REGION Network 8: PREMIXING_TEMP_CUTOUT
   RUNG wire#powerrail
      Contact( "AlwaysTRUE" )
      { S7_Templates := "SrcType := Int" } EQ_Contact(in1 := "MODE SELECTION DB"."MODE BUFF", in2 := 2)
      I_Contact( "DO MAPING"."PAV-13 WATER COOLING INLET" )
      Contact( "MANUAL BIT"."PAV-09 JACKET STEAM INLET" )
      Coil( "MANUAL BIT"."PAV-10 JACKET CONDENSATE DRAIN" )
   END_RUNG
   // the same network as SCL:
   "MANUAL BIT"."PAV-10 JACKET CONDENSATE DRAIN" := "AlwaysTRUE" AND ("MODE SELECTION DB"."MODE BUFF" = 2) AND NOT "DO MAPING"."PAV-13 WATER COOLING INLET" AND "MANUAL BIT"."PAV-09 JACKET STEAM INLET";
END_REGION

REGION Network 9: PREMIXING_COOLING_CUTOUT
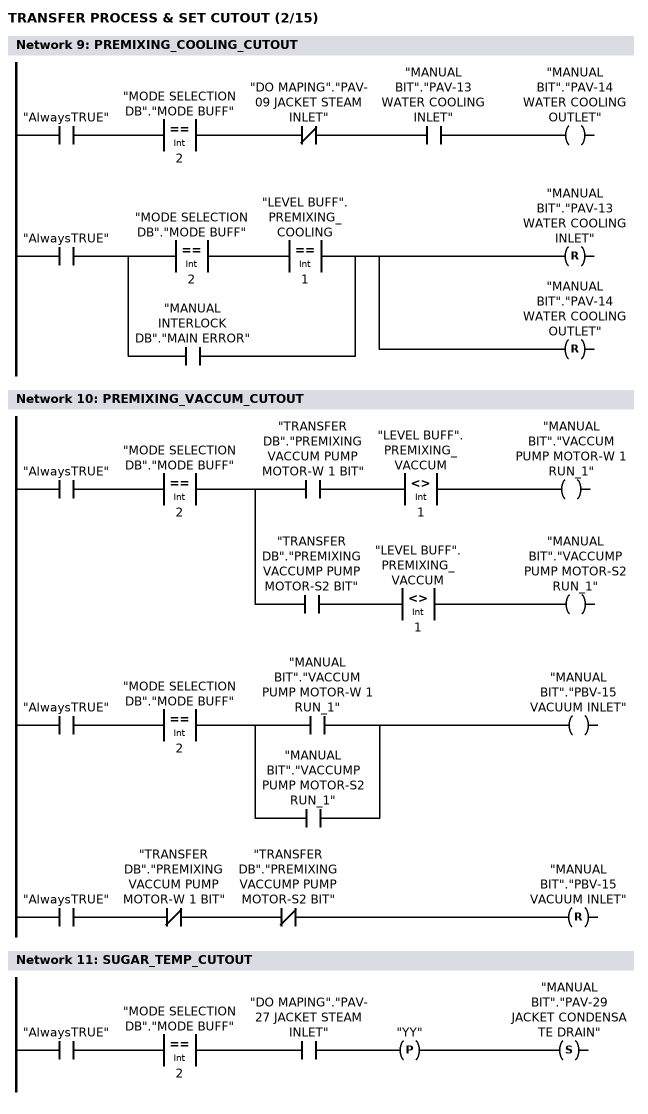
   RUNG wire#powerrail
      Contact( "AlwaysTRUE" )
      { S7_Templates := "SrcType := Int" } EQ_Contact(in1 := "MODE SELECTION DB"."MODE BUFF", in2 := 2)
      I_Contact( "DO MAPING"."PAV-09 JACKET STEAM INLET" )
      Contact( "MANUAL BIT"."PAV-13 WATER COOLING INLET" )
      Coil( "MANUAL BIT"."PAV-14 WATER COOLING OUTLET" )
   END_RUNG
   RUNG wire#powerrail
      Contact( "AlwaysTRUE" )
      wire#w1
      { S7_Templates := "SrcType := Int" } EQ_Contact(in1 := "MODE SELECTION DB"."MODE BUFF", in2 := 2)
      { S7_Templates := "SrcType := Int" } EQ_Contact(in1 := "LEVEL BUFF".PREMIXING_COOLING, in2 := 1)
      wire#w2
      R_Coil( "MANUAL BIT"."PAV-13 WATER COOLING INLET" )
   END_RUNG
   RUNG wire#w1
      Contact( "MANUAL INTERLOCK DB"."MAIN ERROR" )
   END_RUNG wire#w2
   RUNG wire#w2
      R_Coil( "MANUAL BIT"."PAV-14 WATER COOLING OUTLET" )
   END_RUNG
   // the same network as SCL:
   "MANUAL BIT"."PAV-14 WATER COOLING OUTLET" := "AlwaysTRUE" AND ("MODE SELECTION DB"."MODE BUFF" = 2) AND NOT "DO MAPING"."PAV-09 JACKET STEAM INLET" AND "MANUAL BIT"."PAV-13 WATER COOLING INLET";
   IF "AlwaysTRUE" AND ((("MODE SELECTION DB"."MODE BUFF" = 2) AND ("LEVEL BUFF".PREMIXING_COOLING = 1)) OR "MANUAL INTERLOCK DB"."MAIN ERROR") THEN
       "MANUAL BIT"."PAV-13 WATER COOLING INLET" := FALSE;
       "MANUAL BIT"."PAV-14 WATER COOLING OUTLET" := FALSE;
   END_IF;
END_REGION

REGION Network 10: PREMIXING_VACCUM_CUTOUT
   RUNG wire#powerrail
      Contact( "AlwaysTRUE" )
      { S7_Templates := "SrcType := Int" } EQ_Contact(in1 := "MODE SELECTION DB"."MODE BUFF", in2 := 2)
      wire#w1
      Contact( "TRANSFER DB"."PREMIXING VACCUM PUMP MOTOR-W 1 BIT" )
      { S7_Templates := "SrcType := Int" } NE_Contact(in1 := "LEVEL BUFF".PREMIXING_VACCUM, in2 := 1)
      Coil( "MANUAL BIT"."VACCUM PUMP MOTOR-W 1 RUN_1" )
   END_RUNG
   RUNG wire#w1
      Contact( "TRANSFER DB"."PREMIXING VACCUMP PUMP MOTOR-S2 BIT" )
      { S7_Templates := "SrcType := Int" } NE_Contact(in1 := "LEVEL BUFF".PREMIXING_VACCUM, in2 := 1)
      Coil( "MANUAL BIT"."VACCUMP PUMP MOTOR-S2 RUN_1" )
   END_RUNG
   RUNG wire#powerrail
      Contact( "AlwaysTRUE" )
      { S7_Templates := "SrcType := Int" } EQ_Contact(in1 := "MODE SELECTION DB"."MODE BUFF", in2 := 2)
      wire#w2
      Contact( "MANUAL BIT"."VACCUM PUMP MOTOR-W 1 RUN_1" )
      wire#w3
      Coil( "MANUAL BIT"."PBV-15 VACUUM INLET" )
   END_RUNG
   RUNG wire#w2
      Contact( "MANUAL BIT"."VACCUMP PUMP MOTOR-S2 RUN_1" )
   END_RUNG wire#w3
   RUNG wire#powerrail
      Contact( "AlwaysTRUE" )
      I_Contact( "TRANSFER DB"."PREMIXING VACCUM PUMP MOTOR-W 1 BIT" )
      I_Contact( "TRANSFER DB"."PREMIXING VACCUMP PUMP MOTOR-S2 BIT" )
      R_Coil( "MANUAL BIT"."PBV-15 VACUUM INLET" )
   END_RUNG
   // the same network as SCL:
   #_w1 := "AlwaysTRUE" AND ("MODE SELECTION DB"."MODE BUFF" = 2);
   "MANUAL BIT"."VACCUM PUMP MOTOR-W 1 RUN_1" := #_w1 AND "TRANSFER DB"."PREMIXING VACCUM PUMP MOTOR-W 1 BIT" AND ("LEVEL BUFF".PREMIXING_VACCUM <> 1);
   "MANUAL BIT"."VACCUMP PUMP MOTOR-S2 RUN_1" := #_w1 AND "TRANSFER DB"."PREMIXING VACCUMP PUMP MOTOR-S2 BIT" AND ("LEVEL BUFF".PREMIXING_VACCUM <> 1);
   "MANUAL BIT"."PBV-15 VACUUM INLET" := "AlwaysTRUE" AND ("MODE SELECTION DB"."MODE BUFF" = 2) AND ("MANUAL BIT"."VACCUM PUMP MOTOR-W 1 RUN_1" OR "MANUAL BIT"."VACCUMP PUMP MOTOR-S2 RUN_1");
   IF "AlwaysTRUE" AND NOT "TRANSFER DB"."PREMIXING VACCUM PUMP MOTOR-W 1 BIT" AND NOT "TRANSFER DB"."PREMIXING VACCUMP PUMP MOTOR-S2 BIT" THEN
       "MANUAL BIT"."PBV-15 VACUUM INLET" := FALSE;
   END_IF;
END_REGION

REGION Network 11: SUGAR_TEMP_CUTOUT
   RUNG wire#powerrail
      Contact( "AlwaysTRUE" )
      { S7_Templates := "SrcType := Int" } EQ_Contact(in1 := "MODE SELECTION DB"."MODE BUFF", in2 := 2)
      Contact( "DO MAPING"."PAV-27 JACKET STEAM INLET" )
      P_Trig( "YY" )
      S_Coil( "MANUAL BIT"."PAV-29 JACKET CONDENSATE DRAIN" )
   END_RUNG
   // the same network as SCL:
   #_w1 := "AlwaysTRUE" AND ("MODE SELECTION DB"."MODE BUFF" = 2) AND "DO MAPING"."PAV-27 JACKET STEAM INLET";
   #_w2 := #_w1 AND NOT "YY";   // rising edge
   "YY" := #_w1;
   IF #_w2 THEN "MANUAL BIT"."PAV-29 JACKET CONDENSATE DRAIN" := TRUE; END_IF;
END_REGION

REGION Network 12: SUGAR_VACCUM_CUTOUT
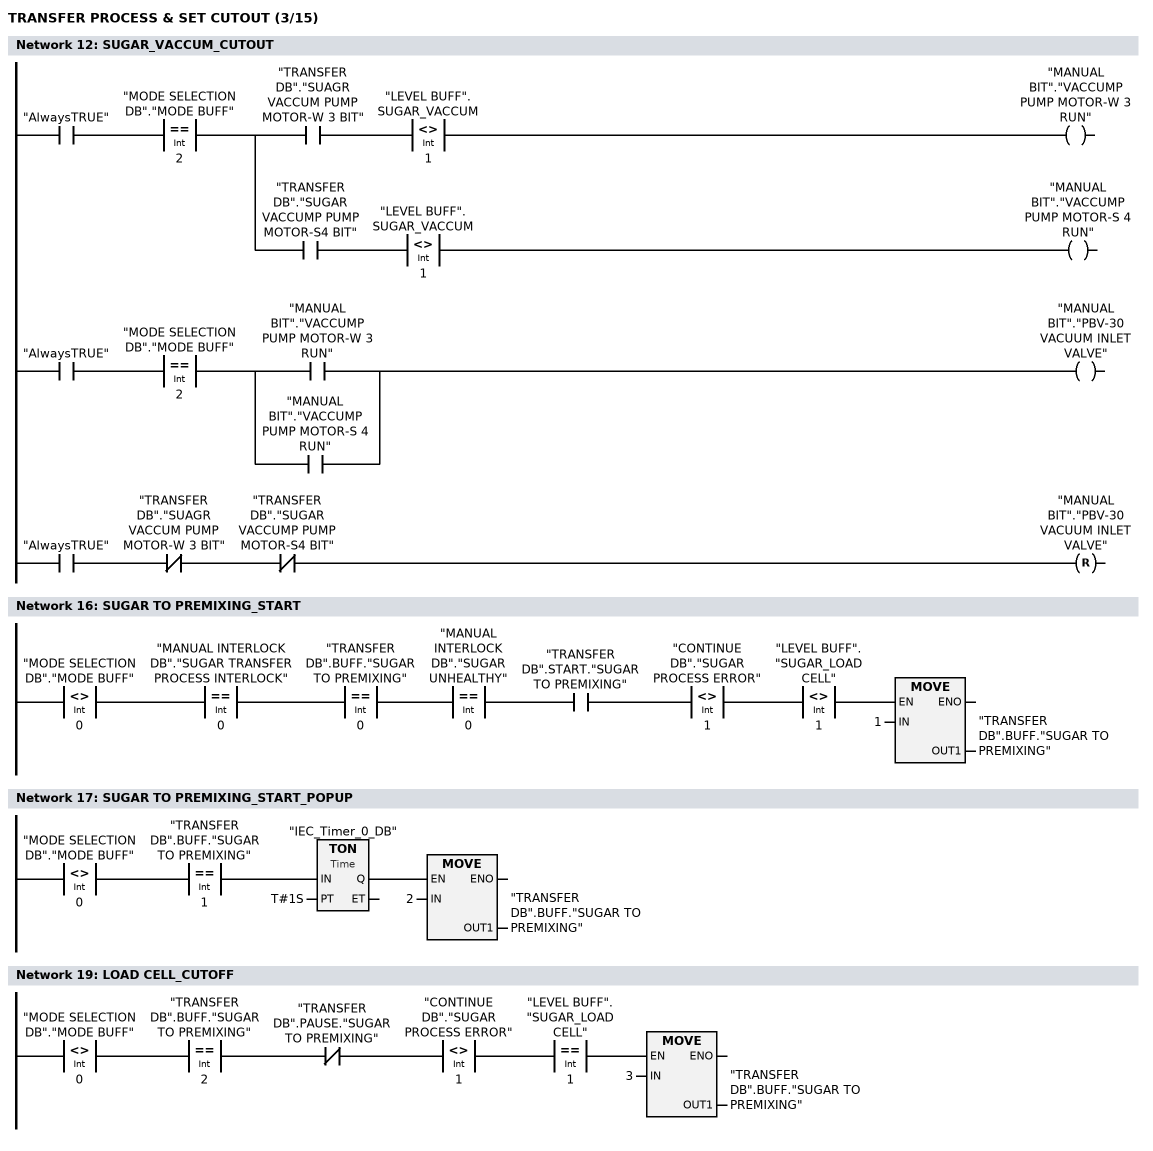
   RUNG wire#powerrail
      Contact( "AlwaysTRUE" )
      { S7_Templates := "SrcType := Int" } EQ_Contact(in1 := "MODE SELECTION DB"."MODE BUFF", in2 := 2)
      wire#w1
      Contact( "TRANSFER DB"."SUAGR VACCUM PUMP MOTOR-W 3 BIT" )
      { S7_Templates := "SrcType := Int" } NE_Contact(in1 := "LEVEL BUFF".SUGAR_VACCUM, in2 := 1)
      Coil( "MANUAL BIT"."VACCUMP PUMP MOTOR-W 3 RUN" )
   END_RUNG
   RUNG wire#w1
      Contact( "TRANSFER DB"."SUGAR VACCUMP PUMP MOTOR-S4 BIT" )
      { S7_Templates := "SrcType := Int" } NE_Contact(in1 := "LEVEL BUFF".SUGAR_VACCUM, in2 := 1)
      Coil( "MANUAL BIT"."VACCUMP PUMP MOTOR-S 4 RUN" )
   END_RUNG
   RUNG wire#powerrail
      Contact( "AlwaysTRUE" )
      { S7_Templates := "SrcType := Int" } EQ_Contact(in1 := "MODE SELECTION DB"."MODE BUFF", in2 := 2)
      wire#w2
      Contact( "MANUAL BIT"."VACCUMP PUMP MOTOR-W 3 RUN" )
      wire#w3
      Coil( "MANUAL BIT"."PBV-30 VACUUM INLET VALVE" )
   END_RUNG
   RUNG wire#w2
      Contact( "MANUAL BIT"."VACCUMP PUMP MOTOR-S 4 RUN" )
   END_RUNG wire#w3
   RUNG wire#powerrail
      Contact( "AlwaysTRUE" )
      I_Contact( "TRANSFER DB"."SUAGR VACCUM PUMP MOTOR-W 3 BIT" )
      I_Contact( "TRANSFER DB"."SUGAR VACCUMP PUMP MOTOR-S4 BIT" )
      R_Coil( "MANUAL BIT"."PBV-30 VACUUM INLET VALVE" )
   END_RUNG
   // the same network as SCL:
   #_w1 := "AlwaysTRUE" AND ("MODE SELECTION DB"."MODE BUFF" = 2);
   "MANUAL BIT"."VACCUMP PUMP MOTOR-W 3 RUN" := #_w1 AND "TRANSFER DB"."SUAGR VACCUM PUMP MOTOR-W 3 BIT" AND ("LEVEL BUFF".SUGAR_VACCUM <> 1);
   "MANUAL BIT"."VACCUMP PUMP MOTOR-S 4 RUN" := #_w1 AND "TRANSFER DB"."SUGAR VACCUMP PUMP MOTOR-S4 BIT" AND ("LEVEL BUFF".SUGAR_VACCUM <> 1);
   "MANUAL BIT"."PBV-30 VACUUM INLET VALVE" := "AlwaysTRUE" AND ("MODE SELECTION DB"."MODE BUFF" = 2) AND ("MANUAL BIT"."VACCUMP PUMP MOTOR-W 3 RUN" OR "MANUAL BIT"."VACCUMP PUMP MOTOR-S 4 RUN");
   IF "AlwaysTRUE" AND NOT "TRANSFER DB"."SUAGR VACCUM PUMP MOTOR-W 3 BIT" AND NOT "TRANSFER DB"."SUGAR VACCUMP PUMP MOTOR-S4 BIT" THEN
       "MANUAL BIT"."PBV-30 VACUUM INLET VALVE" := FALSE;
   END_IF;
END_REGION

REGION Network 15: ////////////////////////////////////////////////////////////////////// TRANSFER PROCESS- SUGAR //////////////////////////////////////////////////////////////////////////////////
END_REGION

REGION Network 16: SUGAR TO PREMIXING_START
   RUNG wire#powerrail
      { S7_Templates := "SrcType := Int" } NE_Contact(in1 := "MODE SELECTION DB"."MODE BUFF", in2 := 0)
      { S7_Templates := "SrcType := Int" } EQ_Contact(in1 := "MANUAL INTERLOCK DB"."SUGAR TRANSFER PROCESS INTERLOCK", in2 := 0)
      { S7_Templates := "SrcType := Int" } EQ_Contact(in1 := "TRANSFER DB".BUFF."SUGAR TO PREMIXING", in2 := 0)
      { S7_Templates := "SrcType := Int" } EQ_Contact(in1 := "MANUAL INTERLOCK DB"."SUGAR UNHEALTHY", in2 := 0)
      Contact( "TRANSFER DB".START."SUGAR TO PREMIXING" )
      { S7_Templates := "SrcType := Int" } NE_Contact(in1 := "CONTINUE DB"."SUGAR PROCESS ERROR", in2 := 1)
      { S7_Templates := "SrcType := Int" } NE_Contact(in1 := "LEVEL BUFF"."SUGAR_LOAD CELL", in2 := 1)
      Move(in := 1, out1 => "TRANSFER DB".BUFF."SUGAR TO PREMIXING")
   END_RUNG
   // the same network as SCL:
   IF ("MODE SELECTION DB"."MODE BUFF" <> 0) AND ("MANUAL INTERLOCK DB"."SUGAR TRANSFER PROCESS INTERLOCK" = 0) AND ("TRANSFER DB".BUFF."SUGAR TO PREMIXING" = 0) AND ("MANUAL INTERLOCK DB"."SUGAR UNHEALTHY" = 0) AND "TRANSFER DB".START."SUGAR TO PREMIXING" AND ("CONTINUE DB"."SUGAR PROCESS ERROR" <> 1) AND ("LEVEL BUFF"."SUGAR_LOAD CELL" <> 1) THEN
       "TRANSFER DB".BUFF."SUGAR TO PREMIXING" := 1;
   END_IF;
END_REGION

REGION Network 17: SUGAR TO PREMIXING_START_POPUP
   RUNG wire#powerrail
      { S7_Templates := "SrcType := Int" } NE_Contact(in1 := "MODE SELECTION DB"."MODE BUFF", in2 := 0)
      { S7_Templates := "SrcType := Int" } EQ_Contact(in1 := "TRANSFER DB".BUFF."SUGAR TO PREMIXING", in2 := 1)
      { S7_Templates := "time_type := Time" } "IEC_Timer_0_DB".TON(pt := T#1S, et =>)
      Move(in := 2, out1 => "TRANSFER DB".BUFF."SUGAR TO PREMIXING")
   END_RUNG
   // the same network as SCL:
   "IEC_Timer_0_DB".TON(IN := ("MODE SELECTION DB"."MODE BUFF" <> 0) AND ("TRANSFER DB".BUFF."SUGAR TO PREMIXING" = 1),
                        PT := T#1S);
   IF "IEC_Timer_0_DB".Q THEN "TRANSFER DB".BUFF."SUGAR TO PREMIXING" := 2; END_IF;
END_REGION

REGION Network 18 (SCL): OPENVALVE
   IF "MODE SELECTION DB"."MODE BUFF" <> 0 AND "TRANSFER DB".BUFF."SUGAR TO PREMIXING" = 2
       AND NOT "TRANSFER DB".PAUSE."SUGAR TO PREMIXING" AND
       "CONTINUE DB"."SUGAR PROCESS ERROR" = 0 AND "LEVEL BUFF"."SUGAR_LOAD CELL" = 0
       OR ("MODE SELECTION DB"."MODE BUFF"=1 AND "SUGAR DB"."AUTO BUFF"=105
       AND "CONTINUE DB"."SUGAR PROCESS ERROR" <>1)
   THEN
       "TRANSFER DB".BIT."SUGAR TO PREMIXING"."PFBV-32 TANK OUTLET VALVE" := TRUE;
       "TRANSFER DB".BIT."SUGAR TO PREMIXING"."PBV-80 BOTTOM OUTLET TO BASKET FILTER" := TRUE;
       "TRANSFER DB".BIT."SUGAR TO PREMIXING"."BASKET FILTER MOTOR RUN" := TRUE;
       "TRANSFER DB".BIT."SUGAR TO PREMIXING"."PBV-79 BASKET FILTER INLET" := TRUE;
       "TRANSFER DB".BIT."SUGAR TO PREMIXING"."PBV-149" := TRUE;
       "TRANSFER DB".BIT."SUGAR TO PREMIXING"."PBV-88 BASKET FILTER TRANSFER LINE" := TRUE;
       "TRANSFER DB".BIT."SUGAR TO PREMIXING"."PBV-87 BASKET FILTER TO PREMIX VESSEL LINE" := TRUE;
   ELSE
       "TRANSFER DB".BIT."SUGAR TO PREMIXING"."PFBV-32 TANK OUTLET VALVE" := FALSE;
       "TRANSFER DB".BIT."SUGAR TO PREMIXING"."PBV-80 BOTTOM OUTLET TO BASKET FILTER" := FALSE;
       "TRANSFER DB".BIT."SUGAR TO PREMIXING"."BASKET FILTER MOTOR RUN" := FALSE;
       "TRANSFER DB".BIT."SUGAR TO PREMIXING"."PBV-79 BASKET FILTER INLET" := FALSE;
       "TRANSFER DB".BIT."SUGAR TO PREMIXING"."PBV-149" := FALSE;
       "TRANSFER DB".BIT."SUGAR TO PREMIXING"."PBV-88 BASKET FILTER TRANSFER LINE" := FALSE;
       "TRANSFER DB".BIT."SUGAR TO PREMIXING"."PBV-87 BASKET FILTER TO PREMIX VESSEL LINE" := FALSE;
       ;
   END_IF;
END_REGION

REGION Network 19: LOAD CELL_CUTOFF
   RUNG wire#powerrail
      { S7_Templates := "SrcType := Int" } NE_Contact(in1 := "MODE SELECTION DB"."MODE BUFF", in2 := 0)
      { S7_Templates := "SrcType := Int" } EQ_Contact(in1 := "TRANSFER DB".BUFF."SUGAR TO PREMIXING", in2 := 2)
      I_Contact( "TRANSFER DB".PAUSE."SUGAR TO PREMIXING" )
      { S7_Templates := "SrcType := Int" } NE_Contact(in1 := "CONTINUE DB"."SUGAR PROCESS ERROR", in2 := 1)
      { S7_Templates := "SrcType := Int" } EQ_Contact(in1 := "LEVEL BUFF"."SUGAR_LOAD CELL", in2 := 1)
      Move(in := 3, out1 => "TRANSFER DB".BUFF."SUGAR TO PREMIXING")
   END_RUNG
   // the same network as SCL:
   IF ("MODE SELECTION DB"."MODE BUFF" <> 0) AND ("TRANSFER DB".BUFF."SUGAR TO PREMIXING" = 2) AND NOT "TRANSFER DB".PAUSE."SUGAR TO PREMIXING" AND ("CONTINUE DB"."SUGAR PROCESS ERROR" <> 1) AND ("LEVEL BUFF"."SUGAR_LOAD CELL" = 1) THEN
       "TRANSFER DB".BUFF."SUGAR TO PREMIXING" := 3;
   END_IF;
END_REGION

REGION Network 20: PROCESS OVER & STOP
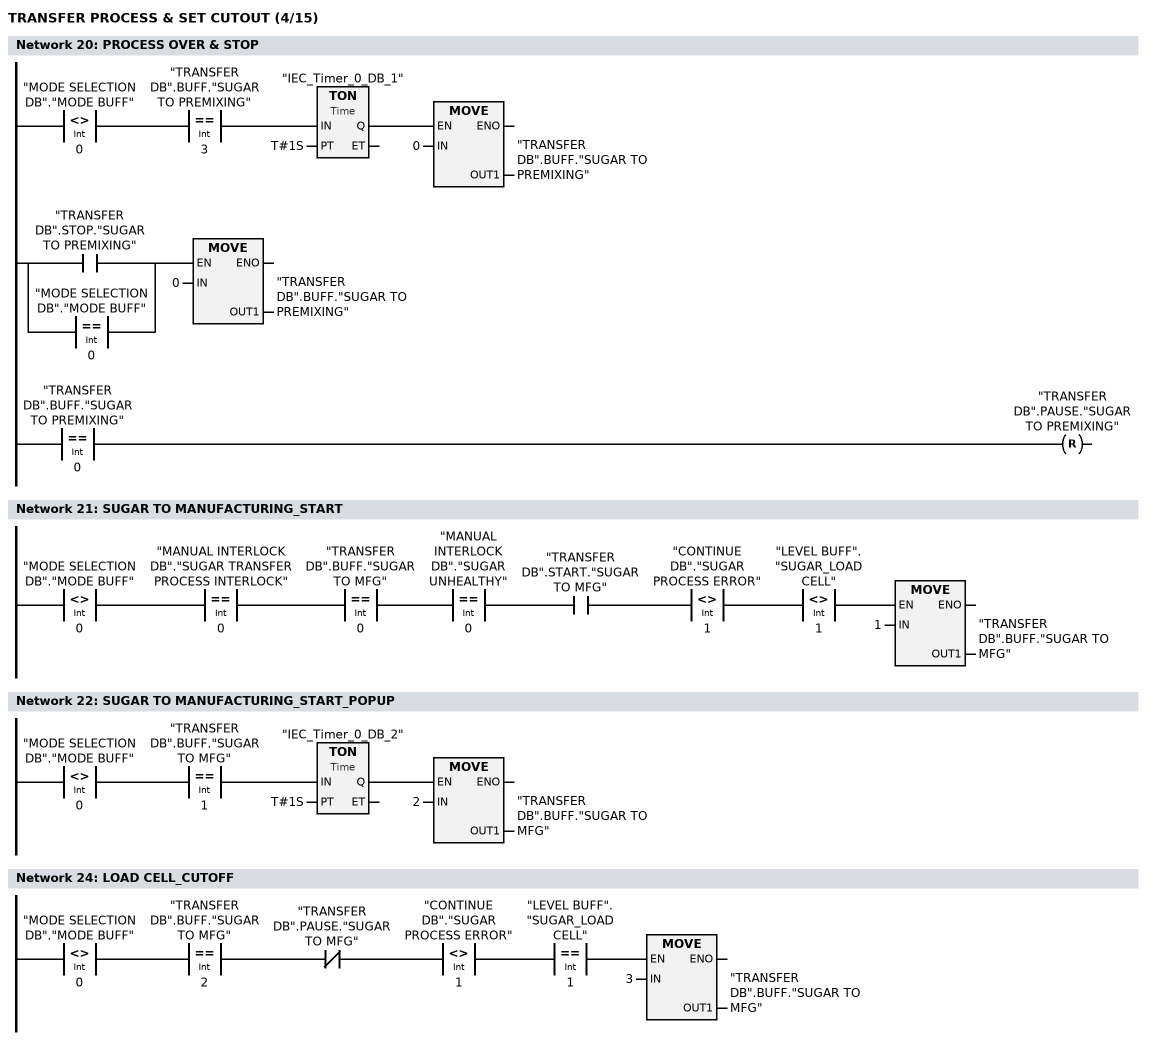
   RUNG wire#powerrail
      { S7_Templates := "SrcType := Int" } NE_Contact(in1 := "MODE SELECTION DB"."MODE BUFF", in2 := 0)
      { S7_Templates := "SrcType := Int" } EQ_Contact(in1 := "TRANSFER DB".BUFF."SUGAR TO PREMIXING", in2 := 3)
      { S7_Templates := "time_type := Time" } "IEC_Timer_0_DB_1".TON(pt := T#1S, et =>)
      Move(in := 0, out1 => "TRANSFER DB".BUFF."SUGAR TO PREMIXING")
   END_RUNG
   RUNG wire#powerrail
      Contact( "TRANSFER DB".STOP."SUGAR TO PREMIXING" )
      wire#w1
      Move(in := 0, out1 => "TRANSFER DB".BUFF."SUGAR TO PREMIXING")
   END_RUNG
   RUNG wire#powerrail
      { S7_Templates := "SrcType := Int" } EQ_Contact(in1 := "MODE SELECTION DB"."MODE BUFF", in2 := 0)
   END_RUNG wire#w1
   RUNG wire#powerrail
      { S7_Templates := "SrcType := Int" } EQ_Contact(in1 := "TRANSFER DB".BUFF."SUGAR TO PREMIXING", in2 := 0)
      R_Coil( "TRANSFER DB".PAUSE."SUGAR TO PREMIXING" )
   END_RUNG
   // the same network as SCL:
   "IEC_Timer_0_DB_1".TON(IN := ("MODE SELECTION DB"."MODE BUFF" <> 0) AND ("TRANSFER DB".BUFF."SUGAR TO PREMIXING" = 3),
                          PT := T#1S);
   IF "IEC_Timer_0_DB_1".Q THEN "TRANSFER DB".BUFF."SUGAR TO PREMIXING" := 0; END_IF;
   IF "TRANSFER DB".STOP."SUGAR TO PREMIXING" OR ("MODE SELECTION DB"."MODE BUFF" = 0) THEN
       "TRANSFER DB".BUFF."SUGAR TO PREMIXING" := 0;
   END_IF;
   IF "TRANSFER DB".BUFF."SUGAR TO PREMIXING" = 0 THEN
       "TRANSFER DB".PAUSE."SUGAR TO PREMIXING" := FALSE;
   END_IF;
END_REGION

REGION Network 21: SUGAR TO MANUFACTURING_START
   RUNG wire#powerrail
      { S7_Templates := "SrcType := Int" } NE_Contact(in1 := "MODE SELECTION DB"."MODE BUFF", in2 := 0)
      { S7_Templates := "SrcType := Int" } EQ_Contact(in1 := "MANUAL INTERLOCK DB"."SUGAR TRANSFER PROCESS INTERLOCK", in2 := 0)
      { S7_Templates := "SrcType := Int" } EQ_Contact(in1 := "TRANSFER DB".BUFF."SUGAR TO MFG", in2 := 0)
      { S7_Templates := "SrcType := Int" } EQ_Contact(in1 := "MANUAL INTERLOCK DB"."SUGAR UNHEALTHY", in2 := 0)
      Contact( "TRANSFER DB".START."SUGAR TO MFG" )
      { S7_Templates := "SrcType := Int" } NE_Contact(in1 := "CONTINUE DB"."SUGAR PROCESS ERROR", in2 := 1)
      { S7_Templates := "SrcType := Int" } NE_Contact(in1 := "LEVEL BUFF"."SUGAR_LOAD CELL", in2 := 1)
      Move(in := 1, out1 => "TRANSFER DB".BUFF."SUGAR TO MFG")
   END_RUNG
   // the same network as SCL:
   IF ("MODE SELECTION DB"."MODE BUFF" <> 0) AND ("MANUAL INTERLOCK DB"."SUGAR TRANSFER PROCESS INTERLOCK" = 0) AND ("TRANSFER DB".BUFF."SUGAR TO MFG" = 0) AND ("MANUAL INTERLOCK DB"."SUGAR UNHEALTHY" = 0) AND "TRANSFER DB".START."SUGAR TO MFG" AND ("CONTINUE DB"."SUGAR PROCESS ERROR" <> 1) AND ("LEVEL BUFF"."SUGAR_LOAD CELL" <> 1) THEN
       "TRANSFER DB".BUFF."SUGAR TO MFG" := 1;
   END_IF;
END_REGION

REGION Network 22: SUGAR TO MANUFACTURING_START_POPUP
   RUNG wire#powerrail
      { S7_Templates := "SrcType := Int" } NE_Contact(in1 := "MODE SELECTION DB"."MODE BUFF", in2 := 0)
      { S7_Templates := "SrcType := Int" } EQ_Contact(in1 := "TRANSFER DB".BUFF."SUGAR TO MFG", in2 := 1)
      { S7_Templates := "time_type := Time" } "IEC_Timer_0_DB_2".TON(pt := T#1S, et =>)
      Move(in := 2, out1 => "TRANSFER DB".BUFF."SUGAR TO MFG")
   END_RUNG
   // the same network as SCL:
   "IEC_Timer_0_DB_2".TON(IN := ("MODE SELECTION DB"."MODE BUFF" <> 0) AND ("TRANSFER DB".BUFF."SUGAR TO MFG" = 1),
                          PT := T#1S);
   IF "IEC_Timer_0_DB_2".Q THEN "TRANSFER DB".BUFF."SUGAR TO MFG" := 2; END_IF;
END_REGION

REGION Network 23 (SCL): OPENVALVE
   IF "MODE SELECTION DB"."MODE BUFF" <> 0 AND "TRANSFER DB".BUFF."SUGAR TO MFG" = 2
       AND NOT "TRANSFER DB".PAUSE."SUGAR TO MFG" 
       AND "CONTINUE DB"."SUGAR PROCESS ERROR" = 0 AND "LEVEL BUFF"."SUGAR_LOAD CELL" = 0
       OR ("MODE SELECTION DB"."MODE BUFF"=1 AND "SUGAR DB"."AUTO BUFF"=125
       AND "CONTINUE DB"."SUGAR PROCESS ERROR" <>1)
   THEN
       "TRANSFER DB".BIT."SUGAR TO MFG"."PFBV-32 TANK OUTLET VALVE" := TRUE;
       "TRANSFER DB".BIT."SUGAR TO MFG"."PBV-80 BOTTOM OUTLET TO BASKET FILTER" := TRUE;
       "TRANSFER DB".BIT."SUGAR TO MFG"."BASKET FILTER MOTOR RUN" := TRUE;
       "TRANSFER DB".BIT."SUGAR TO MFG"."PBV-79 BASKET FILTER INLET" := TRUE;
       "TRANSFER DB".BIT."SUGAR TO MFG"."PBV-149" := TRUE;
       "TRANSFER DB".BIT."SUGAR TO MFG"."PBV-89 BASKET FILTER TO MFG INLET TRANSFER LINE" := TRUE;
       "TRANSFER DB".BIT."SUGAR TO MFG"."PBV-101 SUGAR MELTING TO MFG TRANSFER (TOP DISH)" := TRUE;

   ELSE
       "TRANSFER DB".BIT."SUGAR TO MFG"."PFBV-32 TANK OUTLET VALVE" := FALSE;
       "TRANSFER DB".BIT."SUGAR TO MFG"."PBV-80 BOTTOM OUTLET TO BASKET FILTER" := FALSE;
       "TRANSFER DB".BIT."SUGAR TO MFG"."BASKET FILTER MOTOR RUN" := FALSE;
       "TRANSFER DB".BIT."SUGAR TO MFG"."PBV-79 BASKET FILTER INLET" := FALSE;
       "TRANSFER DB".BIT."SUGAR TO MFG"."PBV-149" := FALSE;
       "TRANSFER DB".BIT."SUGAR TO MFG"."PBV-89 BASKET FILTER TO MFG INLET TRANSFER LINE" := FALSE;
       "TRANSFER DB".BIT."SUGAR TO MFG"."PBV-101 SUGAR MELTING TO MFG TRANSFER (TOP DISH)" := FALSE;
       ;
   END_IF;
END_REGION

REGION Network 24: LOAD CELL_CUTOFF
   RUNG wire#powerrail
      { S7_Templates := "SrcType := Int" } NE_Contact(in1 := "MODE SELECTION DB"."MODE BUFF", in2 := 0)
      { S7_Templates := "SrcType := Int" } EQ_Contact(in1 := "TRANSFER DB".BUFF."SUGAR TO MFG", in2 := 2)
      I_Contact( "TRANSFER DB".PAUSE."SUGAR TO MFG" )
      { S7_Templates := "SrcType := Int" } NE_Contact(in1 := "CONTINUE DB"."SUGAR PROCESS ERROR", in2 := 1)
      { S7_Templates := "SrcType := Int" } EQ_Contact(in1 := "LEVEL BUFF"."SUGAR_LOAD CELL", in2 := 1)
      Move(in := 3, out1 => "TRANSFER DB".BUFF."SUGAR TO MFG")
   END_RUNG
   // the same network as SCL:
   IF ("MODE SELECTION DB"."MODE BUFF" <> 0) AND ("TRANSFER DB".BUFF."SUGAR TO MFG" = 2) AND NOT "TRANSFER DB".PAUSE."SUGAR TO MFG" AND ("CONTINUE DB"."SUGAR PROCESS ERROR" <> 1) AND ("LEVEL BUFF"."SUGAR_LOAD CELL" = 1) THEN
       "TRANSFER DB".BUFF."SUGAR TO MFG" := 3;
   END_IF;
END_REGION

REGION Network 25: PROCESS OVER & STOP
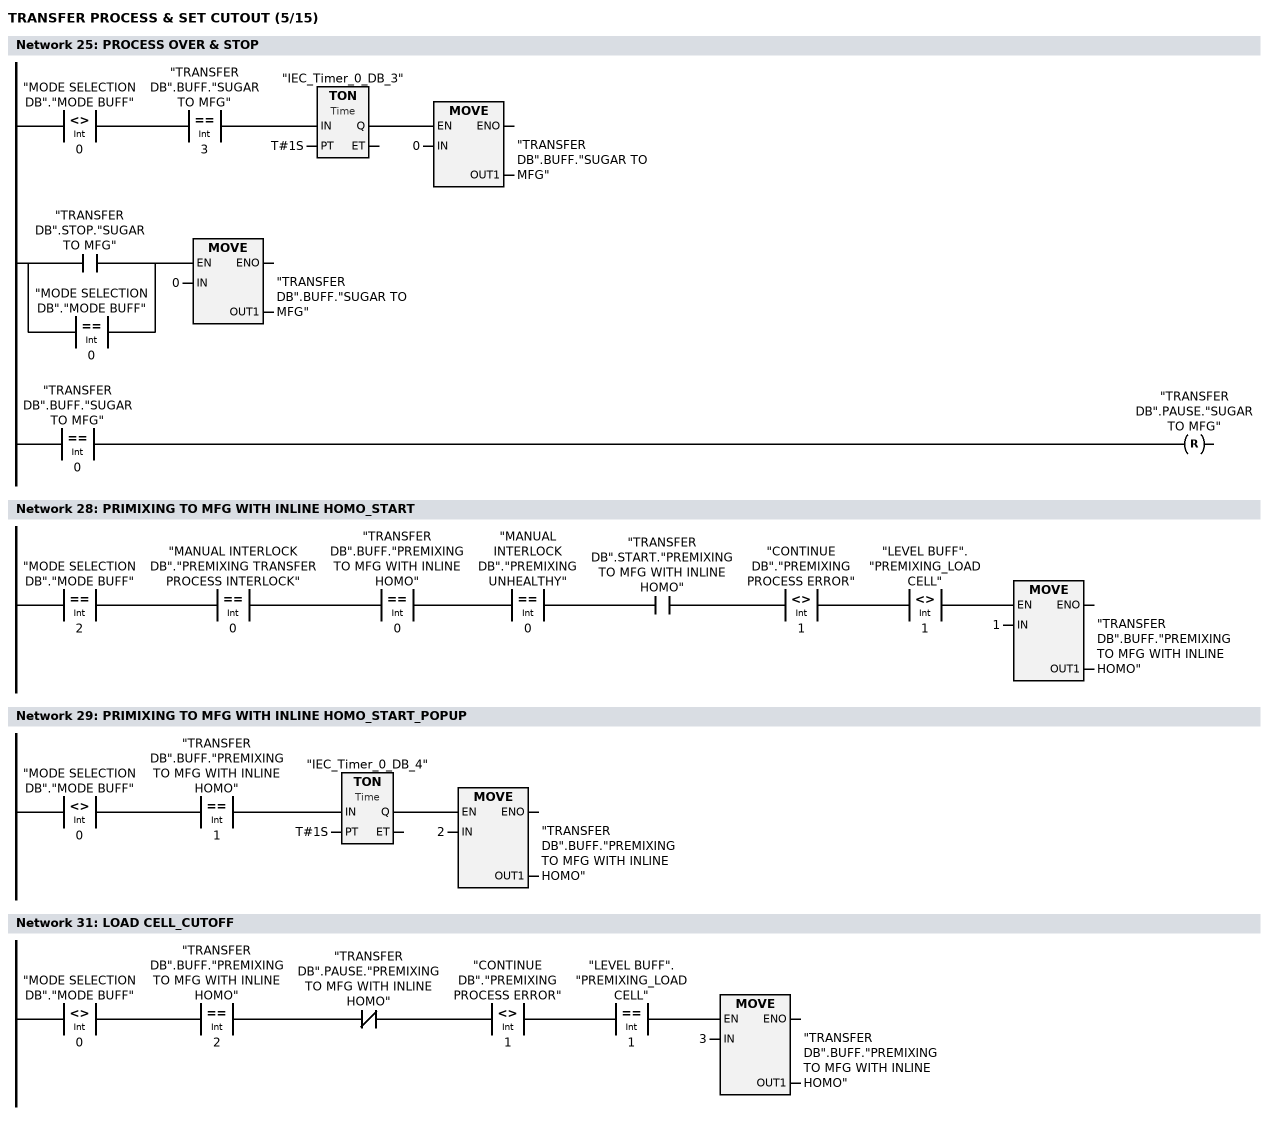
   RUNG wire#powerrail
      { S7_Templates := "SrcType := Int" } NE_Contact(in1 := "MODE SELECTION DB"."MODE BUFF", in2 := 0)
      { S7_Templates := "SrcType := Int" } EQ_Contact(in1 := "TRANSFER DB".BUFF."SUGAR TO MFG", in2 := 3)
      { S7_Templates := "time_type := Time" } "IEC_Timer_0_DB_3".TON(pt := T#1S, et =>)
      Move(in := 0, out1 => "TRANSFER DB".BUFF."SUGAR TO MFG")
   END_RUNG
   RUNG wire#powerrail
      Contact( "TRANSFER DB".STOP."SUGAR TO MFG" )
      wire#w1
      Move(in := 0, out1 => "TRANSFER DB".BUFF."SUGAR TO MFG")
   END_RUNG
   RUNG wire#powerrail
      { S7_Templates := "SrcType := Int" } EQ_Contact(in1 := "MODE SELECTION DB"."MODE BUFF", in2 := 0)
   END_RUNG wire#w1
   RUNG wire#powerrail
      { S7_Templates := "SrcType := Int" } EQ_Contact(in1 := "TRANSFER DB".BUFF."SUGAR TO MFG", in2 := 0)
      R_Coil( "TRANSFER DB".PAUSE."SUGAR TO MFG" )
   END_RUNG
   // the same network as SCL:
   "IEC_Timer_0_DB_3".TON(IN := ("MODE SELECTION DB"."MODE BUFF" <> 0) AND ("TRANSFER DB".BUFF."SUGAR TO MFG" = 3),
                          PT := T#1S);
   IF "IEC_Timer_0_DB_3".Q THEN "TRANSFER DB".BUFF."SUGAR TO MFG" := 0; END_IF;
   IF "TRANSFER DB".STOP."SUGAR TO MFG" OR ("MODE SELECTION DB"."MODE BUFF" = 0) THEN
       "TRANSFER DB".BUFF."SUGAR TO MFG" := 0;
   END_IF;
   IF "TRANSFER DB".BUFF."SUGAR TO MFG" = 0 THEN "TRANSFER DB".PAUSE."SUGAR TO MFG" := FALSE; END_IF;
END_REGION

REGION Network 27: ////////////////////////////////////////////////////////////////////// TRANSFER PROCESS- PREMIXING //////////////////////////////////////////////////////////////////////////////////
END_REGION

REGION Network 28: PRIMIXING TO MFG WITH INLINE HOMO_START
   RUNG wire#powerrail
      { S7_Templates := "SrcType := Int" } EQ_Contact(in1 := "MODE SELECTION DB"."MODE BUFF", in2 := 2)
      { S7_Templates := "SrcType := Int" } EQ_Contact(in1 := "MANUAL INTERLOCK DB"."PREMIXING TRANSFER PROCESS INTERLOCK", in2 := 0)
      { S7_Templates := "SrcType := Int" } EQ_Contact(in1 := "TRANSFER DB".BUFF."PREMIXING TO MFG WITH INLINE HOMO", in2 := 0)
      { S7_Templates := "SrcType := Int" } EQ_Contact(in1 := "MANUAL INTERLOCK DB"."PREMIXING UNHEALTHY", in2 := 0)
      Contact( "TRANSFER DB".START."PREMIXING TO MFG WITH INLINE HOMO" )
      { S7_Templates := "SrcType := Int" } NE_Contact(in1 := "CONTINUE DB"."PREMIXING PROCESS ERROR", in2 := 1)
      { S7_Templates := "SrcType := Int" } NE_Contact(in1 := "LEVEL BUFF"."PREMIXING_LOAD CELL", in2 := 1)
      Move(in := 1, out1 => "TRANSFER DB".BUFF."PREMIXING TO MFG WITH INLINE HOMO")
   END_RUNG
   // the same network as SCL:
   IF ("MODE SELECTION DB"."MODE BUFF" = 2) AND ("MANUAL INTERLOCK DB"."PREMIXING TRANSFER PROCESS INTERLOCK" = 0) AND ("TRANSFER DB".BUFF."PREMIXING TO MFG WITH INLINE HOMO" = 0) AND ("MANUAL INTERLOCK DB"."PREMIXING UNHEALTHY" = 0) AND "TRANSFER DB".START."PREMIXING TO MFG WITH INLINE HOMO" AND ("CONTINUE DB"."PREMIXING PROCESS ERROR" <> 1) AND ("LEVEL BUFF"."PREMIXING_LOAD CELL" <> 1) THEN
       "TRANSFER DB".BUFF."PREMIXING TO MFG WITH INLINE HOMO" := 1;
   END_IF;
END_REGION

REGION Network 29: PRIMIXING TO MFG WITH INLINE HOMO_START_POPUP
   RUNG wire#powerrail
      { S7_Templates := "SrcType := Int" } NE_Contact(in1 := "MODE SELECTION DB"."MODE BUFF", in2 := 0)
      { S7_Templates := "SrcType := Int" } EQ_Contact(in1 := "TRANSFER DB".BUFF."PREMIXING TO MFG WITH INLINE HOMO", in2 := 1)
      { S7_Templates := "time_type := Time" } "IEC_Timer_0_DB_4".TON(pt := T#1S, et =>)
      Move(in := 2, out1 => "TRANSFER DB".BUFF."PREMIXING TO MFG WITH INLINE HOMO")
   END_RUNG
   // the same network as SCL:
   "IEC_Timer_0_DB_4".TON(IN := ("MODE SELECTION DB"."MODE BUFF" <> 0) AND ("TRANSFER DB".BUFF."PREMIXING TO MFG WITH INLINE HOMO" = 1),
                          PT := T#1S);
   IF "IEC_Timer_0_DB_4".Q THEN "TRANSFER DB".BUFF."PREMIXING TO MFG WITH INLINE HOMO" := 2; END_IF;
END_REGION

REGION Network 30 (SCL): OPENVALVE
   IF "MODE SELECTION DB"."MODE BUFF" <> 0 AND "TRANSFER DB".BUFF."PREMIXING TO MFG WITH INLINE HOMO" = 2
       AND NOT "TRANSFER DB".PAUSE."PREMIXING TO MFG WITH INLINE HOMO" 
       AND "CONTINUE DB"."PREMIXING PROCESS ERROR" = 0 AND "LEVEL BUFF"."PREMIXING_LOAD CELL" = 0
       OR ("MODE SELECTION DB"."MODE BUFF"=1 AND "PREMIXING DB"."AUTO BUFF"=0
       AND "PREMIXING TRANSFER CYCLE DB".TRANSFER."TRANSFER BUFF"."PREMIXING TO MFG WITH INLINE HOMO"=10 AND "CONTINUE DB"."PREMIXING PROCESS ERROR" <>1
       AND "PREMIXING TRANSFER CYCLE DB".TRANSFER.SELECT."SELECT BUFF"=1)
   THEN
       "TRANSFER DB".BIT."PREMIXING TO MFG WITH INLINE HOMO"."PFBV-17 TANK OUTLET VALVE" := TRUE;
       "TRANSFER DB".BIT."PREMIXING TO MFG WITH INLINE HOMO"."PBV-93 TANK OUTLET TO INLINE HOMOGENIZER LINE" := TRUE;
       "TRANSFER DB".BIT."PREMIXING TO MFG WITH INLINE HOMO"."PBV-94 INLINE HOMOGENIZER INLET LINE" := TRUE;
       "TRANSFER DB".BIT."PREMIXING TO MFG WITH INLINE HOMO"."PAV-99 INLINE HOMOGENIZER SEAL COOLING" := TRUE;
       "TRANSFER DB".BIT."PREMIXING TO MFG WITH INLINE HOMO"."INLINE 2 HOMOGENIZER MOTOR 2 RUN" := TRUE;
       "TRANSFER DB".BIT."PREMIXING TO MFG WITH INLINE HOMO"."PBV-96 INLINE HOMOGENIZER RECIRCULATION LINE" := TRUE;
       "TRANSFER DB".BIT."PREMIXING TO MFG WITH INLINE HOMO"."PBV-91 PREMIX TO MFG TRANSFER LINE" := TRUE;
       "TRANSFER DB".BIT."PREMIXING TO MFG WITH INLINE HOMO"."PBV-102 PREMIX TO MFG TRANSFER (TOP DISH)" := TRUE;

   ELSE
       "TRANSFER DB".BIT."PREMIXING TO MFG WITH INLINE HOMO"."PFBV-17 TANK OUTLET VALVE" := FALSE;
       "TRANSFER DB".BIT."PREMIXING TO MFG WITH INLINE HOMO"."PBV-93 TANK OUTLET TO INLINE HOMOGENIZER LINE" := FALSE;
       "TRANSFER DB".BIT."PREMIXING TO MFG WITH INLINE HOMO"."PBV-94 INLINE HOMOGENIZER INLET LINE" := FALSE;
       "TRANSFER DB".BIT."PREMIXING TO MFG WITH INLINE HOMO"."PAV-99 INLINE HOMOGENIZER SEAL COOLING" := FALSE;
       "TRANSFER DB".BIT."PREMIXING TO MFG WITH INLINE HOMO"."INLINE 2 HOMOGENIZER MOTOR 2 RUN" := FALSE;
       "TRANSFER DB".BIT."PREMIXING TO MFG WITH INLINE HOMO"."PBV-96 INLINE HOMOGENIZER RECIRCULATION LINE" := FALSE;
       "TRANSFER DB".BIT."PREMIXING TO MFG WITH INLINE HOMO"."PBV-91 PREMIX TO MFG TRANSFER LINE" := FALSE;
       "TRANSFER DB".BIT."PREMIXING TO MFG WITH INLINE HOMO"."PBV-102 PREMIX TO MFG TRANSFER (TOP DISH)" := FALSE;
       ;
   END_IF;
END_REGION

REGION Network 31: LOAD CELL_CUTOFF
   RUNG wire#powerrail
      { S7_Templates := "SrcType := Int" } NE_Contact(in1 := "MODE SELECTION DB"."MODE BUFF", in2 := 0)
      { S7_Templates := "SrcType := Int" } EQ_Contact(in1 := "TRANSFER DB".BUFF."PREMIXING TO MFG WITH INLINE HOMO", in2 := 2)
      I_Contact( "TRANSFER DB".PAUSE."PREMIXING TO MFG WITH INLINE HOMO" )
      { S7_Templates := "SrcType := Int" } NE_Contact(in1 := "CONTINUE DB"."PREMIXING PROCESS ERROR", in2 := 1)
      { S7_Templates := "SrcType := Int" } EQ_Contact(in1 := "LEVEL BUFF"."PREMIXING_LOAD CELL", in2 := 1)
      Move(in := 3, out1 => "TRANSFER DB".BUFF."PREMIXING TO MFG WITH INLINE HOMO")
   END_RUNG
   // the same network as SCL:
   IF ("MODE SELECTION DB"."MODE BUFF" <> 0) AND ("TRANSFER DB".BUFF."PREMIXING TO MFG WITH INLINE HOMO" = 2) AND NOT "TRANSFER DB".PAUSE."PREMIXING TO MFG WITH INLINE HOMO" AND ("CONTINUE DB"."PREMIXING PROCESS ERROR" <> 1) AND ("LEVEL BUFF"."PREMIXING_LOAD CELL" = 1) THEN
       "TRANSFER DB".BUFF."PREMIXING TO MFG WITH INLINE HOMO" := 3;
   END_IF;
END_REGION

REGION Network 32: PROCESS OVER & STOP
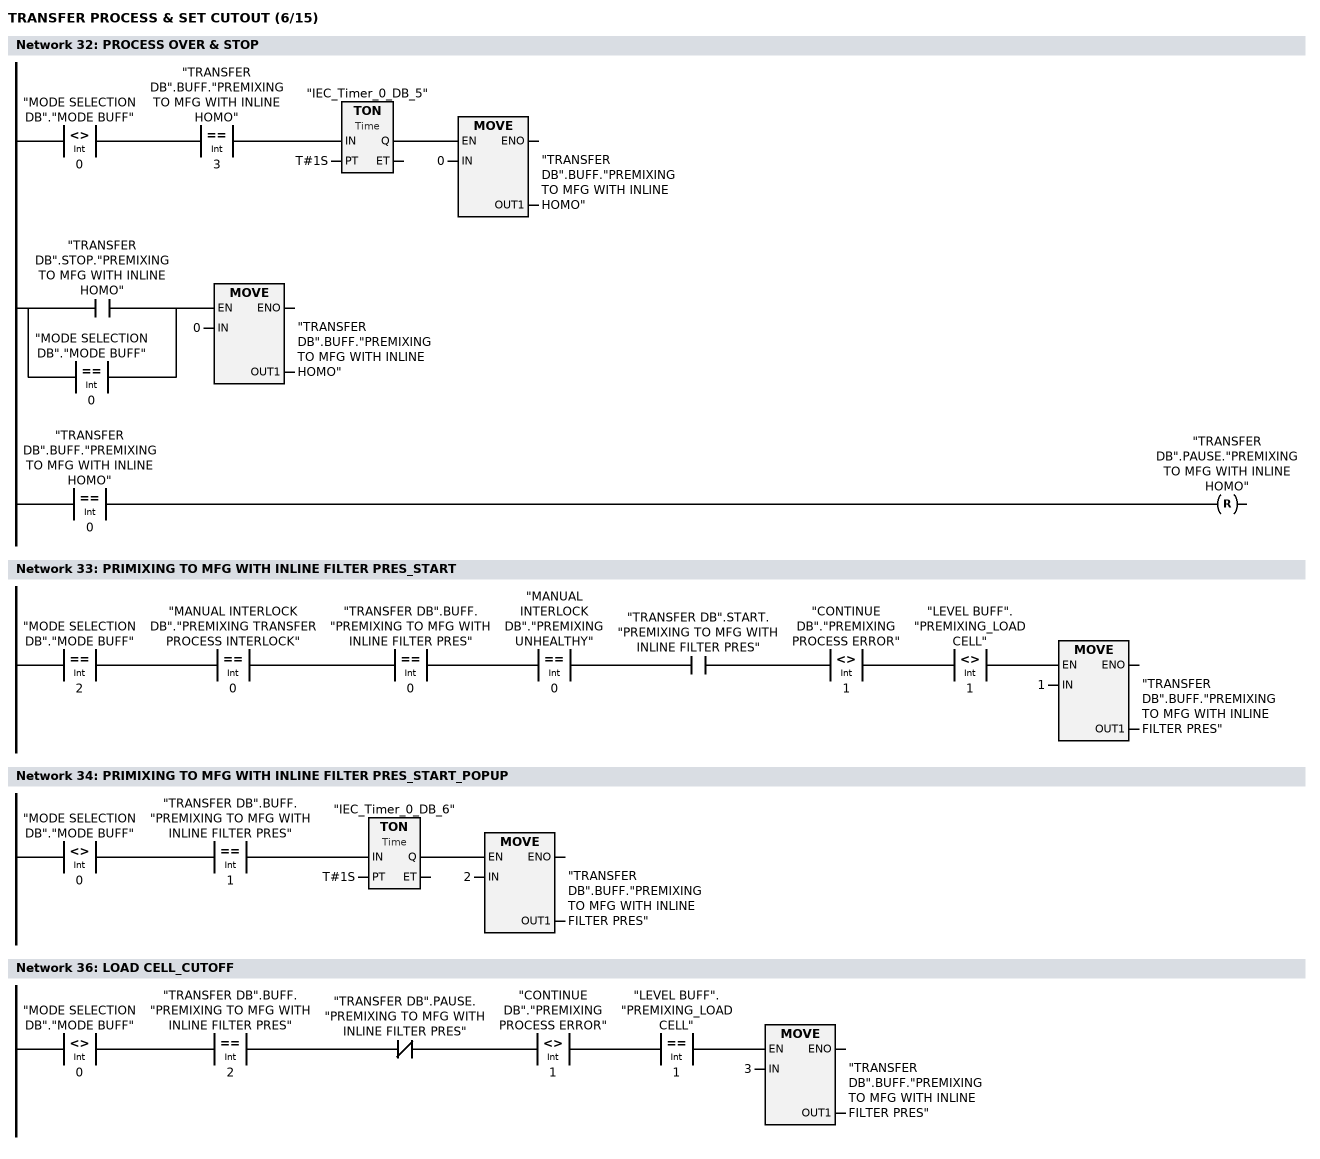
   RUNG wire#powerrail
      { S7_Templates := "SrcType := Int" } NE_Contact(in1 := "MODE SELECTION DB"."MODE BUFF", in2 := 0)
      { S7_Templates := "SrcType := Int" } EQ_Contact(in1 := "TRANSFER DB".BUFF."PREMIXING TO MFG WITH INLINE HOMO", in2 := 3)
      { S7_Templates := "time_type := Time" } "IEC_Timer_0_DB_5".TON(pt := T#1S, et =>)
      Move(in := 0, out1 => "TRANSFER DB".BUFF."PREMIXING TO MFG WITH INLINE HOMO")
   END_RUNG
   RUNG wire#powerrail
      Contact( "TRANSFER DB".STOP."PREMIXING TO MFG WITH INLINE HOMO" )
      wire#w1
      Move(in := 0, out1 => "TRANSFER DB".BUFF."PREMIXING TO MFG WITH INLINE HOMO")
   END_RUNG
   RUNG wire#powerrail
      { S7_Templates := "SrcType := Int" } EQ_Contact(in1 := "MODE SELECTION DB"."MODE BUFF", in2 := 0)
   END_RUNG wire#w1
   RUNG wire#powerrail
      { S7_Templates := "SrcType := Int" } EQ_Contact(in1 := "TRANSFER DB".BUFF."PREMIXING TO MFG WITH INLINE HOMO", in2 := 0)
      R_Coil( "TRANSFER DB".PAUSE."PREMIXING TO MFG WITH INLINE HOMO" )
   END_RUNG
   // the same network as SCL:
   "IEC_Timer_0_DB_5".TON(IN := ("MODE SELECTION DB"."MODE BUFF" <> 0) AND ("TRANSFER DB".BUFF."PREMIXING TO MFG WITH INLINE HOMO" = 3),
                          PT := T#1S);
   IF "IEC_Timer_0_DB_5".Q THEN "TRANSFER DB".BUFF."PREMIXING TO MFG WITH INLINE HOMO" := 0; END_IF;
   IF "TRANSFER DB".STOP."PREMIXING TO MFG WITH INLINE HOMO" OR ("MODE SELECTION DB"."MODE BUFF" = 0) THEN
       "TRANSFER DB".BUFF."PREMIXING TO MFG WITH INLINE HOMO" := 0;
   END_IF;
   IF "TRANSFER DB".BUFF."PREMIXING TO MFG WITH INLINE HOMO" = 0 THEN
       "TRANSFER DB".PAUSE."PREMIXING TO MFG WITH INLINE HOMO" := FALSE;
   END_IF;
END_REGION

REGION Network 33: PRIMIXING TO MFG WITH INLINE FILTER PRES_START
   RUNG wire#powerrail
      { S7_Templates := "SrcType := Int" } EQ_Contact(in1 := "MODE SELECTION DB"."MODE BUFF", in2 := 2)
      { S7_Templates := "SrcType := Int" } EQ_Contact(in1 := "MANUAL INTERLOCK DB"."PREMIXING TRANSFER PROCESS INTERLOCK", in2 := 0)
      { S7_Templates := "SrcType := Int" } EQ_Contact(in1 := "TRANSFER DB".BUFF."PREMIXING TO MFG WITH INLINE FILTER PRES", in2 := 0)
      { S7_Templates := "SrcType := Int" } EQ_Contact(in1 := "MANUAL INTERLOCK DB"."PREMIXING UNHEALTHY", in2 := 0)
      Contact( "TRANSFER DB".START."PREMIXING TO MFG WITH INLINE FILTER PRES" )
      { S7_Templates := "SrcType := Int" } NE_Contact(in1 := "CONTINUE DB"."PREMIXING PROCESS ERROR", in2 := 1)
      { S7_Templates := "SrcType := Int" } NE_Contact(in1 := "LEVEL BUFF"."PREMIXING_LOAD CELL", in2 := 1)
      Move(in := 1, out1 => "TRANSFER DB".BUFF."PREMIXING TO MFG WITH INLINE FILTER PRES")
   END_RUNG
   // the same network as SCL:
   IF ("MODE SELECTION DB"."MODE BUFF" = 2) AND ("MANUAL INTERLOCK DB"."PREMIXING TRANSFER PROCESS INTERLOCK" = 0) AND ("TRANSFER DB".BUFF."PREMIXING TO MFG WITH INLINE FILTER PRES" = 0) AND ("MANUAL INTERLOCK DB"."PREMIXING UNHEALTHY" = 0) AND "TRANSFER DB".START."PREMIXING TO MFG WITH INLINE FILTER PRES" AND ("CONTINUE DB"."PREMIXING PROCESS ERROR" <> 1) AND ("LEVEL BUFF"."PREMIXING_LOAD CELL" <> 1) THEN
       "TRANSFER DB".BUFF."PREMIXING TO MFG WITH INLINE FILTER PRES" := 1;
   END_IF;
END_REGION

REGION Network 34: PRIMIXING TO MFG WITH INLINE FILTER PRES_START_POPUP
   RUNG wire#powerrail
      { S7_Templates := "SrcType := Int" } NE_Contact(in1 := "MODE SELECTION DB"."MODE BUFF", in2 := 0)
      { S7_Templates := "SrcType := Int" } EQ_Contact(in1 := "TRANSFER DB".BUFF."PREMIXING TO MFG WITH INLINE FILTER PRES", in2 := 1)
      { S7_Templates := "time_type := Time" } "IEC_Timer_0_DB_6".TON(pt := T#1S, et =>)
      Move(in := 2, out1 => "TRANSFER DB".BUFF."PREMIXING TO MFG WITH INLINE FILTER PRES")
   END_RUNG
   // the same network as SCL:
   "IEC_Timer_0_DB_6".TON(IN := ("MODE SELECTION DB"."MODE BUFF" <> 0) AND ("TRANSFER DB".BUFF."PREMIXING TO MFG WITH INLINE FILTER PRES" = 1),
                          PT := T#1S);
   IF "IEC_Timer_0_DB_6".Q THEN "TRANSFER DB".BUFF."PREMIXING TO MFG WITH INLINE FILTER PRES" := 2; END_IF;
END_REGION

REGION Network 35 (SCL): OPENVALVE
   IF "MODE SELECTION DB"."MODE BUFF" <> 0 AND "TRANSFER DB".BUFF."PREMIXING TO MFG WITH INLINE FILTER PRES" = 2
       AND NOT "TRANSFER DB".PAUSE."PREMIXING TO MFG WITH INLINE FILTER PRES" 
       AND "CONTINUE DB"."PREMIXING PROCESS ERROR" = 0 AND "LEVEL BUFF"."PREMIXING_LOAD CELL" = 0
       OR ("MODE SELECTION DB"."MODE BUFF"=1 AND "PREMIXING DB"."AUTO BUFF"=0
       AND "PREMIXING TRANSFER CYCLE DB".TRANSFER."TRANSFER BUFF"."PREMIXING TO MFG WITH INLINE FILTER PRES"=10 AND "CONTINUE DB"."PREMIXING PROCESS ERROR" <>1
       AND "PREMIXING TRANSFER CYCLE DB".TRANSFER.SELECT."SELECT BUFF"=2)
   THEN
       "TRANSFER DB".BIT."PREMIXING TO MFG WITH INLINE FILTER PRES"."PFBV-17 TANK OUTLET VALVE" := TRUE;
       "TRANSFER DB".BIT."PREMIXING TO MFG WITH INLINE FILTER PRES"."PBV-93 TANK OUTLET TO INLINE HOMOGENIZER LINE" := TRUE;
       "TRANSFER DB".BIT."PREMIXING TO MFG WITH INLINE FILTER PRES"."PBV-95 TANK OUTLET TO FILTER PRESS LINE" := TRUE;
       "TRANSFER DB".BIT."PREMIXING TO MFG WITH INLINE FILTER PRES"."FILTER PRESS MOTOR 2 RUN" := TRUE;
       "TRANSFER DB".BIT."PREMIXING TO MFG WITH INLINE FILTER PRES"."PBV-100 FILTER PRESS INLET" := TRUE;
       "TRANSFER DB".BIT."PREMIXING TO MFG WITH INLINE FILTER PRES"."PBV-97 FILTER PRESS OUTLET" := TRUE;
       "TRANSFER DB".BIT."PREMIXING TO MFG WITH INLINE FILTER PRES"."PBV-98 INLINE HOMOGENIZER TO FILTER PRESS OUTLET LINE" := TRUE;
       "TRANSFER DB".BIT."PREMIXING TO MFG WITH INLINE FILTER PRES"."PBV-91 PREMIX TO MFG TRANSFER LINE" := TRUE;
       "TRANSFER DB".BIT."PREMIXING TO MFG WITH INLINE FILTER PRES"."PBV-102 PREMIX TO MFG TRANSFER (TOP DISH)" := TRUE;

   ELSE
       "TRANSFER DB".BIT."PREMIXING TO MFG WITH INLINE FILTER PRES"."PFBV-17 TANK OUTLET VALVE" := FALSE;
       "TRANSFER DB".BIT."PREMIXING TO MFG WITH INLINE FILTER PRES"."PBV-93 TANK OUTLET TO INLINE HOMOGENIZER LINE" := FALSE;
       "TRANSFER DB".BIT."PREMIXING TO MFG WITH INLINE FILTER PRES"."PBV-95 TANK OUTLET TO FILTER PRESS LINE" := FALSE;
       "TRANSFER DB".BIT."PREMIXING TO MFG WITH INLINE FILTER PRES"."FILTER PRESS MOTOR 2 RUN" := FALSE;
       "TRANSFER DB".BIT."PREMIXING TO MFG WITH INLINE FILTER PRES"."PBV-100 FILTER PRESS INLET" := FALSE;
       "TRANSFER DB".BIT."PREMIXING TO MFG WITH INLINE FILTER PRES"."PBV-97 FILTER PRESS OUTLET" := FALSE;
       "TRANSFER DB".BIT."PREMIXING TO MFG WITH INLINE FILTER PRES"."PBV-98 INLINE HOMOGENIZER TO FILTER PRESS OUTLET LINE" := FALSE;
       "TRANSFER DB".BIT."PREMIXING TO MFG WITH INLINE FILTER PRES"."PBV-91 PREMIX TO MFG TRANSFER LINE" := FALSE;
       "TRANSFER DB".BIT."PREMIXING TO MFG WITH INLINE FILTER PRES"."PBV-102 PREMIX TO MFG TRANSFER (TOP DISH)" := FALSE;
       ;
   END_IF;
END_REGION

REGION Network 36: LOAD CELL_CUTOFF
   RUNG wire#powerrail
      { S7_Templates := "SrcType := Int" } NE_Contact(in1 := "MODE SELECTION DB"."MODE BUFF", in2 := 0)
      { S7_Templates := "SrcType := Int" } EQ_Contact(in1 := "TRANSFER DB".BUFF."PREMIXING TO MFG WITH INLINE FILTER PRES", in2 := 2)
      I_Contact( "TRANSFER DB".PAUSE."PREMIXING TO MFG WITH INLINE FILTER PRES" )
      { S7_Templates := "SrcType := Int" } NE_Contact(in1 := "CONTINUE DB"."PREMIXING PROCESS ERROR", in2 := 1)
      { S7_Templates := "SrcType := Int" } EQ_Contact(in1 := "LEVEL BUFF"."PREMIXING_LOAD CELL", in2 := 1)
      Move(in := 3, out1 => "TRANSFER DB".BUFF."PREMIXING TO MFG WITH INLINE FILTER PRES")
   END_RUNG
   // the same network as SCL:
   IF ("MODE SELECTION DB"."MODE BUFF" <> 0) AND ("TRANSFER DB".BUFF."PREMIXING TO MFG WITH INLINE FILTER PRES" = 2) AND NOT "TRANSFER DB".PAUSE."PREMIXING TO MFG WITH INLINE FILTER PRES" AND ("CONTINUE DB"."PREMIXING PROCESS ERROR" <> 1) AND ("LEVEL BUFF"."PREMIXING_LOAD CELL" = 1) THEN
       "TRANSFER DB".BUFF."PREMIXING TO MFG WITH INLINE FILTER PRES" := 3;
   END_IF;
END_REGION

REGION Network 37: PROCESS OVER & STOP
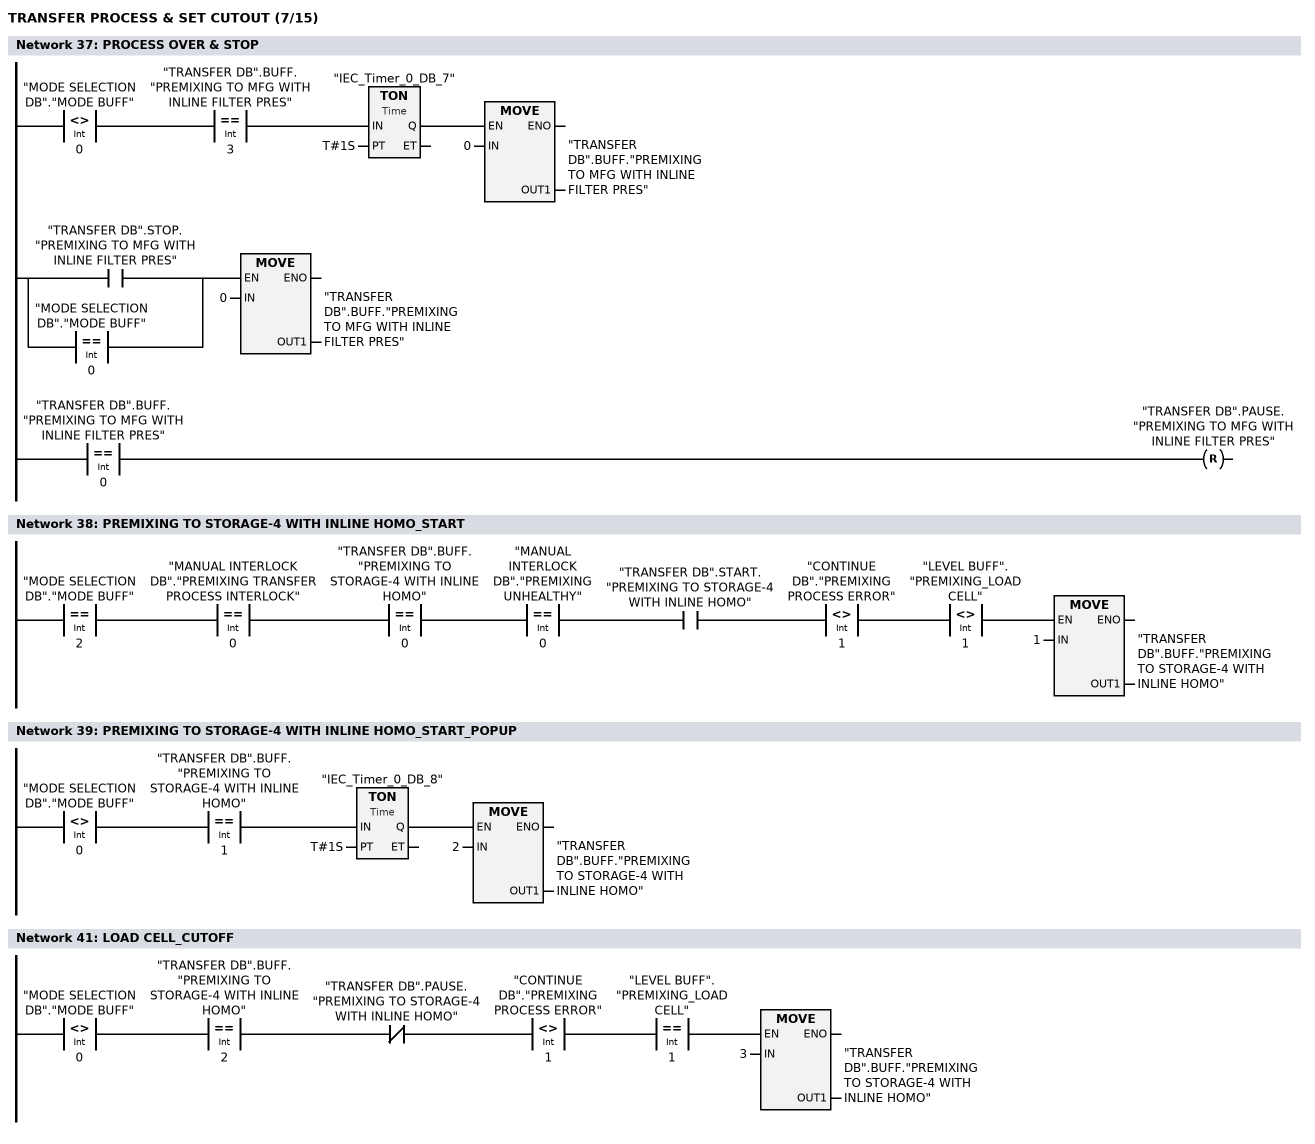
   RUNG wire#powerrail
      { S7_Templates := "SrcType := Int" } NE_Contact(in1 := "MODE SELECTION DB"."MODE BUFF", in2 := 0)
      { S7_Templates := "SrcType := Int" } EQ_Contact(in1 := "TRANSFER DB".BUFF."PREMIXING TO MFG WITH INLINE FILTER PRES", in2 := 3)
      { S7_Templates := "time_type := Time" } "IEC_Timer_0_DB_7".TON(pt := T#1S, et =>)
      Move(in := 0, out1 => "TRANSFER DB".BUFF."PREMIXING TO MFG WITH INLINE FILTER PRES")
   END_RUNG
   RUNG wire#powerrail
      Contact( "TRANSFER DB".STOP."PREMIXING TO MFG WITH INLINE FILTER PRES" )
      wire#w1
      Move(in := 0, out1 => "TRANSFER DB".BUFF."PREMIXING TO MFG WITH INLINE FILTER PRES")
   END_RUNG
   RUNG wire#powerrail
      { S7_Templates := "SrcType := Int" } EQ_Contact(in1 := "MODE SELECTION DB"."MODE BUFF", in2 := 0)
   END_RUNG wire#w1
   RUNG wire#powerrail
      { S7_Templates := "SrcType := Int" } EQ_Contact(in1 := "TRANSFER DB".BUFF."PREMIXING TO MFG WITH INLINE FILTER PRES", in2 := 0)
      R_Coil( "TRANSFER DB".PAUSE."PREMIXING TO MFG WITH INLINE FILTER PRES" )
   END_RUNG
   // the same network as SCL:
   "IEC_Timer_0_DB_7".TON(IN := ("MODE SELECTION DB"."MODE BUFF" <> 0) AND ("TRANSFER DB".BUFF."PREMIXING TO MFG WITH INLINE FILTER PRES" = 3),
                          PT := T#1S);
   IF "IEC_Timer_0_DB_7".Q THEN "TRANSFER DB".BUFF."PREMIXING TO MFG WITH INLINE FILTER PRES" := 0; END_IF;
   IF "TRANSFER DB".STOP."PREMIXING TO MFG WITH INLINE FILTER PRES" OR ("MODE SELECTION DB"."MODE BUFF" = 0) THEN
       "TRANSFER DB".BUFF."PREMIXING TO MFG WITH INLINE FILTER PRES" := 0;
   END_IF;
   IF "TRANSFER DB".BUFF."PREMIXING TO MFG WITH INLINE FILTER PRES" = 0 THEN
       "TRANSFER DB".PAUSE."PREMIXING TO MFG WITH INLINE FILTER PRES" := FALSE;
   END_IF;
END_REGION

REGION Network 38: PREMIXING TO STORAGE-4 WITH INLINE HOMO_START
   RUNG wire#powerrail
      { S7_Templates := "SrcType := Int" } EQ_Contact(in1 := "MODE SELECTION DB"."MODE BUFF", in2 := 2)
      { S7_Templates := "SrcType := Int" } EQ_Contact(in1 := "MANUAL INTERLOCK DB"."PREMIXING TRANSFER PROCESS INTERLOCK", in2 := 0)
      { S7_Templates := "SrcType := Int" } EQ_Contact(in1 := "TRANSFER DB".BUFF."PREMIXING TO STORAGE-4 WITH INLINE HOMO", in2 := 0)
      { S7_Templates := "SrcType := Int" } EQ_Contact(in1 := "MANUAL INTERLOCK DB"."PREMIXING UNHEALTHY", in2 := 0)
      Contact( "TRANSFER DB".START."PREMIXING TO STORAGE-4 WITH INLINE HOMO" )
      { S7_Templates := "SrcType := Int" } NE_Contact(in1 := "CONTINUE DB"."PREMIXING PROCESS ERROR", in2 := 1)
      { S7_Templates := "SrcType := Int" } NE_Contact(in1 := "LEVEL BUFF"."PREMIXING_LOAD CELL", in2 := 1)
      Move(in := 1, out1 => "TRANSFER DB".BUFF."PREMIXING TO STORAGE-4 WITH INLINE HOMO")
   END_RUNG
   // the same network as SCL:
   IF ("MODE SELECTION DB"."MODE BUFF" = 2) AND ("MANUAL INTERLOCK DB"."PREMIXING TRANSFER PROCESS INTERLOCK" = 0) AND ("TRANSFER DB".BUFF."PREMIXING TO STORAGE-4 WITH INLINE HOMO" = 0) AND ("MANUAL INTERLOCK DB"."PREMIXING UNHEALTHY" = 0) AND "TRANSFER DB".START."PREMIXING TO STORAGE-4 WITH INLINE HOMO" AND ("CONTINUE DB"."PREMIXING PROCESS ERROR" <> 1) AND ("LEVEL BUFF"."PREMIXING_LOAD CELL" <> 1) THEN
       "TRANSFER DB".BUFF."PREMIXING TO STORAGE-4 WITH INLINE HOMO" := 1;
   END_IF;
END_REGION

REGION Network 39: PREMIXING TO STORAGE-4 WITH INLINE HOMO_START_POPUP
   RUNG wire#powerrail
      { S7_Templates := "SrcType := Int" } NE_Contact(in1 := "MODE SELECTION DB"."MODE BUFF", in2 := 0)
      { S7_Templates := "SrcType := Int" } EQ_Contact(in1 := "TRANSFER DB".BUFF."PREMIXING TO STORAGE-4 WITH INLINE HOMO", in2 := 1)
      { S7_Templates := "time_type := Time" } "IEC_Timer_0_DB_8".TON(pt := T#1S, et =>)
      Move(in := 2, out1 => "TRANSFER DB".BUFF."PREMIXING TO STORAGE-4 WITH INLINE HOMO")
   END_RUNG
   // the same network as SCL:
   "IEC_Timer_0_DB_8".TON(IN := ("MODE SELECTION DB"."MODE BUFF" <> 0) AND ("TRANSFER DB".BUFF."PREMIXING TO STORAGE-4 WITH INLINE HOMO" = 1),
                          PT := T#1S);
   IF "IEC_Timer_0_DB_8".Q THEN "TRANSFER DB".BUFF."PREMIXING TO STORAGE-4 WITH INLINE HOMO" := 2; END_IF;
END_REGION

REGION Network 40 (SCL): OPENVALVE
   IF "MODE SELECTION DB"."MODE BUFF" <> 0 AND "TRANSFER DB".BUFF."PREMIXING TO STORAGE-4 WITH INLINE HOMO" = 2
       AND NOT "TRANSFER DB".PAUSE."PREMIXING TO STORAGE-4 WITH INLINE HOMO"
       AND "CONTINUE DB"."PREMIXING PROCESS ERROR" = 0 AND "LEVEL BUFF"."PREMIXING_LOAD CELL" = 0
       OR ("MODE SELECTION DB"."MODE BUFF"=1 AND "PREMIXING DB"."AUTO BUFF"=0
       AND "PREMIXING TRANSFER CYCLE DB".TRANSFER."TRANSFER BUFF"."PREMIXING TO STORAGE-4 WITH INLINE HOMO"=10 AND "CONTINUE DB"."PREMIXING PROCESS ERROR" <>1
       AND "PREMIXING TRANSFER CYCLE DB".TRANSFER.SELECT."SELECT BUFF"=3)
   THEN
       "TRANSFER DB".BIT."PREMIXING TO STORAGE-4 WITH INLINE HOMO"."PFBV-17 TANK OUTLET VALVE" := TRUE;
       "TRANSFER DB".BIT."PREMIXING TO STORAGE-4 WITH INLINE HOMO"."PBV-93 TANK OUTLET TO INLINE HOMOGENIZER LINE" := TRUE;
       "TRANSFER DB".BIT."PREMIXING TO STORAGE-4 WITH INLINE HOMO"."PBV-94 INLINE HOMOGENIZER INLET LINE" := TRUE;
       "TRANSFER DB".BIT."PREMIXING TO STORAGE-4 WITH INLINE HOMO"."PAV-99 INLINE HOMOGENIZER SEAL COOLING" := TRUE;
       "TRANSFER DB".BIT."PREMIXING TO STORAGE-4 WITH INLINE HOMO"."INLINE 2 HOMOGENIZER MOTOR 2 RUN" := TRUE;
       "TRANSFER DB".BIT."PREMIXING TO STORAGE-4 WITH INLINE HOMO"."PBV-96 INLINE HOMOGENIZER RECIRCULATION LINE" := TRUE;
       "TRANSFER DB".BIT."PREMIXING TO STORAGE-4 WITH INLINE HOMO"."PBV-92 PREMIX TO STORAGE – 4 TRANSFER LINE" := TRUE;

   ELSE
       "TRANSFER DB".BIT."PREMIXING TO STORAGE-4 WITH INLINE HOMO"."PFBV-17 TANK OUTLET VALVE" := FALSE;
       "TRANSFER DB".BIT."PREMIXING TO STORAGE-4 WITH INLINE HOMO"."PBV-93 TANK OUTLET TO INLINE HOMOGENIZER LINE" := FALSE;
       "TRANSFER DB".BIT."PREMIXING TO STORAGE-4 WITH INLINE HOMO"."PBV-94 INLINE HOMOGENIZER INLET LINE" := FALSE;
       "TRANSFER DB".BIT."PREMIXING TO STORAGE-4 WITH INLINE HOMO"."PAV-99 INLINE HOMOGENIZER SEAL COOLING" := FALSE;
       "TRANSFER DB".BIT."PREMIXING TO STORAGE-4 WITH INLINE HOMO"."INLINE 2 HOMOGENIZER MOTOR 2 RUN" := FALSE;
       "TRANSFER DB".BIT."PREMIXING TO STORAGE-4 WITH INLINE HOMO"."PBV-96 INLINE HOMOGENIZER RECIRCULATION LINE" := FALSE;
       "TRANSFER DB".BIT."PREMIXING TO STORAGE-4 WITH INLINE HOMO"."PBV-92 PREMIX TO STORAGE – 4 TRANSFER LINE" := FALSE;
       ;
   END_IF;
END_REGION

REGION Network 41: LOAD CELL_CUTOFF
   RUNG wire#powerrail
      { S7_Templates := "SrcType := Int" } NE_Contact(in1 := "MODE SELECTION DB"."MODE BUFF", in2 := 0)
      { S7_Templates := "SrcType := Int" } EQ_Contact(in1 := "TRANSFER DB".BUFF."PREMIXING TO STORAGE-4 WITH INLINE HOMO", in2 := 2)
      I_Contact( "TRANSFER DB".PAUSE."PREMIXING TO STORAGE-4 WITH INLINE HOMO" )
      { S7_Templates := "SrcType := Int" } NE_Contact(in1 := "CONTINUE DB"."PREMIXING PROCESS ERROR", in2 := 1)
      { S7_Templates := "SrcType := Int" } EQ_Contact(in1 := "LEVEL BUFF"."PREMIXING_LOAD CELL", in2 := 1)
      Move(in := 3, out1 => "TRANSFER DB".BUFF."PREMIXING TO STORAGE-4 WITH INLINE HOMO")
   END_RUNG
   // the same network as SCL:
   IF ("MODE SELECTION DB"."MODE BUFF" <> 0) AND ("TRANSFER DB".BUFF."PREMIXING TO STORAGE-4 WITH INLINE HOMO" = 2) AND NOT "TRANSFER DB".PAUSE."PREMIXING TO STORAGE-4 WITH INLINE HOMO" AND ("CONTINUE DB"."PREMIXING PROCESS ERROR" <> 1) AND ("LEVEL BUFF"."PREMIXING_LOAD CELL" = 1) THEN
       "TRANSFER DB".BUFF."PREMIXING TO STORAGE-4 WITH INLINE HOMO" := 3;
   END_IF;
END_REGION

REGION Network 42: PROCESS OVER & STOP
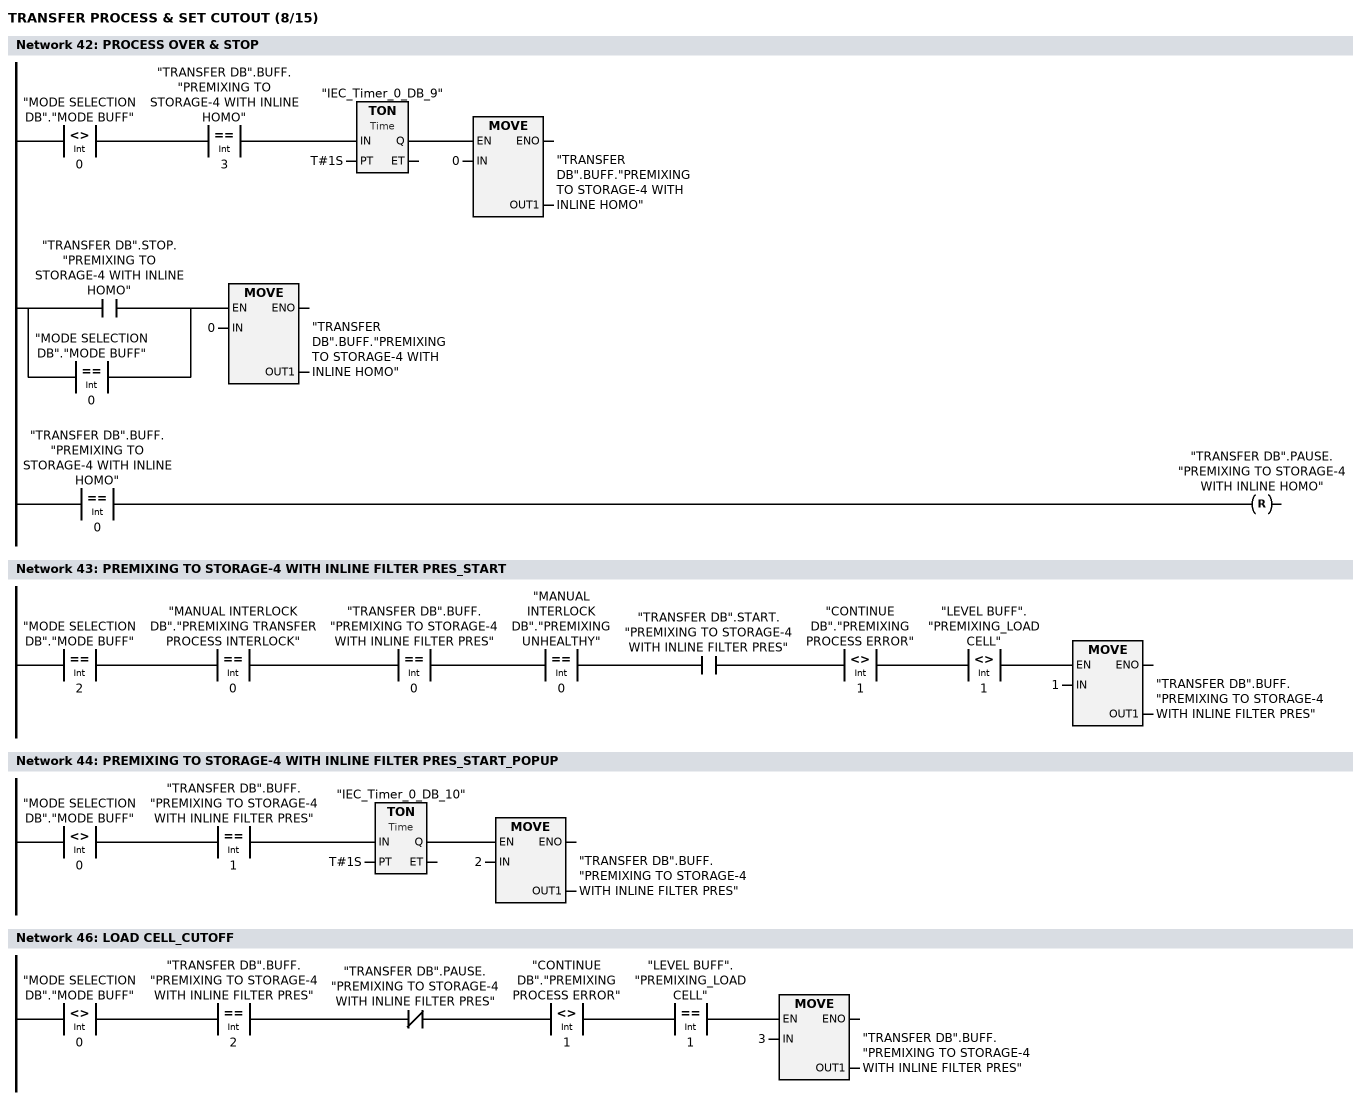
   RUNG wire#powerrail
      { S7_Templates := "SrcType := Int" } NE_Contact(in1 := "MODE SELECTION DB"."MODE BUFF", in2 := 0)
      { S7_Templates := "SrcType := Int" } EQ_Contact(in1 := "TRANSFER DB".BUFF."PREMIXING TO STORAGE-4 WITH INLINE HOMO", in2 := 3)
      { S7_Templates := "time_type := Time" } "IEC_Timer_0_DB_9".TON(pt := T#1S, et =>)
      Move(in := 0, out1 => "TRANSFER DB".BUFF."PREMIXING TO STORAGE-4 WITH INLINE HOMO")
   END_RUNG
   RUNG wire#powerrail
      Contact( "TRANSFER DB".STOP."PREMIXING TO STORAGE-4 WITH INLINE HOMO" )
      wire#w1
      Move(in := 0, out1 => "TRANSFER DB".BUFF."PREMIXING TO STORAGE-4 WITH INLINE HOMO")
   END_RUNG
   RUNG wire#powerrail
      { S7_Templates := "SrcType := Int" } EQ_Contact(in1 := "MODE SELECTION DB"."MODE BUFF", in2 := 0)
   END_RUNG wire#w1
   RUNG wire#powerrail
      { S7_Templates := "SrcType := Int" } EQ_Contact(in1 := "TRANSFER DB".BUFF."PREMIXING TO STORAGE-4 WITH INLINE HOMO", in2 := 0)
      R_Coil( "TRANSFER DB".PAUSE."PREMIXING TO STORAGE-4 WITH INLINE HOMO" )
   END_RUNG
   // the same network as SCL:
   "IEC_Timer_0_DB_9".TON(IN := ("MODE SELECTION DB"."MODE BUFF" <> 0) AND ("TRANSFER DB".BUFF."PREMIXING TO STORAGE-4 WITH INLINE HOMO" = 3),
                          PT := T#1S);
   IF "IEC_Timer_0_DB_9".Q THEN "TRANSFER DB".BUFF."PREMIXING TO STORAGE-4 WITH INLINE HOMO" := 0; END_IF;
   IF "TRANSFER DB".STOP."PREMIXING TO STORAGE-4 WITH INLINE HOMO" OR ("MODE SELECTION DB"."MODE BUFF" = 0) THEN
       "TRANSFER DB".BUFF."PREMIXING TO STORAGE-4 WITH INLINE HOMO" := 0;
   END_IF;
   IF "TRANSFER DB".BUFF."PREMIXING TO STORAGE-4 WITH INLINE HOMO" = 0 THEN
       "TRANSFER DB".PAUSE."PREMIXING TO STORAGE-4 WITH INLINE HOMO" := FALSE;
   END_IF;
END_REGION

REGION Network 43: PREMIXING TO STORAGE-4 WITH INLINE FILTER PRES_START
   RUNG wire#powerrail
      { S7_Templates := "SrcType := Int" } EQ_Contact(in1 := "MODE SELECTION DB"."MODE BUFF", in2 := 2)
      { S7_Templates := "SrcType := Int" } EQ_Contact(in1 := "MANUAL INTERLOCK DB"."PREMIXING TRANSFER PROCESS INTERLOCK", in2 := 0)
      { S7_Templates := "SrcType := Int" } EQ_Contact(in1 := "TRANSFER DB".BUFF."PREMIXING TO STORAGE-4 WITH INLINE FILTER PRES", in2 := 0)
      { S7_Templates := "SrcType := Int" } EQ_Contact(in1 := "MANUAL INTERLOCK DB"."PREMIXING UNHEALTHY", in2 := 0)
      Contact( "TRANSFER DB".START."PREMIXING TO STORAGE-4 WITH INLINE FILTER PRES" )
      { S7_Templates := "SrcType := Int" } NE_Contact(in1 := "CONTINUE DB"."PREMIXING PROCESS ERROR", in2 := 1)
      { S7_Templates := "SrcType := Int" } NE_Contact(in1 := "LEVEL BUFF"."PREMIXING_LOAD CELL", in2 := 1)
      Move(in := 1, out1 => "TRANSFER DB".BUFF."PREMIXING TO STORAGE-4 WITH INLINE FILTER PRES")
   END_RUNG
   // the same network as SCL:
   IF ("MODE SELECTION DB"."MODE BUFF" = 2) AND ("MANUAL INTERLOCK DB"."PREMIXING TRANSFER PROCESS INTERLOCK" = 0) AND ("TRANSFER DB".BUFF."PREMIXING TO STORAGE-4 WITH INLINE FILTER PRES" = 0) AND ("MANUAL INTERLOCK DB"."PREMIXING UNHEALTHY" = 0) AND "TRANSFER DB".START."PREMIXING TO STORAGE-4 WITH INLINE FILTER PRES" AND ("CONTINUE DB"."PREMIXING PROCESS ERROR" <> 1) AND ("LEVEL BUFF"."PREMIXING_LOAD CELL" <> 1) THEN
       "TRANSFER DB".BUFF."PREMIXING TO STORAGE-4 WITH INLINE FILTER PRES" := 1;
   END_IF;
END_REGION

REGION Network 44: PREMIXING TO STORAGE-4 WITH INLINE FILTER PRES_START_POPUP
   RUNG wire#powerrail
      { S7_Templates := "SrcType := Int" } NE_Contact(in1 := "MODE SELECTION DB"."MODE BUFF", in2 := 0)
      { S7_Templates := "SrcType := Int" } EQ_Contact(in1 := "TRANSFER DB".BUFF."PREMIXING TO STORAGE-4 WITH INLINE FILTER PRES", in2 := 1)
      { S7_Templates := "time_type := Time" } "IEC_Timer_0_DB_10".TON(pt := T#1S, et =>)
      Move(in := 2, out1 => "TRANSFER DB".BUFF."PREMIXING TO STORAGE-4 WITH INLINE FILTER PRES")
   END_RUNG
   // the same network as SCL:
   "IEC_Timer_0_DB_10".TON(IN := ("MODE SELECTION DB"."MODE BUFF" <> 0) AND ("TRANSFER DB".BUFF."PREMIXING TO STORAGE-4 WITH INLINE FILTER PRES" = 1),
                           PT := T#1S);
   IF "IEC_Timer_0_DB_10".Q THEN
       "TRANSFER DB".BUFF."PREMIXING TO STORAGE-4 WITH INLINE FILTER PRES" := 2;
   END_IF;
END_REGION

REGION Network 45 (SCL): OPENVALVE
   IF "MODE SELECTION DB"."MODE BUFF" <> 0 AND "TRANSFER DB".BUFF."PREMIXING TO STORAGE-4 WITH INLINE FILTER PRES" = 2
       AND NOT "TRANSFER DB".PAUSE."PREMIXING TO STORAGE-4 WITH INLINE FILTER PRES" 
       AND "CONTINUE DB"."PREMIXING PROCESS ERROR" = 0 AND "LEVEL BUFF"."PREMIXING_LOAD CELL" = 0
       OR ("MODE SELECTION DB"."MODE BUFF"=1 AND "PREMIXING DB"."AUTO BUFF"=0
       AND "PREMIXING TRANSFER CYCLE DB".TRANSFER."TRANSFER BUFF"."PREMIXING TO STORAGE-4 WITH INLINE FILTER PRES"=10 AND "CONTINUE DB"."PREMIXING PROCESS ERROR" <>1
       AND "PREMIXING TRANSFER CYCLE DB".TRANSFER.SELECT."SELECT BUFF"=4)
   THEN
       "TRANSFER DB".BIT."PREMIXING TO STORAGE-4 WITH INLINE FILTER PRES"."PFBV-17 TANK OUTLET VALVE" := TRUE;
       "TRANSFER DB".BIT."PREMIXING TO STORAGE-4 WITH INLINE FILTER PRES"."PBV-93 TANK OUTLET TO INLINE HOMOGENIZER LINE" := TRUE;
       "TRANSFER DB".BIT."PREMIXING TO STORAGE-4 WITH INLINE FILTER PRES"."PBV-95 TANK OUTLET TO FILTER PRESS LINE" := TRUE;
       "TRANSFER DB".BIT."PREMIXING TO STORAGE-4 WITH INLINE FILTER PRES"."FILTER PRESS MOTOR 2 RUN" := TRUE;
       "TRANSFER DB".BIT."PREMIXING TO STORAGE-4 WITH INLINE FILTER PRES"."PBV-100 FILTER PRESS INLET" := TRUE;
       "TRANSFER DB".BIT."PREMIXING TO STORAGE-4 WITH INLINE FILTER PRES"."PBV-97 FILTER PRESS OUTLET" := TRUE;
       "TRANSFER DB".BIT."PREMIXING TO STORAGE-4 WITH INLINE FILTER PRES"."PBV-98 INLINE HOMOGENIZER TO FILTER PRESS OUTLET LINE" := TRUE;
       "TRANSFER DB".BIT."PREMIXING TO STORAGE-4 WITH INLINE FILTER PRES"."PBV-92 PREMIX TO STORAGE – 4 TRANSFER LINE" := TRUE;

   ELSE
       "TRANSFER DB".BIT."PREMIXING TO STORAGE-4 WITH INLINE FILTER PRES"."PFBV-17 TANK OUTLET VALVE" := FALSE;
       "TRANSFER DB".BIT."PREMIXING TO STORAGE-4 WITH INLINE FILTER PRES"."PBV-93 TANK OUTLET TO INLINE HOMOGENIZER LINE" := FALSE;
       "TRANSFER DB".BIT."PREMIXING TO STORAGE-4 WITH INLINE FILTER PRES"."PBV-95 TANK OUTLET TO FILTER PRESS LINE" := FALSE;
       "TRANSFER DB".BIT."PREMIXING TO STORAGE-4 WITH INLINE FILTER PRES"."FILTER PRESS MOTOR 2 RUN" := FALSE;
       "TRANSFER DB".BIT."PREMIXING TO STORAGE-4 WITH INLINE FILTER PRES"."PBV-100 FILTER PRESS INLET" := FALSE;
       "TRANSFER DB".BIT."PREMIXING TO STORAGE-4 WITH INLINE FILTER PRES"."PBV-97 FILTER PRESS OUTLET" := FALSE;
       "TRANSFER DB".BIT."PREMIXING TO STORAGE-4 WITH INLINE FILTER PRES"."PBV-98 INLINE HOMOGENIZER TO FILTER PRESS OUTLET LINE" := FALSE;
       "TRANSFER DB".BIT."PREMIXING TO STORAGE-4 WITH INLINE FILTER PRES"."PBV-92 PREMIX TO STORAGE – 4 TRANSFER LINE" := FALSE;
       ;
   END_IF;
END_REGION

REGION Network 46: LOAD CELL_CUTOFF
   RUNG wire#powerrail
      { S7_Templates := "SrcType := Int" } NE_Contact(in1 := "MODE SELECTION DB"."MODE BUFF", in2 := 0)
      { S7_Templates := "SrcType := Int" } EQ_Contact(in1 := "TRANSFER DB".BUFF."PREMIXING TO STORAGE-4 WITH INLINE FILTER PRES", in2 := 2)
      I_Contact( "TRANSFER DB".PAUSE."PREMIXING TO STORAGE-4 WITH INLINE FILTER PRES" )
      { S7_Templates := "SrcType := Int" } NE_Contact(in1 := "CONTINUE DB"."PREMIXING PROCESS ERROR", in2 := 1)
      { S7_Templates := "SrcType := Int" } EQ_Contact(in1 := "LEVEL BUFF"."PREMIXING_LOAD CELL", in2 := 1)
      Move(in := 3, out1 => "TRANSFER DB".BUFF."PREMIXING TO STORAGE-4 WITH INLINE FILTER PRES")
   END_RUNG
   // the same network as SCL:
   IF ("MODE SELECTION DB"."MODE BUFF" <> 0) AND ("TRANSFER DB".BUFF."PREMIXING TO STORAGE-4 WITH INLINE FILTER PRES" = 2) AND NOT "TRANSFER DB".PAUSE."PREMIXING TO STORAGE-4 WITH INLINE FILTER PRES" AND ("CONTINUE DB"."PREMIXING PROCESS ERROR" <> 1) AND ("LEVEL BUFF"."PREMIXING_LOAD CELL" = 1) THEN
       "TRANSFER DB".BUFF."PREMIXING TO STORAGE-4 WITH INLINE FILTER PRES" := 3;
   END_IF;
END_REGION

REGION Network 47: PROCESS OVER & STOP
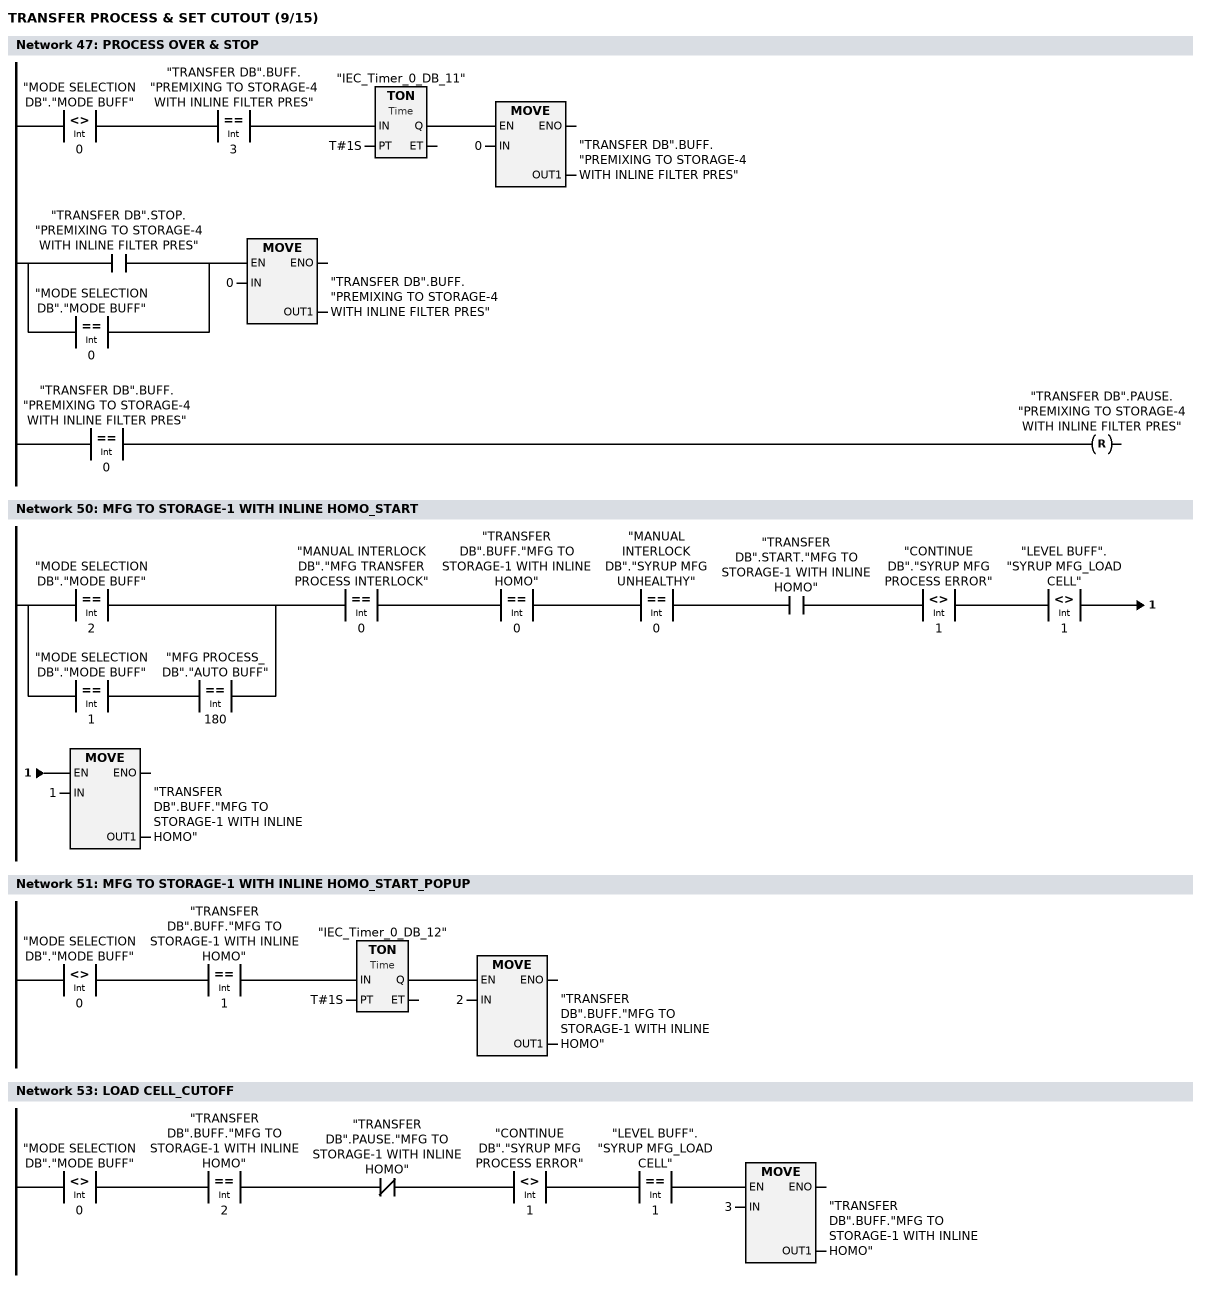
   RUNG wire#powerrail
      { S7_Templates := "SrcType := Int" } NE_Contact(in1 := "MODE SELECTION DB"."MODE BUFF", in2 := 0)
      { S7_Templates := "SrcType := Int" } EQ_Contact(in1 := "TRANSFER DB".BUFF."PREMIXING TO STORAGE-4 WITH INLINE FILTER PRES", in2 := 3)
      { S7_Templates := "time_type := Time" } "IEC_Timer_0_DB_11".TON(pt := T#1S, et =>)
      Move(in := 0, out1 => "TRANSFER DB".BUFF."PREMIXING TO STORAGE-4 WITH INLINE FILTER PRES")
   END_RUNG
   RUNG wire#powerrail
      Contact( "TRANSFER DB".STOP."PREMIXING TO STORAGE-4 WITH INLINE FILTER PRES" )
      wire#w1
      Move(in := 0, out1 => "TRANSFER DB".BUFF."PREMIXING TO STORAGE-4 WITH INLINE FILTER PRES")
   END_RUNG
   RUNG wire#powerrail
      { S7_Templates := "SrcType := Int" } EQ_Contact(in1 := "MODE SELECTION DB"."MODE BUFF", in2 := 0)
   END_RUNG wire#w1
   RUNG wire#powerrail
      { S7_Templates := "SrcType := Int" } EQ_Contact(in1 := "TRANSFER DB".BUFF."PREMIXING TO STORAGE-4 WITH INLINE FILTER PRES", in2 := 0)
      R_Coil( "TRANSFER DB".PAUSE."PREMIXING TO STORAGE-4 WITH INLINE FILTER PRES" )
   END_RUNG
   // the same network as SCL:
   "IEC_Timer_0_DB_11".TON(IN := ("MODE SELECTION DB"."MODE BUFF" <> 0) AND ("TRANSFER DB".BUFF."PREMIXING TO STORAGE-4 WITH INLINE FILTER PRES" = 3),
                           PT := T#1S);
   IF "IEC_Timer_0_DB_11".Q THEN
       "TRANSFER DB".BUFF."PREMIXING TO STORAGE-4 WITH INLINE FILTER PRES" := 0;
   END_IF;
   IF "TRANSFER DB".STOP."PREMIXING TO STORAGE-4 WITH INLINE FILTER PRES" OR ("MODE SELECTION DB"."MODE BUFF" = 0) THEN
       "TRANSFER DB".BUFF."PREMIXING TO STORAGE-4 WITH INLINE FILTER PRES" := 0;
   END_IF;
   IF "TRANSFER DB".BUFF."PREMIXING TO STORAGE-4 WITH INLINE FILTER PRES" = 0 THEN
       "TRANSFER DB".PAUSE."PREMIXING TO STORAGE-4 WITH INLINE FILTER PRES" := FALSE;
   END_IF;
END_REGION

REGION Network 49: ////////////////////////////////////////////////////////////////////// TRANSFER PROCESS- MFG //////////////////////////////////////////////////////////////////////////////////
END_REGION

REGION Network 50: MFG TO STORAGE-1 WITH INLINE HOMO_START
   RUNG wire#powerrail
      { S7_Templates := "SrcType := Int" } EQ_Contact(in1 := "MODE SELECTION DB"."MODE BUFF", in2 := 2)
      wire#w1
      { S7_Templates := "SrcType := Int" } EQ_Contact(in1 := "MANUAL INTERLOCK DB"."MFG TRANSFER PROCESS INTERLOCK", in2 := 0)
      { S7_Templates := "SrcType := Int" } EQ_Contact(in1 := "TRANSFER DB".BUFF."MFG TO STORAGE-1 WITH INLINE HOMO", in2 := 0)
      { S7_Templates := "SrcType := Int" } EQ_Contact(in1 := "MANUAL INTERLOCK DB"."SYRUP MFG UNHEALTHY", in2 := 0)
      Contact( "TRANSFER DB".START."MFG TO STORAGE-1 WITH INLINE HOMO" )
      { S7_Templates := "SrcType := Int" } NE_Contact(in1 := "CONTINUE DB"."SYRUP MFG PROCESS ERROR", in2 := 1)
      { S7_Templates := "SrcType := Int" } NE_Contact(in1 := "LEVEL BUFF"."SYRUP MFG_LOAD CELL", in2 := 1)
      Move(in := 1, out1 => "TRANSFER DB".BUFF."MFG TO STORAGE-1 WITH INLINE HOMO")
   END_RUNG
   RUNG wire#powerrail
      { S7_Templates := "SrcType := Int" } EQ_Contact(in1 := "MODE SELECTION DB"."MODE BUFF", in2 := 1)
      { S7_Templates := "SrcType := Int" } EQ_Contact(in1 := "MFG PROCESS_DB"."AUTO BUFF", in2 := 180)
   END_RUNG wire#w1
   // the same network as SCL:
   IF (("MODE SELECTION DB"."MODE BUFF" = 2) OR (("MODE SELECTION DB"."MODE BUFF" = 1) AND ("MFG PROCESS_DB"."AUTO BUFF" = 180))) AND ("MANUAL INTERLOCK DB"."MFG TRANSFER PROCESS INTERLOCK" = 0) AND ("TRANSFER DB".BUFF."MFG TO STORAGE-1 WITH INLINE HOMO" = 0) AND ("MANUAL INTERLOCK DB"."SYRUP MFG UNHEALTHY" = 0) AND "TRANSFER DB".START."MFG TO STORAGE-1 WITH INLINE HOMO" AND ("CONTINUE DB"."SYRUP MFG PROCESS ERROR" <> 1) AND ("LEVEL BUFF"."SYRUP MFG_LOAD CELL" <> 1) THEN
       "TRANSFER DB".BUFF."MFG TO STORAGE-1 WITH INLINE HOMO" := 1;
   END_IF;
END_REGION

REGION Network 51: MFG TO STORAGE-1 WITH INLINE HOMO_START_POPUP
   RUNG wire#powerrail
      { S7_Templates := "SrcType := Int" } NE_Contact(in1 := "MODE SELECTION DB"."MODE BUFF", in2 := 0)
      { S7_Templates := "SrcType := Int" } EQ_Contact(in1 := "TRANSFER DB".BUFF."MFG TO STORAGE-1 WITH INLINE HOMO", in2 := 1)
      { S7_Templates := "time_type := Time" } "IEC_Timer_0_DB_12".TON(pt := T#1S, et =>)
      Move(in := 2, out1 => "TRANSFER DB".BUFF."MFG TO STORAGE-1 WITH INLINE HOMO")
   END_RUNG
   // the same network as SCL:
   "IEC_Timer_0_DB_12".TON(IN := ("MODE SELECTION DB"."MODE BUFF" <> 0) AND ("TRANSFER DB".BUFF."MFG TO STORAGE-1 WITH INLINE HOMO" = 1),
                           PT := T#1S);
   IF "IEC_Timer_0_DB_12".Q THEN "TRANSFER DB".BUFF."MFG TO STORAGE-1 WITH INLINE HOMO" := 2; END_IF;
END_REGION

REGION Network 52 (SCL): OPENVALVE
   IF ("MODE SELECTION DB"."MODE BUFF" <> 0 AND "TRANSFER DB".BUFF."MFG TO STORAGE-1 WITH INLINE HOMO" = 2
       AND NOT "TRANSFER DB".PAUSE."MFG TO STORAGE-1 WITH INLINE HOMO"
       AND "CONTINUE DB"."SYRUP MFG PROCESS ERROR" = 0 AND "LEVEL BUFF"."SYRUP MFG_LOAD CELL" = 0)
       OR ("MODE SELECTION DB"."MODE BUFF"=1 AND "MFG PROCESS_DB"."AUTO BUFF"=0
       AND "MFG TRANSFER CYCLE DB".TRANSFER."TRANSFER BUFF"."MFG TO STORAGE-1 WITH INLINE HOMO"=10 AND "CONTINUE DB"."SYRUP MFG PROCESS ERROR" <>1
       AND "MFG TRANSFER CYCLE DB".TRANSFER.SELECT."SELECT BUFF"=1)
   THEN
       "TRANSFER DB".BIT."MFG TO STORAGE-1 WITH INLINE HOMO"."PFBV-59 TANK OUTLET VALVE" := TRUE;
       "TRANSFER DB".BIT."MFG TO STORAGE-1 WITH INLINE HOMO"."PBV-114 TANK OUTLET TO INLINE HOMOGENIZER LINE" := TRUE;
       "TRANSFER DB".BIT."MFG TO STORAGE-1 WITH INLINE HOMO"."PBV-110 INLINE HOMOGENIZER TO INLET LINE" := TRUE;
       "TRANSFER DB".BIT."MFG TO STORAGE-1 WITH INLINE HOMO"."PAV-56 INLINE HOMO. SEAL COOLING INLET" := TRUE;
       "TRANSFER DB".BIT."MFG TO STORAGE-1 WITH INLINE HOMO"."INLINE 1 HOMOGENIZER MOTOR1 RUN" := TRUE;
       "TRANSFER DB".BIT."MFG TO STORAGE-1 WITH INLINE HOMO"."PBV-109 HOMO. RECIRCULATION INLET" := TRUE;
       "TRANSFER DB".BIT."MFG TO STORAGE-1 WITH INLINE HOMO"."PBV-115 MFG TO STORAGE – 1 TRANSFER LINE" := TRUE;
   ELSE
       "TRANSFER DB".BIT."MFG TO STORAGE-1 WITH INLINE HOMO"."PFBV-59 TANK OUTLET VALVE" := FALSE;
       "TRANSFER DB".BIT."MFG TO STORAGE-1 WITH INLINE HOMO"."PBV-114 TANK OUTLET TO INLINE HOMOGENIZER LINE" := FALSE;
       "TRANSFER DB".BIT."MFG TO STORAGE-1 WITH INLINE HOMO"."PBV-110 INLINE HOMOGENIZER TO INLET LINE" := FALSE;
       "TRANSFER DB".BIT."MFG TO STORAGE-1 WITH INLINE HOMO"."PAV-56 INLINE HOMO. SEAL COOLING INLET" := FALSE;
       "TRANSFER DB".BIT."MFG TO STORAGE-1 WITH INLINE HOMO"."INLINE 1 HOMOGENIZER MOTOR1 RUN" := FALSE;
       "TRANSFER DB".BIT."MFG TO STORAGE-1 WITH INLINE HOMO"."PBV-109 HOMO. RECIRCULATION INLET" := FALSE;
       "TRANSFER DB".BIT."MFG TO STORAGE-1 WITH INLINE HOMO"."PBV-115 MFG TO STORAGE – 1 TRANSFER LINE" := FALSE;
       ;
   END_IF;
END_REGION

REGION Network 53: LOAD CELL_CUTOFF
   RUNG wire#powerrail
      { S7_Templates := "SrcType := Int" } NE_Contact(in1 := "MODE SELECTION DB"."MODE BUFF", in2 := 0)
      { S7_Templates := "SrcType := Int" } EQ_Contact(in1 := "TRANSFER DB".BUFF."MFG TO STORAGE-1 WITH INLINE HOMO", in2 := 2)
      I_Contact( "TRANSFER DB".PAUSE."MFG TO STORAGE-1 WITH INLINE HOMO" )
      { S7_Templates := "SrcType := Int" } NE_Contact(in1 := "CONTINUE DB"."SYRUP MFG PROCESS ERROR", in2 := 1)
      { S7_Templates := "SrcType := Int" } EQ_Contact(in1 := "LEVEL BUFF"."SYRUP MFG_LOAD CELL", in2 := 1)
      Move(in := 3, out1 => "TRANSFER DB".BUFF."MFG TO STORAGE-1 WITH INLINE HOMO")
   END_RUNG
   // the same network as SCL:
   IF ("MODE SELECTION DB"."MODE BUFF" <> 0) AND ("TRANSFER DB".BUFF."MFG TO STORAGE-1 WITH INLINE HOMO" = 2) AND NOT "TRANSFER DB".PAUSE."MFG TO STORAGE-1 WITH INLINE HOMO" AND ("CONTINUE DB"."SYRUP MFG PROCESS ERROR" <> 1) AND ("LEVEL BUFF"."SYRUP MFG_LOAD CELL" = 1) THEN
       "TRANSFER DB".BUFF."MFG TO STORAGE-1 WITH INLINE HOMO" := 3;
   END_IF;
END_REGION

REGION Network 54: PROCESS OVER & STOP
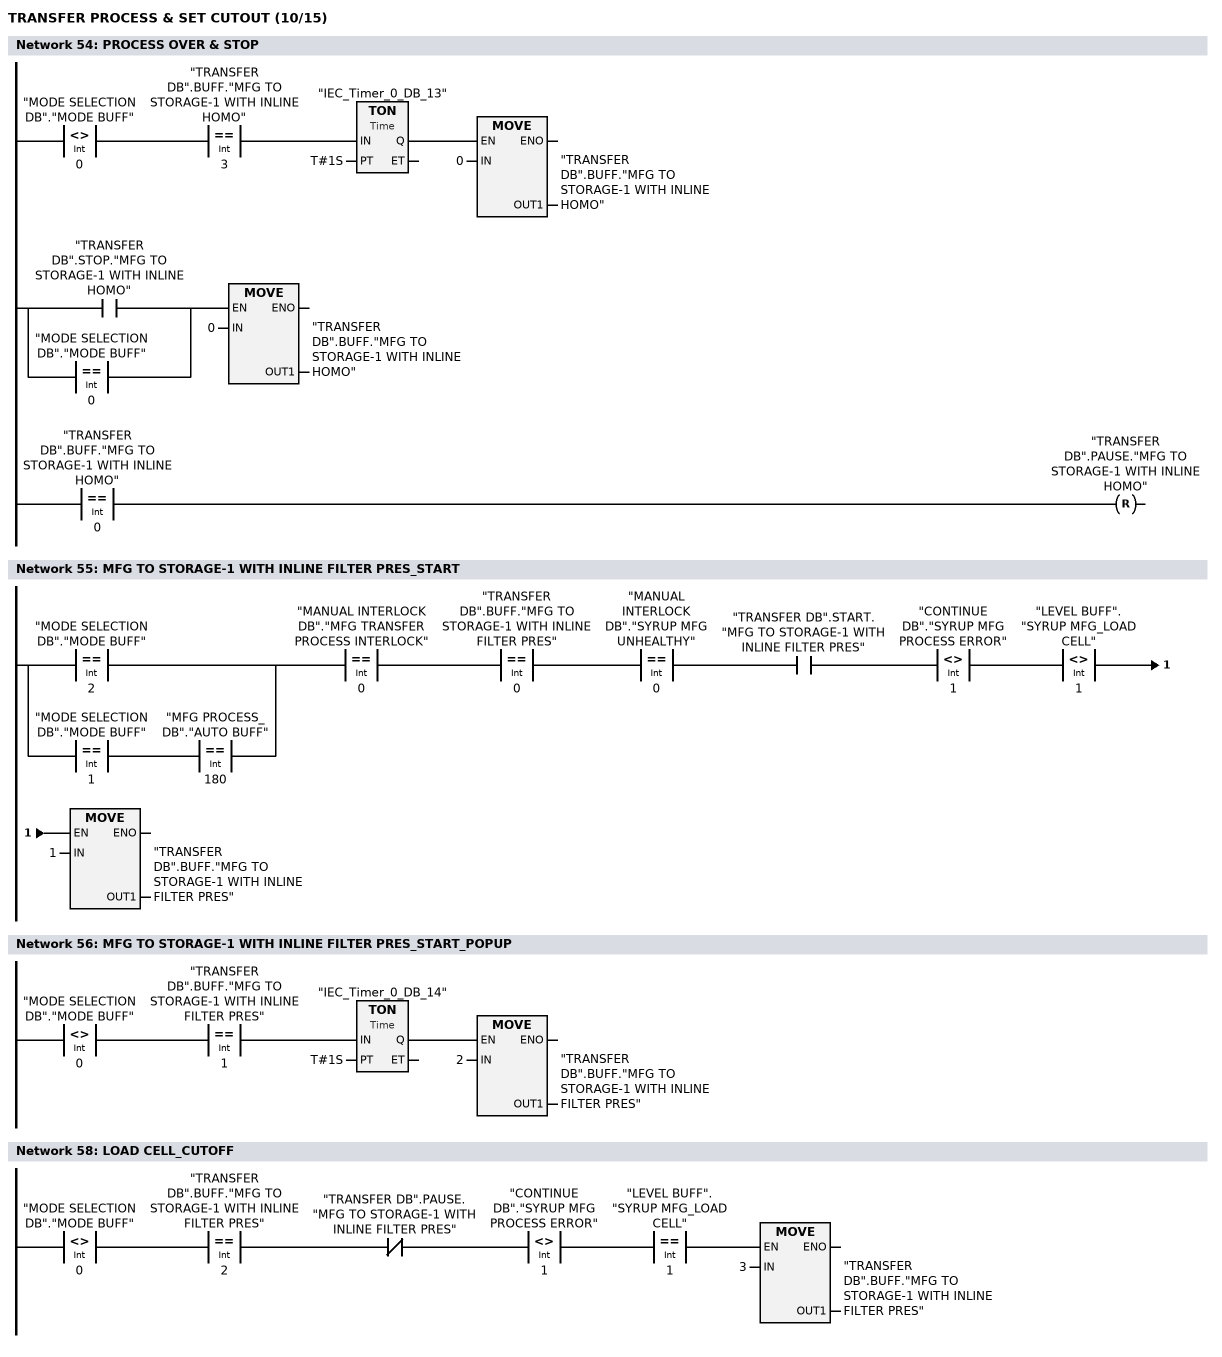
   RUNG wire#powerrail
      { S7_Templates := "SrcType := Int" } NE_Contact(in1 := "MODE SELECTION DB"."MODE BUFF", in2 := 0)
      { S7_Templates := "SrcType := Int" } EQ_Contact(in1 := "TRANSFER DB".BUFF."MFG TO STORAGE-1 WITH INLINE HOMO", in2 := 3)
      { S7_Templates := "time_type := Time" } "IEC_Timer_0_DB_13".TON(pt := T#1S, et =>)
      Move(in := 0, out1 => "TRANSFER DB".BUFF."MFG TO STORAGE-1 WITH INLINE HOMO")
   END_RUNG
   RUNG wire#powerrail
      Contact( "TRANSFER DB".STOP."MFG TO STORAGE-1 WITH INLINE HOMO" )
      wire#w1
      Move(in := 0, out1 => "TRANSFER DB".BUFF."MFG TO STORAGE-1 WITH INLINE HOMO")
   END_RUNG
   RUNG wire#powerrail
      { S7_Templates := "SrcType := Int" } EQ_Contact(in1 := "MODE SELECTION DB"."MODE BUFF", in2 := 0)
   END_RUNG wire#w1
   RUNG wire#powerrail
      { S7_Templates := "SrcType := Int" } EQ_Contact(in1 := "TRANSFER DB".BUFF."MFG TO STORAGE-1 WITH INLINE HOMO", in2 := 0)
      R_Coil( "TRANSFER DB".PAUSE."MFG TO STORAGE-1 WITH INLINE HOMO" )
   END_RUNG
   // the same network as SCL:
   "IEC_Timer_0_DB_13".TON(IN := ("MODE SELECTION DB"."MODE BUFF" <> 0) AND ("TRANSFER DB".BUFF."MFG TO STORAGE-1 WITH INLINE HOMO" = 3),
                           PT := T#1S);
   IF "IEC_Timer_0_DB_13".Q THEN "TRANSFER DB".BUFF."MFG TO STORAGE-1 WITH INLINE HOMO" := 0; END_IF;
   IF "TRANSFER DB".STOP."MFG TO STORAGE-1 WITH INLINE HOMO" OR ("MODE SELECTION DB"."MODE BUFF" = 0) THEN
       "TRANSFER DB".BUFF."MFG TO STORAGE-1 WITH INLINE HOMO" := 0;
   END_IF;
   IF "TRANSFER DB".BUFF."MFG TO STORAGE-1 WITH INLINE HOMO" = 0 THEN
       "TRANSFER DB".PAUSE."MFG TO STORAGE-1 WITH INLINE HOMO" := FALSE;
   END_IF;
END_REGION

REGION Network 55: MFG TO STORAGE-1 WITH INLINE FILTER PRES_START
   RUNG wire#powerrail
      { S7_Templates := "SrcType := Int" } EQ_Contact(in1 := "MODE SELECTION DB"."MODE BUFF", in2 := 2)
      wire#w1
      { S7_Templates := "SrcType := Int" } EQ_Contact(in1 := "MANUAL INTERLOCK DB"."MFG TRANSFER PROCESS INTERLOCK", in2 := 0)
      { S7_Templates := "SrcType := Int" } EQ_Contact(in1 := "TRANSFER DB".BUFF."MFG TO STORAGE-1 WITH INLINE FILTER PRES", in2 := 0)
      { S7_Templates := "SrcType := Int" } EQ_Contact(in1 := "MANUAL INTERLOCK DB"."SYRUP MFG UNHEALTHY", in2 := 0)
      Contact( "TRANSFER DB".START."MFG TO STORAGE-1 WITH INLINE FILTER PRES" )
      { S7_Templates := "SrcType := Int" } NE_Contact(in1 := "CONTINUE DB"."SYRUP MFG PROCESS ERROR", in2 := 1)
      { S7_Templates := "SrcType := Int" } NE_Contact(in1 := "LEVEL BUFF"."SYRUP MFG_LOAD CELL", in2 := 1)
      Move(in := 1, out1 => "TRANSFER DB".BUFF."MFG TO STORAGE-1 WITH INLINE FILTER PRES")
   END_RUNG
   RUNG wire#powerrail
      { S7_Templates := "SrcType := Int" } EQ_Contact(in1 := "MODE SELECTION DB"."MODE BUFF", in2 := 1)
      { S7_Templates := "SrcType := Int" } EQ_Contact(in1 := "MFG PROCESS_DB"."AUTO BUFF", in2 := 180)
   END_RUNG wire#w1
   // the same network as SCL:
   IF (("MODE SELECTION DB"."MODE BUFF" = 2) OR (("MODE SELECTION DB"."MODE BUFF" = 1) AND ("MFG PROCESS_DB"."AUTO BUFF" = 180))) AND ("MANUAL INTERLOCK DB"."MFG TRANSFER PROCESS INTERLOCK" = 0) AND ("TRANSFER DB".BUFF."MFG TO STORAGE-1 WITH INLINE FILTER PRES" = 0) AND ("MANUAL INTERLOCK DB"."SYRUP MFG UNHEALTHY" = 0) AND "TRANSFER DB".START."MFG TO STORAGE-1 WITH INLINE FILTER PRES" AND ("CONTINUE DB"."SYRUP MFG PROCESS ERROR" <> 1) AND ("LEVEL BUFF"."SYRUP MFG_LOAD CELL" <> 1) THEN
       "TRANSFER DB".BUFF."MFG TO STORAGE-1 WITH INLINE FILTER PRES" := 1;
   END_IF;
END_REGION

REGION Network 56: MFG TO STORAGE-1 WITH INLINE FILTER PRES_START_POPUP
   RUNG wire#powerrail
      { S7_Templates := "SrcType := Int" } NE_Contact(in1 := "MODE SELECTION DB"."MODE BUFF", in2 := 0)
      { S7_Templates := "SrcType := Int" } EQ_Contact(in1 := "TRANSFER DB".BUFF."MFG TO STORAGE-1 WITH INLINE FILTER PRES", in2 := 1)
      { S7_Templates := "time_type := Time" } "IEC_Timer_0_DB_14".TON(pt := T#1S, et =>)
      Move(in := 2, out1 => "TRANSFER DB".BUFF."MFG TO STORAGE-1 WITH INLINE FILTER PRES")
   END_RUNG
   // the same network as SCL:
   "IEC_Timer_0_DB_14".TON(IN := ("MODE SELECTION DB"."MODE BUFF" <> 0) AND ("TRANSFER DB".BUFF."MFG TO STORAGE-1 WITH INLINE FILTER PRES" = 1),
                           PT := T#1S);
   IF "IEC_Timer_0_DB_14".Q THEN "TRANSFER DB".BUFF."MFG TO STORAGE-1 WITH INLINE FILTER PRES" := 2; END_IF;
END_REGION

REGION Network 57 (SCL): OPENVALVE
   IF ("MODE SELECTION DB"."MODE BUFF" <> 0 AND "TRANSFER DB".BUFF."MFG TO STORAGE-1 WITH INLINE FILTER PRES" = 2
       AND NOT "TRANSFER DB".PAUSE."MFG TO STORAGE-1 WITH INLINE FILTER PRES"
       AND "CONTINUE DB"."SYRUP MFG PROCESS ERROR" = 0 AND "LEVEL BUFF"."SYRUP MFG_LOAD CELL" = 0)
       OR ("MODE SELECTION DB"."MODE BUFF"=1 AND "MFG PROCESS_DB"."AUTO BUFF"=0
       AND "MFG TRANSFER CYCLE DB".TRANSFER."TRANSFER BUFF"."MFG TO STORAGE-1 WITH INLINE FILTER PRES"=10 AND "CONTINUE DB"."SYRUP MFG PROCESS ERROR" <>1
       AND "MFG TRANSFER CYCLE DB".TRANSFER.SELECT."SELECT BUFF"=2)
   THEN
       "TRANSFER DB".BIT."MFG TO STORAGE-1 WITH INLINE FILTER PRES"."PFBV-59 TANK OUTLET VALVE" := TRUE;
       "TRANSFER DB".BIT."MFG TO STORAGE-1 WITH INLINE FILTER PRES"."PBV-114 TANK OUTLET TO INLINE HOMOGENIZER LINE" := TRUE;
       "TRANSFER DB".BIT."MFG TO STORAGE-1 WITH INLINE FILTER PRES"."PBV-108 INLINE HOMOGENIZER TO FILTER PRESS INLET LINE" := TRUE;
       "TRANSFER DB".BIT."MFG TO STORAGE-1 WITH INLINE FILTER PRES"."FILTER PRESS MOTOR 1 RUN" := TRUE;
       "TRANSFER DB".BIT."MFG TO STORAGE-1 WITH INLINE FILTER PRES"."PBV-118 FILTER PRESS INLET" := TRUE;
       "TRANSFER DB".BIT."MFG TO STORAGE-1 WITH INLINE FILTER PRES"."PBV-111 FILTER PRESS OUTLER VALVE" := TRUE;
       "TRANSFER DB".BIT."MFG TO STORAGE-1 WITH INLINE FILTER PRES"."PBV-112 FILTER PRESS TO TRANSFER LINE" := TRUE;
       "TRANSFER DB".BIT."MFG TO STORAGE-1 WITH INLINE FILTER PRES"."PBV-115 MFG TO STORAGE – 1 TRANSFER LINE" := TRUE;
   ELSE
       "TRANSFER DB".BIT."MFG TO STORAGE-1 WITH INLINE FILTER PRES"."PFBV-59 TANK OUTLET VALVE" := FALSE;
       "TRANSFER DB".BIT."MFG TO STORAGE-1 WITH INLINE FILTER PRES"."PBV-114 TANK OUTLET TO INLINE HOMOGENIZER LINE" := FALSE;
       "TRANSFER DB".BIT."MFG TO STORAGE-1 WITH INLINE FILTER PRES"."PBV-108 INLINE HOMOGENIZER TO FILTER PRESS INLET LINE" := FALSE;
       "TRANSFER DB".BIT."MFG TO STORAGE-1 WITH INLINE FILTER PRES"."FILTER PRESS MOTOR 1 RUN" := FALSE;
       "TRANSFER DB".BIT."MFG TO STORAGE-1 WITH INLINE FILTER PRES"."PBV-118 FILTER PRESS INLET" := FALSE;
       "TRANSFER DB".BIT."MFG TO STORAGE-1 WITH INLINE FILTER PRES"."PBV-111 FILTER PRESS OUTLER VALVE" := FALSE;
       "TRANSFER DB".BIT."MFG TO STORAGE-1 WITH INLINE FILTER PRES"."PBV-112 FILTER PRESS TO TRANSFER LINE" := FALSE;
       "TRANSFER DB".BIT."MFG TO STORAGE-1 WITH INLINE FILTER PRES"."PBV-115 MFG TO STORAGE – 1 TRANSFER LINE" := FALSE;
       ;
   END_IF;
END_REGION

REGION Network 58: LOAD CELL_CUTOFF
   RUNG wire#powerrail
      { S7_Templates := "SrcType := Int" } NE_Contact(in1 := "MODE SELECTION DB"."MODE BUFF", in2 := 0)
      { S7_Templates := "SrcType := Int" } EQ_Contact(in1 := "TRANSFER DB".BUFF."MFG TO STORAGE-1 WITH INLINE FILTER PRES", in2 := 2)
      I_Contact( "TRANSFER DB".PAUSE."MFG TO STORAGE-1 WITH INLINE FILTER PRES" )
      { S7_Templates := "SrcType := Int" } NE_Contact(in1 := "CONTINUE DB"."SYRUP MFG PROCESS ERROR", in2 := 1)
      { S7_Templates := "SrcType := Int" } EQ_Contact(in1 := "LEVEL BUFF"."SYRUP MFG_LOAD CELL", in2 := 1)
      Move(in := 3, out1 => "TRANSFER DB".BUFF."MFG TO STORAGE-1 WITH INLINE FILTER PRES")
   END_RUNG
   // the same network as SCL:
   IF ("MODE SELECTION DB"."MODE BUFF" <> 0) AND ("TRANSFER DB".BUFF."MFG TO STORAGE-1 WITH INLINE FILTER PRES" = 2) AND NOT "TRANSFER DB".PAUSE."MFG TO STORAGE-1 WITH INLINE FILTER PRES" AND ("CONTINUE DB"."SYRUP MFG PROCESS ERROR" <> 1) AND ("LEVEL BUFF"."SYRUP MFG_LOAD CELL" = 1) THEN
       "TRANSFER DB".BUFF."MFG TO STORAGE-1 WITH INLINE FILTER PRES" := 3;
   END_IF;
END_REGION

REGION Network 59: PROCESS OVER & STOP
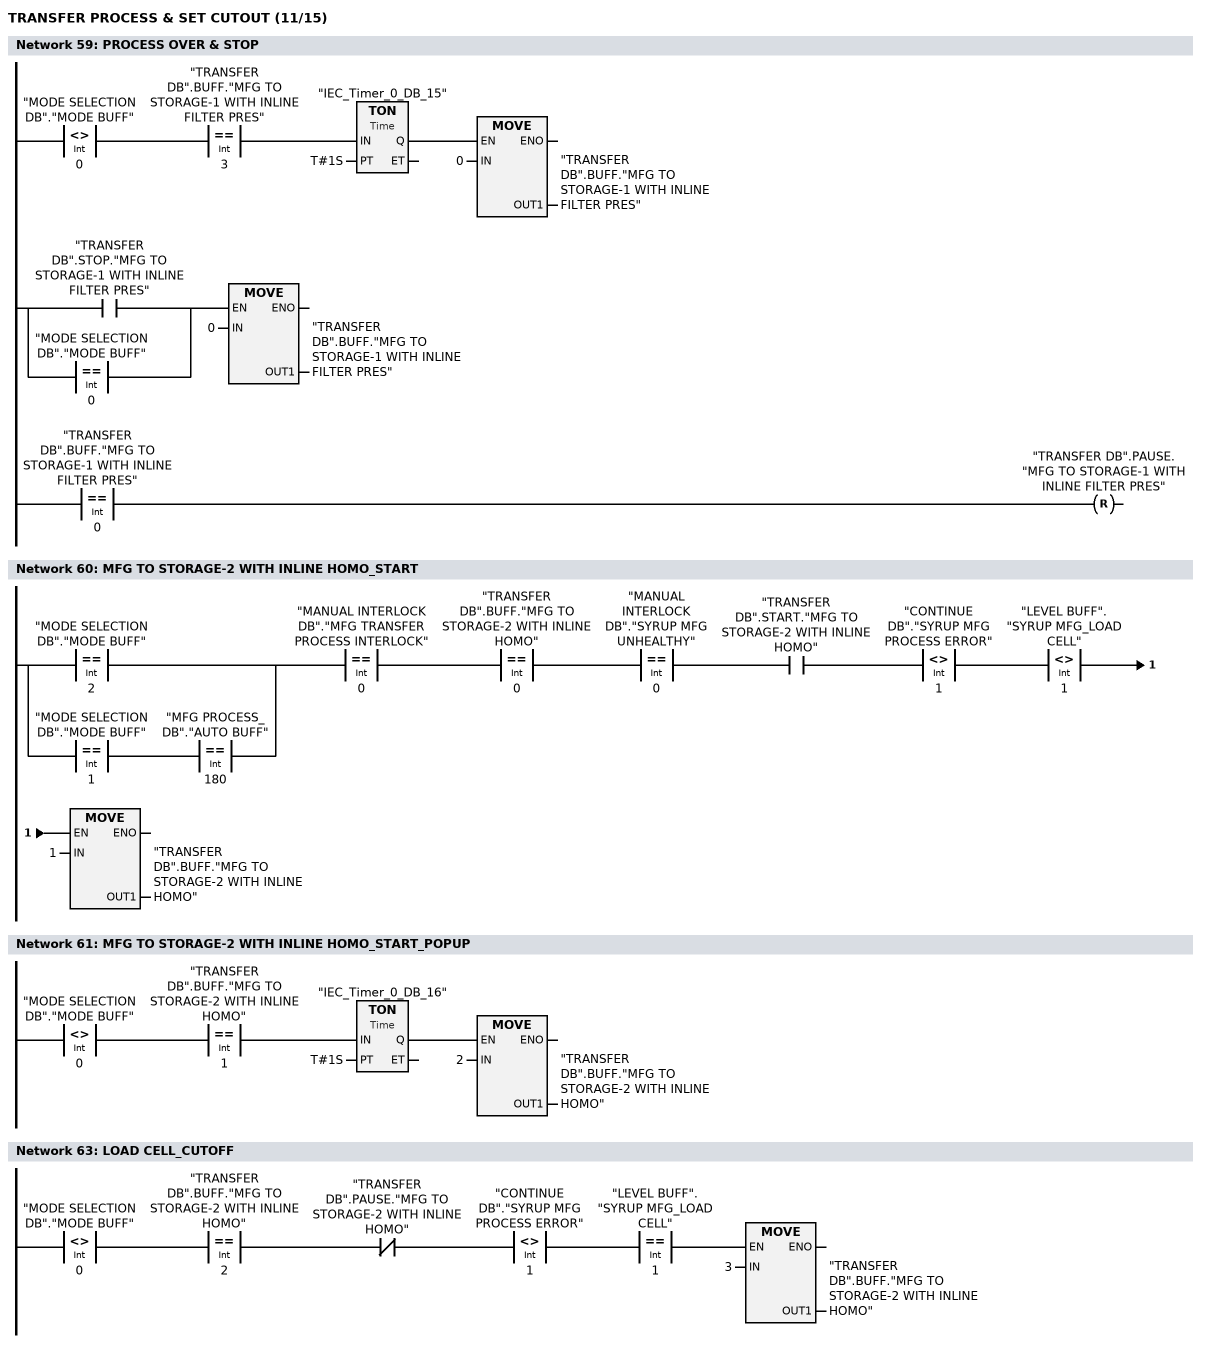
   RUNG wire#powerrail
      { S7_Templates := "SrcType := Int" } NE_Contact(in1 := "MODE SELECTION DB"."MODE BUFF", in2 := 0)
      { S7_Templates := "SrcType := Int" } EQ_Contact(in1 := "TRANSFER DB".BUFF."MFG TO STORAGE-1 WITH INLINE FILTER PRES", in2 := 3)
      { S7_Templates := "time_type := Time" } "IEC_Timer_0_DB_15".TON(pt := T#1S, et =>)
      Move(in := 0, out1 => "TRANSFER DB".BUFF."MFG TO STORAGE-1 WITH INLINE FILTER PRES")
   END_RUNG
   RUNG wire#powerrail
      Contact( "TRANSFER DB".STOP."MFG TO STORAGE-1 WITH INLINE FILTER PRES" )
      wire#w1
      Move(in := 0, out1 => "TRANSFER DB".BUFF."MFG TO STORAGE-1 WITH INLINE FILTER PRES")
   END_RUNG
   RUNG wire#powerrail
      { S7_Templates := "SrcType := Int" } EQ_Contact(in1 := "MODE SELECTION DB"."MODE BUFF", in2 := 0)
   END_RUNG wire#w1
   RUNG wire#powerrail
      { S7_Templates := "SrcType := Int" } EQ_Contact(in1 := "TRANSFER DB".BUFF."MFG TO STORAGE-1 WITH INLINE FILTER PRES", in2 := 0)
      R_Coil( "TRANSFER DB".PAUSE."MFG TO STORAGE-1 WITH INLINE FILTER PRES" )
   END_RUNG
   // the same network as SCL:
   "IEC_Timer_0_DB_15".TON(IN := ("MODE SELECTION DB"."MODE BUFF" <> 0) AND ("TRANSFER DB".BUFF."MFG TO STORAGE-1 WITH INLINE FILTER PRES" = 3),
                           PT := T#1S);
   IF "IEC_Timer_0_DB_15".Q THEN "TRANSFER DB".BUFF."MFG TO STORAGE-1 WITH INLINE FILTER PRES" := 0; END_IF;
   IF "TRANSFER DB".STOP."MFG TO STORAGE-1 WITH INLINE FILTER PRES" OR ("MODE SELECTION DB"."MODE BUFF" = 0) THEN
       "TRANSFER DB".BUFF."MFG TO STORAGE-1 WITH INLINE FILTER PRES" := 0;
   END_IF;
   IF "TRANSFER DB".BUFF."MFG TO STORAGE-1 WITH INLINE FILTER PRES" = 0 THEN
       "TRANSFER DB".PAUSE."MFG TO STORAGE-1 WITH INLINE FILTER PRES" := FALSE;
   END_IF;
END_REGION

REGION Network 60: MFG TO STORAGE-2 WITH INLINE HOMO_START
   RUNG wire#powerrail
      { S7_Templates := "SrcType := Int" } EQ_Contact(in1 := "MODE SELECTION DB"."MODE BUFF", in2 := 2)
      wire#w1
      { S7_Templates := "SrcType := Int" } EQ_Contact(in1 := "MANUAL INTERLOCK DB"."MFG TRANSFER PROCESS INTERLOCK", in2 := 0)
      { S7_Templates := "SrcType := Int" } EQ_Contact(in1 := "TRANSFER DB".BUFF."MFG TO STORAGE-2 WITH INLINE HOMO", in2 := 0)
      { S7_Templates := "SrcType := Int" } EQ_Contact(in1 := "MANUAL INTERLOCK DB"."SYRUP MFG UNHEALTHY", in2 := 0)
      Contact( "TRANSFER DB".START."MFG TO STORAGE-2 WITH INLINE HOMO" )
      { S7_Templates := "SrcType := Int" } NE_Contact(in1 := "CONTINUE DB"."SYRUP MFG PROCESS ERROR", in2 := 1)
      { S7_Templates := "SrcType := Int" } NE_Contact(in1 := "LEVEL BUFF"."SYRUP MFG_LOAD CELL", in2 := 1)
      Move(in := 1, out1 => "TRANSFER DB".BUFF."MFG TO STORAGE-2 WITH INLINE HOMO")
   END_RUNG
   RUNG wire#powerrail
      { S7_Templates := "SrcType := Int" } EQ_Contact(in1 := "MODE SELECTION DB"."MODE BUFF", in2 := 1)
      { S7_Templates := "SrcType := Int" } EQ_Contact(in1 := "MFG PROCESS_DB"."AUTO BUFF", in2 := 180)
   END_RUNG wire#w1
   // the same network as SCL:
   IF (("MODE SELECTION DB"."MODE BUFF" = 2) OR (("MODE SELECTION DB"."MODE BUFF" = 1) AND ("MFG PROCESS_DB"."AUTO BUFF" = 180))) AND ("MANUAL INTERLOCK DB"."MFG TRANSFER PROCESS INTERLOCK" = 0) AND ("TRANSFER DB".BUFF."MFG TO STORAGE-2 WITH INLINE HOMO" = 0) AND ("MANUAL INTERLOCK DB"."SYRUP MFG UNHEALTHY" = 0) AND "TRANSFER DB".START."MFG TO STORAGE-2 WITH INLINE HOMO" AND ("CONTINUE DB"."SYRUP MFG PROCESS ERROR" <> 1) AND ("LEVEL BUFF"."SYRUP MFG_LOAD CELL" <> 1) THEN
       "TRANSFER DB".BUFF."MFG TO STORAGE-2 WITH INLINE HOMO" := 1;
   END_IF;
END_REGION

REGION Network 61: MFG TO STORAGE-2 WITH INLINE HOMO_START_POPUP
   RUNG wire#powerrail
      { S7_Templates := "SrcType := Int" } NE_Contact(in1 := "MODE SELECTION DB"."MODE BUFF", in2 := 0)
      { S7_Templates := "SrcType := Int" } EQ_Contact(in1 := "TRANSFER DB".BUFF."MFG TO STORAGE-2 WITH INLINE HOMO", in2 := 1)
      { S7_Templates := "time_type := Time" } "IEC_Timer_0_DB_16".TON(pt := T#1S, et =>)
      Move(in := 2, out1 => "TRANSFER DB".BUFF."MFG TO STORAGE-2 WITH INLINE HOMO")
   END_RUNG
   // the same network as SCL:
   "IEC_Timer_0_DB_16".TON(IN := ("MODE SELECTION DB"."MODE BUFF" <> 0) AND ("TRANSFER DB".BUFF."MFG TO STORAGE-2 WITH INLINE HOMO" = 1),
                           PT := T#1S);
   IF "IEC_Timer_0_DB_16".Q THEN "TRANSFER DB".BUFF."MFG TO STORAGE-2 WITH INLINE HOMO" := 2; END_IF;
END_REGION

REGION Network 62 (SCL): OPENVALVE
   IF ("MODE SELECTION DB"."MODE BUFF" <> 0 AND "TRANSFER DB".BUFF."MFG TO STORAGE-2 WITH INLINE HOMO" = 2
       AND NOT "TRANSFER DB".PAUSE."MFG TO STORAGE-2 WITH INLINE HOMO"
       AND "CONTINUE DB"."SYRUP MFG PROCESS ERROR" = 0 AND "LEVEL BUFF"."SYRUP MFG_LOAD CELL" = 0)
       OR ("MODE SELECTION DB"."MODE BUFF"=1 AND "MFG PROCESS_DB"."AUTO BUFF"=0
       AND "MFG TRANSFER CYCLE DB".TRANSFER."TRANSFER BUFF"."MFG TO STORAGE-2 WITH INLINE HOMO"=10 AND "CONTINUE DB"."SYRUP MFG PROCESS ERROR" <>1
       AND "MFG TRANSFER CYCLE DB".TRANSFER.SELECT."SELECT BUFF"=3)
   THEN
       "TRANSFER DB".BIT."MFG TO STORAGE-2 WITH INLINE HOMO"."PFBV-59 TANK OUTLET VALVE" := TRUE;
       "TRANSFER DB".BIT."MFG TO STORAGE-2 WITH INLINE HOMO"."PBV-114 TANK OUTLET TO INLINE HOMOGENIZER LINE" := TRUE;
       "TRANSFER DB".BIT."MFG TO STORAGE-2 WITH INLINE HOMO"."PBV-110 INLINE HOMOGENIZER TO INLET LINE" := TRUE;
       "TRANSFER DB".BIT."MFG TO STORAGE-2 WITH INLINE HOMO"."PAV-56 INLINE HOMO. SEAL COOLING INLET" := TRUE;
       "TRANSFER DB".BIT."MFG TO STORAGE-2 WITH INLINE HOMO"."INLINE 1 HOMOGENIZER MOTOR1 RUN" := TRUE;
       "TRANSFER DB".BIT."MFG TO STORAGE-2 WITH INLINE HOMO"."PBV-109 HOMO. RECIRCULATION INLET" := TRUE;
       "TRANSFER DB".BIT."MFG TO STORAGE-2 WITH INLINE HOMO"."PBV-116 MFG TO STORAGE – 2 TRANSFER LINE" := TRUE;
   ELSE
       "TRANSFER DB".BIT."MFG TO STORAGE-2 WITH INLINE HOMO"."PFBV-59 TANK OUTLET VALVE" := FALSE;
       "TRANSFER DB".BIT."MFG TO STORAGE-2 WITH INLINE HOMO"."PBV-114 TANK OUTLET TO INLINE HOMOGENIZER LINE" := FALSE;
       "TRANSFER DB".BIT."MFG TO STORAGE-2 WITH INLINE HOMO"."PBV-110 INLINE HOMOGENIZER TO INLET LINE" := FALSE;
       "TRANSFER DB".BIT."MFG TO STORAGE-2 WITH INLINE HOMO"."PAV-56 INLINE HOMO. SEAL COOLING INLET" := FALSE;
       "TRANSFER DB".BIT."MFG TO STORAGE-2 WITH INLINE HOMO"."INLINE 1 HOMOGENIZER MOTOR1 RUN" := FALSE;
       "TRANSFER DB".BIT."MFG TO STORAGE-2 WITH INLINE HOMO"."PBV-109 HOMO. RECIRCULATION INLET" := FALSE;
       "TRANSFER DB".BIT."MFG TO STORAGE-2 WITH INLINE HOMO"."PBV-116 MFG TO STORAGE – 2 TRANSFER LINE" := FALSE;
       ;
   END_IF;
END_REGION

REGION Network 63: LOAD CELL_CUTOFF
   RUNG wire#powerrail
      { S7_Templates := "SrcType := Int" } NE_Contact(in1 := "MODE SELECTION DB"."MODE BUFF", in2 := 0)
      { S7_Templates := "SrcType := Int" } EQ_Contact(in1 := "TRANSFER DB".BUFF."MFG TO STORAGE-2 WITH INLINE HOMO", in2 := 2)
      I_Contact( "TRANSFER DB".PAUSE."MFG TO STORAGE-2 WITH INLINE HOMO" )
      { S7_Templates := "SrcType := Int" } NE_Contact(in1 := "CONTINUE DB"."SYRUP MFG PROCESS ERROR", in2 := 1)
      { S7_Templates := "SrcType := Int" } EQ_Contact(in1 := "LEVEL BUFF"."SYRUP MFG_LOAD CELL", in2 := 1)
      Move(in := 3, out1 => "TRANSFER DB".BUFF."MFG TO STORAGE-2 WITH INLINE HOMO")
   END_RUNG
   // the same network as SCL:
   IF ("MODE SELECTION DB"."MODE BUFF" <> 0) AND ("TRANSFER DB".BUFF."MFG TO STORAGE-2 WITH INLINE HOMO" = 2) AND NOT "TRANSFER DB".PAUSE."MFG TO STORAGE-2 WITH INLINE HOMO" AND ("CONTINUE DB"."SYRUP MFG PROCESS ERROR" <> 1) AND ("LEVEL BUFF"."SYRUP MFG_LOAD CELL" = 1) THEN
       "TRANSFER DB".BUFF."MFG TO STORAGE-2 WITH INLINE HOMO" := 3;
   END_IF;
END_REGION

REGION Network 64: PROCESS OVER & STOP
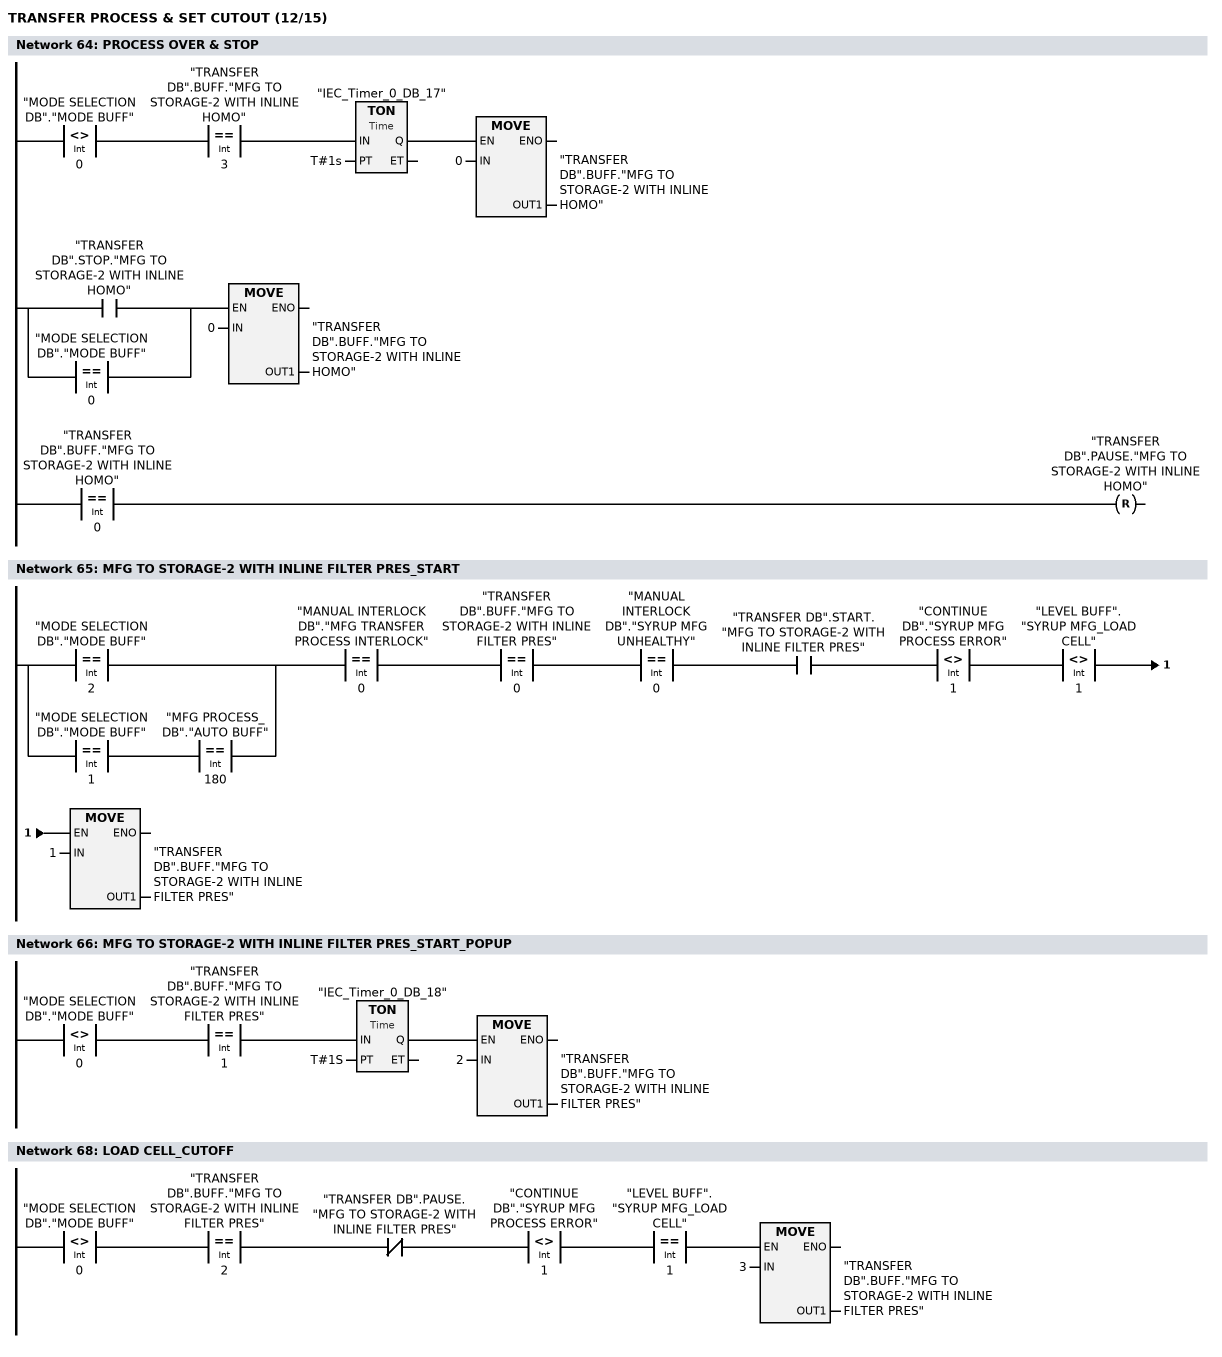
   RUNG wire#powerrail
      { S7_Templates := "SrcType := Int" } NE_Contact(in1 := "MODE SELECTION DB"."MODE BUFF", in2 := 0)
      { S7_Templates := "SrcType := Int" } EQ_Contact(in1 := "TRANSFER DB".BUFF."MFG TO STORAGE-2 WITH INLINE HOMO", in2 := 3)
      { S7_Templates := "time_type := Time" } "IEC_Timer_0_DB_17".TON(pt := T#1s, et =>)
      Move(in := 0, out1 => "TRANSFER DB".BUFF."MFG TO STORAGE-2 WITH INLINE HOMO")
   END_RUNG
   RUNG wire#powerrail
      Contact( "TRANSFER DB".STOP."MFG TO STORAGE-2 WITH INLINE HOMO" )
      wire#w1
      Move(in := 0, out1 => "TRANSFER DB".BUFF."MFG TO STORAGE-2 WITH INLINE HOMO")
   END_RUNG
   RUNG wire#powerrail
      { S7_Templates := "SrcType := Int" } EQ_Contact(in1 := "MODE SELECTION DB"."MODE BUFF", in2 := 0)
   END_RUNG wire#w1
   RUNG wire#powerrail
      { S7_Templates := "SrcType := Int" } EQ_Contact(in1 := "TRANSFER DB".BUFF."MFG TO STORAGE-2 WITH INLINE HOMO", in2 := 0)
      R_Coil( "TRANSFER DB".PAUSE."MFG TO STORAGE-2 WITH INLINE HOMO" )
   END_RUNG
   // the same network as SCL:
   "IEC_Timer_0_DB_17".TON(IN := ("MODE SELECTION DB"."MODE BUFF" <> 0) AND ("TRANSFER DB".BUFF."MFG TO STORAGE-2 WITH INLINE HOMO" = 3),
                           PT := T#1s);
   IF "IEC_Timer_0_DB_17".Q THEN "TRANSFER DB".BUFF."MFG TO STORAGE-2 WITH INLINE HOMO" := 0; END_IF;
   IF "TRANSFER DB".STOP."MFG TO STORAGE-2 WITH INLINE HOMO" OR ("MODE SELECTION DB"."MODE BUFF" = 0) THEN
       "TRANSFER DB".BUFF."MFG TO STORAGE-2 WITH INLINE HOMO" := 0;
   END_IF;
   IF "TRANSFER DB".BUFF."MFG TO STORAGE-2 WITH INLINE HOMO" = 0 THEN
       "TRANSFER DB".PAUSE."MFG TO STORAGE-2 WITH INLINE HOMO" := FALSE;
   END_IF;
END_REGION

REGION Network 65: MFG TO STORAGE-2 WITH INLINE FILTER PRES_START
   RUNG wire#powerrail
      { S7_Templates := "SrcType := Int" } EQ_Contact(in1 := "MODE SELECTION DB"."MODE BUFF", in2 := 2)
      wire#w1
      { S7_Templates := "SrcType := Int" } EQ_Contact(in1 := "MANUAL INTERLOCK DB"."MFG TRANSFER PROCESS INTERLOCK", in2 := 0)
      { S7_Templates := "SrcType := Int" } EQ_Contact(in1 := "TRANSFER DB".BUFF."MFG TO STORAGE-2 WITH INLINE FILTER PRES", in2 := 0)
      { S7_Templates := "SrcType := Int" } EQ_Contact(in1 := "MANUAL INTERLOCK DB"."SYRUP MFG UNHEALTHY", in2 := 0)
      Contact( "TRANSFER DB".START."MFG TO STORAGE-2 WITH INLINE FILTER PRES" )
      { S7_Templates := "SrcType := Int" } NE_Contact(in1 := "CONTINUE DB"."SYRUP MFG PROCESS ERROR", in2 := 1)
      { S7_Templates := "SrcType := Int" } NE_Contact(in1 := "LEVEL BUFF"."SYRUP MFG_LOAD CELL", in2 := 1)
      Move(in := 1, out1 => "TRANSFER DB".BUFF."MFG TO STORAGE-2 WITH INLINE FILTER PRES")
   END_RUNG
   RUNG wire#powerrail
      { S7_Templates := "SrcType := Int" } EQ_Contact(in1 := "MODE SELECTION DB"."MODE BUFF", in2 := 1)
      { S7_Templates := "SrcType := Int" } EQ_Contact(in1 := "MFG PROCESS_DB"."AUTO BUFF", in2 := 180)
   END_RUNG wire#w1
   // the same network as SCL:
   IF (("MODE SELECTION DB"."MODE BUFF" = 2) OR (("MODE SELECTION DB"."MODE BUFF" = 1) AND ("MFG PROCESS_DB"."AUTO BUFF" = 180))) AND ("MANUAL INTERLOCK DB"."MFG TRANSFER PROCESS INTERLOCK" = 0) AND ("TRANSFER DB".BUFF."MFG TO STORAGE-2 WITH INLINE FILTER PRES" = 0) AND ("MANUAL INTERLOCK DB"."SYRUP MFG UNHEALTHY" = 0) AND "TRANSFER DB".START."MFG TO STORAGE-2 WITH INLINE FILTER PRES" AND ("CONTINUE DB"."SYRUP MFG PROCESS ERROR" <> 1) AND ("LEVEL BUFF"."SYRUP MFG_LOAD CELL" <> 1) THEN
       "TRANSFER DB".BUFF."MFG TO STORAGE-2 WITH INLINE FILTER PRES" := 1;
   END_IF;
END_REGION

REGION Network 66: MFG TO STORAGE-2 WITH INLINE FILTER PRES_START_POPUP
   RUNG wire#powerrail
      { S7_Templates := "SrcType := Int" } NE_Contact(in1 := "MODE SELECTION DB"."MODE BUFF", in2 := 0)
      { S7_Templates := "SrcType := Int" } EQ_Contact(in1 := "TRANSFER DB".BUFF."MFG TO STORAGE-2 WITH INLINE FILTER PRES", in2 := 1)
      { S7_Templates := "time_type := Time" } "IEC_Timer_0_DB_18".TON(pt := T#1S, et =>)
      Move(in := 2, out1 => "TRANSFER DB".BUFF."MFG TO STORAGE-2 WITH INLINE FILTER PRES")
   END_RUNG
   // the same network as SCL:
   "IEC_Timer_0_DB_18".TON(IN := ("MODE SELECTION DB"."MODE BUFF" <> 0) AND ("TRANSFER DB".BUFF."MFG TO STORAGE-2 WITH INLINE FILTER PRES" = 1),
                           PT := T#1S);
   IF "IEC_Timer_0_DB_18".Q THEN "TRANSFER DB".BUFF."MFG TO STORAGE-2 WITH INLINE FILTER PRES" := 2; END_IF;
END_REGION

REGION Network 67 (SCL): OPENVALVE
   IF ("MODE SELECTION DB"."MODE BUFF" <> 0 AND "TRANSFER DB".BUFF."MFG TO STORAGE-2 WITH INLINE FILTER PRES" = 2
       AND NOT "TRANSFER DB".PAUSE."MFG TO STORAGE-2 WITH INLINE FILTER PRES" 
       AND "CONTINUE DB"."SYRUP MFG PROCESS ERROR" = 0 AND "LEVEL BUFF"."SYRUP MFG_LOAD CELL" = 0)
       OR ("MODE SELECTION DB"."MODE BUFF"=1 AND "MFG PROCESS_DB"."AUTO BUFF"=0
       AND "MFG TRANSFER CYCLE DB".TRANSFER."TRANSFER BUFF"."MFG TO STORAGE-2 WITH INLINE FILTER PRES"=10 AND "CONTINUE DB"."SYRUP MFG PROCESS ERROR" <>1
       AND "MFG TRANSFER CYCLE DB".TRANSFER.SELECT."SELECT BUFF"=4)
   THEN
       "TRANSFER DB".BIT."MFG TO STORAGE-2 WITH INLINE FILTER PRES"."PFBV-59 TANK OUTLET VALVE" := TRUE;
       "TRANSFER DB".BIT."MFG TO STORAGE-2 WITH INLINE FILTER PRES"."PBV-114 TANK OUTLET TO INLINE HOMOGENIZER LINE" := TRUE;
       "TRANSFER DB".BIT."MFG TO STORAGE-2 WITH INLINE FILTER PRES"."PBV-108 INLINE HOMOGENIZER TO FILTER PRESS INLET LINE" := TRUE;
       "TRANSFER DB".BIT."MFG TO STORAGE-2 WITH INLINE FILTER PRES"."FILTER PRESS MOTOR 1 RUN" := TRUE;
       "TRANSFER DB".BIT."MFG TO STORAGE-2 WITH INLINE FILTER PRES"."PBV-118 FILTER PRESS INLET" := TRUE;
       "TRANSFER DB".BIT."MFG TO STORAGE-2 WITH INLINE FILTER PRES"."PBV-111 FILTER PRESS OUTLER VALVE" := TRUE;
       "TRANSFER DB".BIT."MFG TO STORAGE-2 WITH INLINE FILTER PRES"."PBV-112 FILTER PRESS TO TRANSFER LINE" := TRUE;
       "TRANSFER DB".BIT."MFG TO STORAGE-2 WITH INLINE FILTER PRES"."PBV-116 MFG TO STORAGE – 2 TRANSFER LINE" := TRUE;
   ELSE
       "TRANSFER DB".BIT."MFG TO STORAGE-2 WITH INLINE FILTER PRES"."PFBV-59 TANK OUTLET VALVE" := FALSE;
       "TRANSFER DB".BIT."MFG TO STORAGE-2 WITH INLINE FILTER PRES"."PBV-114 TANK OUTLET TO INLINE HOMOGENIZER LINE" := FALSE;
       "TRANSFER DB".BIT."MFG TO STORAGE-2 WITH INLINE FILTER PRES"."PBV-108 INLINE HOMOGENIZER TO FILTER PRESS INLET LINE" := FALSE;
       "TRANSFER DB".BIT."MFG TO STORAGE-2 WITH INLINE FILTER PRES"."FILTER PRESS MOTOR 1 RUN" := FALSE;
       "TRANSFER DB".BIT."MFG TO STORAGE-2 WITH INLINE FILTER PRES"."PBV-118 FILTER PRESS INLET" := FALSE;
       "TRANSFER DB".BIT."MFG TO STORAGE-2 WITH INLINE FILTER PRES"."PBV-111 FILTER PRESS OUTLER VALVE" := FALSE;
       "TRANSFER DB".BIT."MFG TO STORAGE-2 WITH INLINE FILTER PRES"."PBV-112 FILTER PRESS TO TRANSFER LINE" := FALSE;
       "TRANSFER DB".BIT."MFG TO STORAGE-2 WITH INLINE FILTER PRES"."PBV-116 MFG TO STORAGE – 2 TRANSFER LINE" := FALSE;
       ;
   END_IF;
END_REGION

REGION Network 68: LOAD CELL_CUTOFF
   RUNG wire#powerrail
      { S7_Templates := "SrcType := Int" } NE_Contact(in1 := "MODE SELECTION DB"."MODE BUFF", in2 := 0)
      { S7_Templates := "SrcType := Int" } EQ_Contact(in1 := "TRANSFER DB".BUFF."MFG TO STORAGE-2 WITH INLINE FILTER PRES", in2 := 2)
      I_Contact( "TRANSFER DB".PAUSE."MFG TO STORAGE-2 WITH INLINE FILTER PRES" )
      { S7_Templates := "SrcType := Int" } NE_Contact(in1 := "CONTINUE DB"."SYRUP MFG PROCESS ERROR", in2 := 1)
      { S7_Templates := "SrcType := Int" } EQ_Contact(in1 := "LEVEL BUFF"."SYRUP MFG_LOAD CELL", in2 := 1)
      Move(in := 3, out1 => "TRANSFER DB".BUFF."MFG TO STORAGE-2 WITH INLINE FILTER PRES")
   END_RUNG
   // the same network as SCL:
   IF ("MODE SELECTION DB"."MODE BUFF" <> 0) AND ("TRANSFER DB".BUFF."MFG TO STORAGE-2 WITH INLINE FILTER PRES" = 2) AND NOT "TRANSFER DB".PAUSE."MFG TO STORAGE-2 WITH INLINE FILTER PRES" AND ("CONTINUE DB"."SYRUP MFG PROCESS ERROR" <> 1) AND ("LEVEL BUFF"."SYRUP MFG_LOAD CELL" = 1) THEN
       "TRANSFER DB".BUFF."MFG TO STORAGE-2 WITH INLINE FILTER PRES" := 3;
   END_IF;
END_REGION

REGION Network 69: PROCESS OVER & STOP
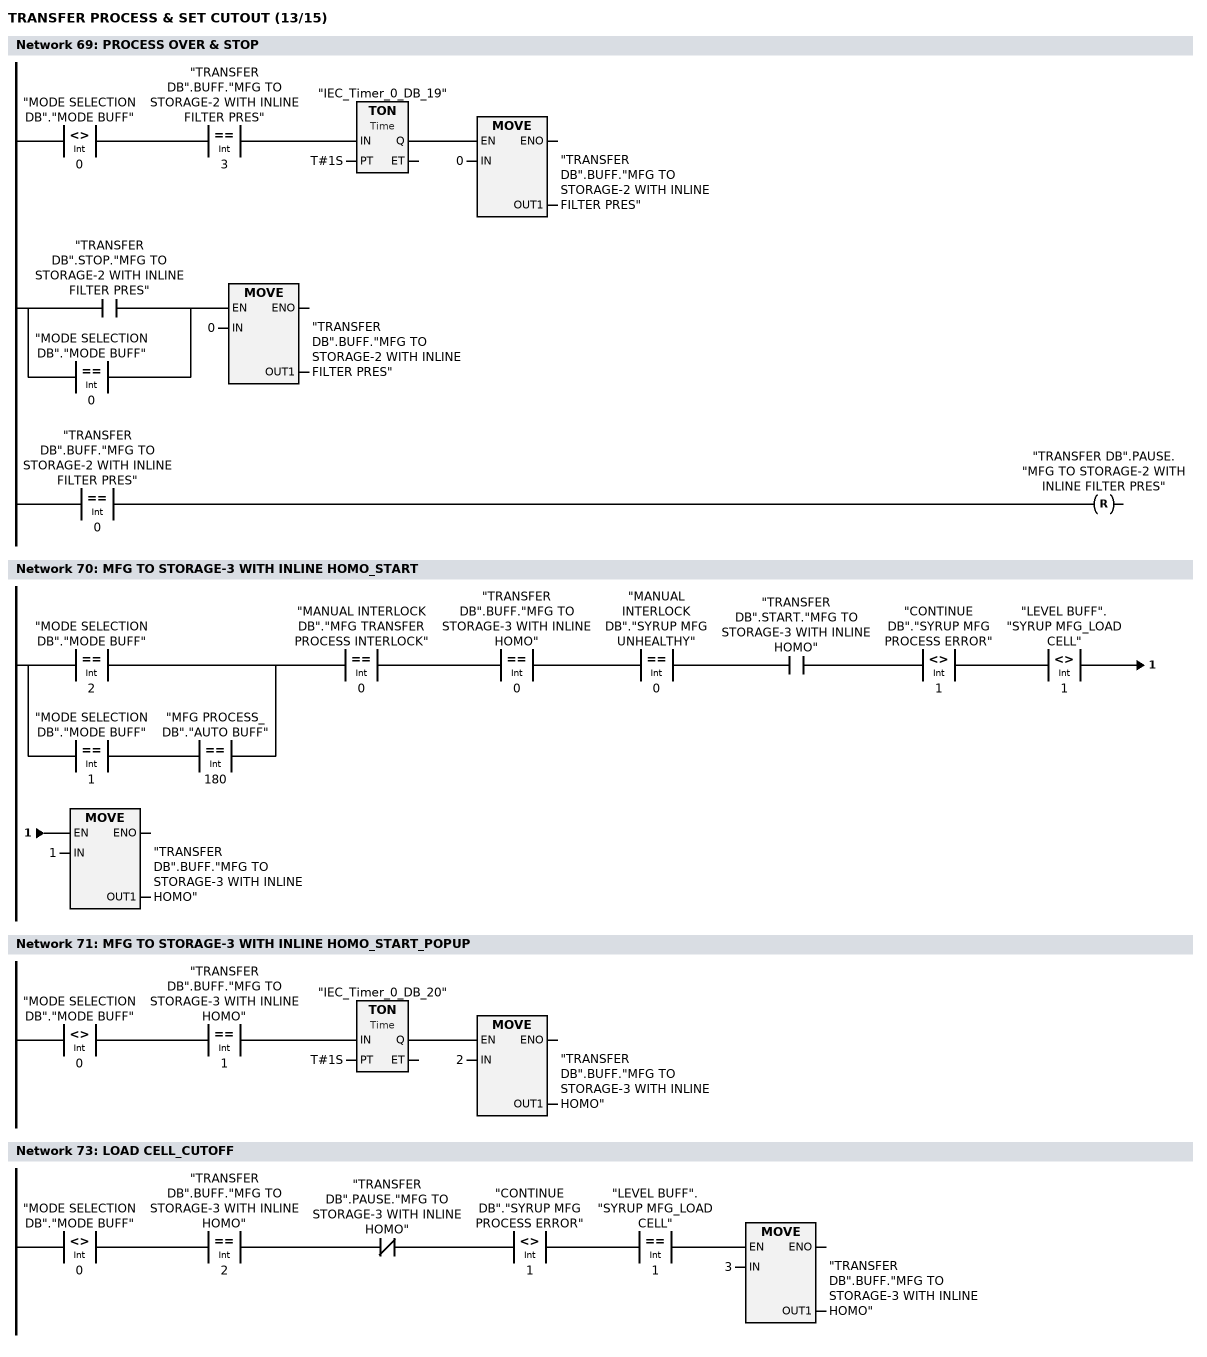
   RUNG wire#powerrail
      { S7_Templates := "SrcType := Int" } NE_Contact(in1 := "MODE SELECTION DB"."MODE BUFF", in2 := 0)
      { S7_Templates := "SrcType := Int" } EQ_Contact(in1 := "TRANSFER DB".BUFF."MFG TO STORAGE-2 WITH INLINE FILTER PRES", in2 := 3)
      { S7_Templates := "time_type := Time" } "IEC_Timer_0_DB_19".TON(pt := T#1S, et =>)
      Move(in := 0, out1 => "TRANSFER DB".BUFF."MFG TO STORAGE-2 WITH INLINE FILTER PRES")
   END_RUNG
   RUNG wire#powerrail
      Contact( "TRANSFER DB".STOP."MFG TO STORAGE-2 WITH INLINE FILTER PRES" )
      wire#w1
      Move(in := 0, out1 => "TRANSFER DB".BUFF."MFG TO STORAGE-2 WITH INLINE FILTER PRES")
   END_RUNG
   RUNG wire#powerrail
      { S7_Templates := "SrcType := Int" } EQ_Contact(in1 := "MODE SELECTION DB"."MODE BUFF", in2 := 0)
   END_RUNG wire#w1
   RUNG wire#powerrail
      { S7_Templates := "SrcType := Int" } EQ_Contact(in1 := "TRANSFER DB".BUFF."MFG TO STORAGE-2 WITH INLINE FILTER PRES", in2 := 0)
      R_Coil( "TRANSFER DB".PAUSE."MFG TO STORAGE-2 WITH INLINE FILTER PRES" )
   END_RUNG
   // the same network as SCL:
   "IEC_Timer_0_DB_19".TON(IN := ("MODE SELECTION DB"."MODE BUFF" <> 0) AND ("TRANSFER DB".BUFF."MFG TO STORAGE-2 WITH INLINE FILTER PRES" = 3),
                           PT := T#1S);
   IF "IEC_Timer_0_DB_19".Q THEN "TRANSFER DB".BUFF."MFG TO STORAGE-2 WITH INLINE FILTER PRES" := 0; END_IF;
   IF "TRANSFER DB".STOP."MFG TO STORAGE-2 WITH INLINE FILTER PRES" OR ("MODE SELECTION DB"."MODE BUFF" = 0) THEN
       "TRANSFER DB".BUFF."MFG TO STORAGE-2 WITH INLINE FILTER PRES" := 0;
   END_IF;
   IF "TRANSFER DB".BUFF."MFG TO STORAGE-2 WITH INLINE FILTER PRES" = 0 THEN
       "TRANSFER DB".PAUSE."MFG TO STORAGE-2 WITH INLINE FILTER PRES" := FALSE;
   END_IF;
END_REGION

REGION Network 70: MFG TO STORAGE-3 WITH INLINE HOMO_START
   RUNG wire#powerrail
      { S7_Templates := "SrcType := Int" } EQ_Contact(in1 := "MODE SELECTION DB"."MODE BUFF", in2 := 2)
      wire#w1
      { S7_Templates := "SrcType := Int" } EQ_Contact(in1 := "MANUAL INTERLOCK DB"."MFG TRANSFER PROCESS INTERLOCK", in2 := 0)
      { S7_Templates := "SrcType := Int" } EQ_Contact(in1 := "TRANSFER DB".BUFF."MFG TO STORAGE-3 WITH INLINE HOMO", in2 := 0)
      { S7_Templates := "SrcType := Int" } EQ_Contact(in1 := "MANUAL INTERLOCK DB"."SYRUP MFG UNHEALTHY", in2 := 0)
      Contact( "TRANSFER DB".START."MFG TO STORAGE-3 WITH INLINE HOMO" )
      { S7_Templates := "SrcType := Int" } NE_Contact(in1 := "CONTINUE DB"."SYRUP MFG PROCESS ERROR", in2 := 1)
      { S7_Templates := "SrcType := Int" } NE_Contact(in1 := "LEVEL BUFF"."SYRUP MFG_LOAD CELL", in2 := 1)
      Move(in := 1, out1 => "TRANSFER DB".BUFF."MFG TO STORAGE-3 WITH INLINE HOMO")
   END_RUNG
   RUNG wire#powerrail
      { S7_Templates := "SrcType := Int" } EQ_Contact(in1 := "MODE SELECTION DB"."MODE BUFF", in2 := 1)
      { S7_Templates := "SrcType := Int" } EQ_Contact(in1 := "MFG PROCESS_DB"."AUTO BUFF", in2 := 180)
   END_RUNG wire#w1
   // the same network as SCL:
   IF (("MODE SELECTION DB"."MODE BUFF" = 2) OR (("MODE SELECTION DB"."MODE BUFF" = 1) AND ("MFG PROCESS_DB"."AUTO BUFF" = 180))) AND ("MANUAL INTERLOCK DB"."MFG TRANSFER PROCESS INTERLOCK" = 0) AND ("TRANSFER DB".BUFF."MFG TO STORAGE-3 WITH INLINE HOMO" = 0) AND ("MANUAL INTERLOCK DB"."SYRUP MFG UNHEALTHY" = 0) AND "TRANSFER DB".START."MFG TO STORAGE-3 WITH INLINE HOMO" AND ("CONTINUE DB"."SYRUP MFG PROCESS ERROR" <> 1) AND ("LEVEL BUFF"."SYRUP MFG_LOAD CELL" <> 1) THEN
       "TRANSFER DB".BUFF."MFG TO STORAGE-3 WITH INLINE HOMO" := 1;
   END_IF;
END_REGION

REGION Network 71: MFG TO STORAGE-3 WITH INLINE HOMO_START_POPUP
   RUNG wire#powerrail
      { S7_Templates := "SrcType := Int" } NE_Contact(in1 := "MODE SELECTION DB"."MODE BUFF", in2 := 0)
      { S7_Templates := "SrcType := Int" } EQ_Contact(in1 := "TRANSFER DB".BUFF."MFG TO STORAGE-3 WITH INLINE HOMO", in2 := 1)
      { S7_Templates := "time_type := Time" } "IEC_Timer_0_DB_20".TON(pt := T#1S, et =>)
      Move(in := 2, out1 => "TRANSFER DB".BUFF."MFG TO STORAGE-3 WITH INLINE HOMO")
   END_RUNG
   // the same network as SCL:
   "IEC_Timer_0_DB_20".TON(IN := ("MODE SELECTION DB"."MODE BUFF" <> 0) AND ("TRANSFER DB".BUFF."MFG TO STORAGE-3 WITH INLINE HOMO" = 1),
                           PT := T#1S);
   IF "IEC_Timer_0_DB_20".Q THEN "TRANSFER DB".BUFF."MFG TO STORAGE-3 WITH INLINE HOMO" := 2; END_IF;
END_REGION

REGION Network 72 (SCL): OPENVALVE
   IF ("MODE SELECTION DB"."MODE BUFF" <> 0 AND "TRANSFER DB".BUFF."MFG TO STORAGE-3 WITH INLINE HOMO" = 2
       AND NOT "TRANSFER DB".PAUSE."MFG TO STORAGE-3 WITH INLINE HOMO"
       AND "CONTINUE DB"."SYRUP MFG PROCESS ERROR" = 0 AND "LEVEL BUFF"."SYRUP MFG_LOAD CELL" = 0)
       OR ("MODE SELECTION DB"."MODE BUFF"=1 AND "MFG PROCESS_DB"."AUTO BUFF"=0
       AND "MFG TRANSFER CYCLE DB".TRANSFER."TRANSFER BUFF"."MFG TO STORAGE-3 WITH INLINE HOMO"=10 AND "CONTINUE DB"."SYRUP MFG PROCESS ERROR" <>1
       AND "MFG TRANSFER CYCLE DB".TRANSFER.SELECT."SELECT BUFF"=5)
   THEN
       "TRANSFER DB".BIT."MFG TO STORAGE-3 WITH INLINE HOMO"."PFBV-59 TANK OUTLET VALVE" := TRUE;
       "TRANSFER DB".BIT."MFG TO STORAGE-3 WITH INLINE HOMO"."PBV-114 TANK OUTLET TO INLINE HOMOGENIZER LINE" := TRUE;
       "TRANSFER DB".BIT."MFG TO STORAGE-3 WITH INLINE HOMO"."PBV-110 INLINE HOMOGENIZER TO INLET LINE" := TRUE;
       "TRANSFER DB".BIT."MFG TO STORAGE-3 WITH INLINE HOMO"."PAV-56 INLINE HOMO. SEAL COOLING INLET" := TRUE;
       "TRANSFER DB".BIT."MFG TO STORAGE-3 WITH INLINE HOMO"."INLINE 1 HOMOGENIZER MOTOR1 RUN" := TRUE;
       "TRANSFER DB".BIT."MFG TO STORAGE-3 WITH INLINE HOMO"."PBV-109 HOMO. RECIRCULATION INLET" := TRUE;
       "TRANSFER DB".BIT."MFG TO STORAGE-3 WITH INLINE HOMO"."PBV-117 MFG TO STORAGE – 3 TRANSFER LINE" := TRUE;
   ELSE
       "TRANSFER DB".BIT."MFG TO STORAGE-3 WITH INLINE HOMO"."PFBV-59 TANK OUTLET VALVE" := FALSE;
       "TRANSFER DB".BIT."MFG TO STORAGE-3 WITH INLINE HOMO"."PBV-114 TANK OUTLET TO INLINE HOMOGENIZER LINE" := FALSE;
       "TRANSFER DB".BIT."MFG TO STORAGE-3 WITH INLINE HOMO"."PBV-110 INLINE HOMOGENIZER TO INLET LINE" := FALSE;
       "TRANSFER DB".BIT."MFG TO STORAGE-3 WITH INLINE HOMO"."PAV-56 INLINE HOMO. SEAL COOLING INLET" := FALSE;
       "TRANSFER DB".BIT."MFG TO STORAGE-3 WITH INLINE HOMO"."INLINE 1 HOMOGENIZER MOTOR1 RUN" := FALSE;
       "TRANSFER DB".BIT."MFG TO STORAGE-3 WITH INLINE HOMO"."PBV-109 HOMO. RECIRCULATION INLET" := FALSE;
       "TRANSFER DB".BIT."MFG TO STORAGE-3 WITH INLINE HOMO"."PBV-117 MFG TO STORAGE – 3 TRANSFER LINE" := FALSE;
       ;
   END_IF;
END_REGION

REGION Network 73: LOAD CELL_CUTOFF
   RUNG wire#powerrail
      { S7_Templates := "SrcType := Int" } NE_Contact(in1 := "MODE SELECTION DB"."MODE BUFF", in2 := 0)
      { S7_Templates := "SrcType := Int" } EQ_Contact(in1 := "TRANSFER DB".BUFF."MFG TO STORAGE-3 WITH INLINE HOMO", in2 := 2)
      I_Contact( "TRANSFER DB".PAUSE."MFG TO STORAGE-3 WITH INLINE HOMO" )
      { S7_Templates := "SrcType := Int" } NE_Contact(in1 := "CONTINUE DB"."SYRUP MFG PROCESS ERROR", in2 := 1)
      { S7_Templates := "SrcType := Int" } EQ_Contact(in1 := "LEVEL BUFF"."SYRUP MFG_LOAD CELL", in2 := 1)
      Move(in := 3, out1 => "TRANSFER DB".BUFF."MFG TO STORAGE-3 WITH INLINE HOMO")
   END_RUNG
   // the same network as SCL:
   IF ("MODE SELECTION DB"."MODE BUFF" <> 0) AND ("TRANSFER DB".BUFF."MFG TO STORAGE-3 WITH INLINE HOMO" = 2) AND NOT "TRANSFER DB".PAUSE."MFG TO STORAGE-3 WITH INLINE HOMO" AND ("CONTINUE DB"."SYRUP MFG PROCESS ERROR" <> 1) AND ("LEVEL BUFF"."SYRUP MFG_LOAD CELL" = 1) THEN
       "TRANSFER DB".BUFF."MFG TO STORAGE-3 WITH INLINE HOMO" := 3;
   END_IF;
END_REGION

REGION Network 74: PROCESS OVER & STOP
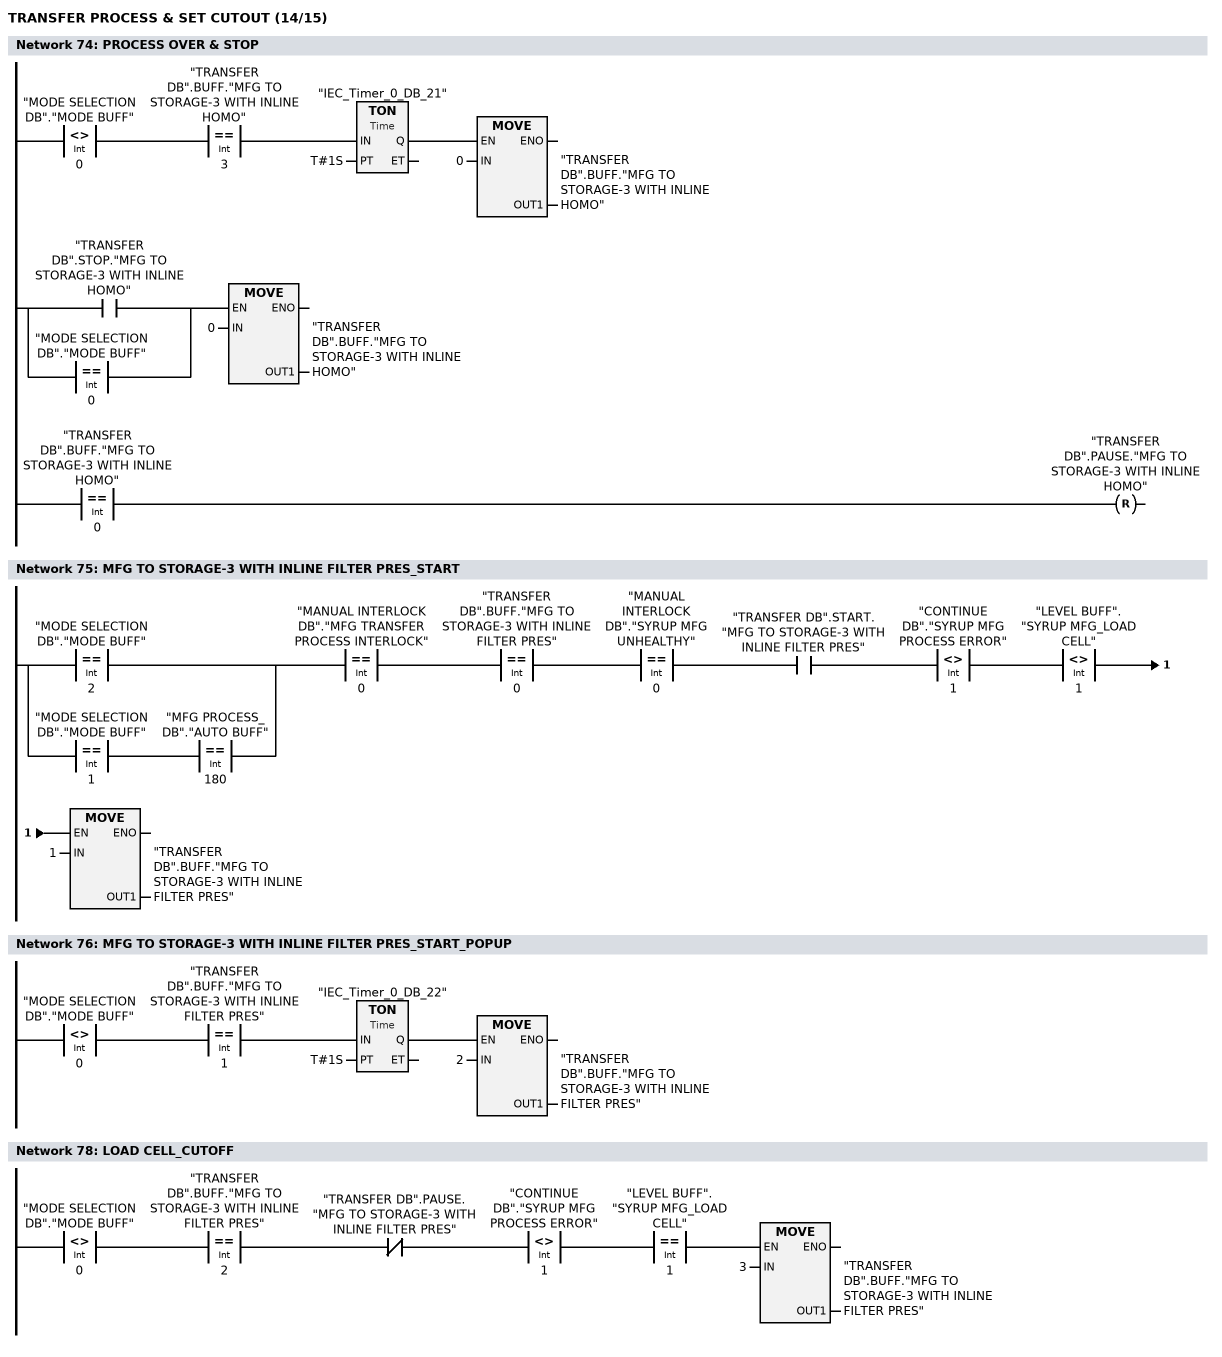
   RUNG wire#powerrail
      { S7_Templates := "SrcType := Int" } NE_Contact(in1 := "MODE SELECTION DB"."MODE BUFF", in2 := 0)
      { S7_Templates := "SrcType := Int" } EQ_Contact(in1 := "TRANSFER DB".BUFF."MFG TO STORAGE-3 WITH INLINE HOMO", in2 := 3)
      { S7_Templates := "time_type := Time" } "IEC_Timer_0_DB_21".TON(pt := T#1S, et =>)
      Move(in := 0, out1 => "TRANSFER DB".BUFF."MFG TO STORAGE-3 WITH INLINE HOMO")
   END_RUNG
   RUNG wire#powerrail
      Contact( "TRANSFER DB".STOP."MFG TO STORAGE-3 WITH INLINE HOMO" )
      wire#w1
      Move(in := 0, out1 => "TRANSFER DB".BUFF."MFG TO STORAGE-3 WITH INLINE HOMO")
   END_RUNG
   RUNG wire#powerrail
      { S7_Templates := "SrcType := Int" } EQ_Contact(in1 := "MODE SELECTION DB"."MODE BUFF", in2 := 0)
   END_RUNG wire#w1
   RUNG wire#powerrail
      { S7_Templates := "SrcType := Int" } EQ_Contact(in1 := "TRANSFER DB".BUFF."MFG TO STORAGE-3 WITH INLINE HOMO", in2 := 0)
      R_Coil( "TRANSFER DB".PAUSE."MFG TO STORAGE-3 WITH INLINE HOMO" )
   END_RUNG
   // the same network as SCL:
   "IEC_Timer_0_DB_21".TON(IN := ("MODE SELECTION DB"."MODE BUFF" <> 0) AND ("TRANSFER DB".BUFF."MFG TO STORAGE-3 WITH INLINE HOMO" = 3),
                           PT := T#1S);
   IF "IEC_Timer_0_DB_21".Q THEN "TRANSFER DB".BUFF."MFG TO STORAGE-3 WITH INLINE HOMO" := 0; END_IF;
   IF "TRANSFER DB".STOP."MFG TO STORAGE-3 WITH INLINE HOMO" OR ("MODE SELECTION DB"."MODE BUFF" = 0) THEN
       "TRANSFER DB".BUFF."MFG TO STORAGE-3 WITH INLINE HOMO" := 0;
   END_IF;
   IF "TRANSFER DB".BUFF."MFG TO STORAGE-3 WITH INLINE HOMO" = 0 THEN
       "TRANSFER DB".PAUSE."MFG TO STORAGE-3 WITH INLINE HOMO" := FALSE;
   END_IF;
END_REGION

REGION Network 75: MFG TO STORAGE-3 WITH INLINE FILTER PRES_START
   RUNG wire#powerrail
      { S7_Templates := "SrcType := Int" } EQ_Contact(in1 := "MODE SELECTION DB"."MODE BUFF", in2 := 2)
      wire#w1
      { S7_Templates := "SrcType := Int" } EQ_Contact(in1 := "MANUAL INTERLOCK DB"."MFG TRANSFER PROCESS INTERLOCK", in2 := 0)
      { S7_Templates := "SrcType := Int" } EQ_Contact(in1 := "TRANSFER DB".BUFF."MFG TO STORAGE-3 WITH INLINE FILTER PRES", in2 := 0)
      { S7_Templates := "SrcType := Int" } EQ_Contact(in1 := "MANUAL INTERLOCK DB"."SYRUP MFG UNHEALTHY", in2 := 0)
      Contact( "TRANSFER DB".START."MFG TO STORAGE-3 WITH INLINE FILTER PRES" )
      { S7_Templates := "SrcType := Int" } NE_Contact(in1 := "CONTINUE DB"."SYRUP MFG PROCESS ERROR", in2 := 1)
      { S7_Templates := "SrcType := Int" } NE_Contact(in1 := "LEVEL BUFF"."SYRUP MFG_LOAD CELL", in2 := 1)
      Move(in := 1, out1 => "TRANSFER DB".BUFF."MFG TO STORAGE-3 WITH INLINE FILTER PRES")
   END_RUNG
   RUNG wire#powerrail
      { S7_Templates := "SrcType := Int" } EQ_Contact(in1 := "MODE SELECTION DB"."MODE BUFF", in2 := 1)
      { S7_Templates := "SrcType := Int" } EQ_Contact(in1 := "MFG PROCESS_DB"."AUTO BUFF", in2 := 180)
   END_RUNG wire#w1
   // the same network as SCL:
   IF (("MODE SELECTION DB"."MODE BUFF" = 2) OR (("MODE SELECTION DB"."MODE BUFF" = 1) AND ("MFG PROCESS_DB"."AUTO BUFF" = 180))) AND ("MANUAL INTERLOCK DB"."MFG TRANSFER PROCESS INTERLOCK" = 0) AND ("TRANSFER DB".BUFF."MFG TO STORAGE-3 WITH INLINE FILTER PRES" = 0) AND ("MANUAL INTERLOCK DB"."SYRUP MFG UNHEALTHY" = 0) AND "TRANSFER DB".START."MFG TO STORAGE-3 WITH INLINE FILTER PRES" AND ("CONTINUE DB"."SYRUP MFG PROCESS ERROR" <> 1) AND ("LEVEL BUFF"."SYRUP MFG_LOAD CELL" <> 1) THEN
       "TRANSFER DB".BUFF."MFG TO STORAGE-3 WITH INLINE FILTER PRES" := 1;
   END_IF;
END_REGION

REGION Network 76: MFG TO STORAGE-3 WITH INLINE FILTER PRES_START_POPUP
   RUNG wire#powerrail
      { S7_Templates := "SrcType := Int" } NE_Contact(in1 := "MODE SELECTION DB"."MODE BUFF", in2 := 0)
      { S7_Templates := "SrcType := Int" } EQ_Contact(in1 := "TRANSFER DB".BUFF."MFG TO STORAGE-3 WITH INLINE FILTER PRES", in2 := 1)
      { S7_Templates := "time_type := Time" } "IEC_Timer_0_DB_22".TON(pt := T#1S, et =>)
      Move(in := 2, out1 => "TRANSFER DB".BUFF."MFG TO STORAGE-3 WITH INLINE FILTER PRES")
   END_RUNG
   // the same network as SCL:
   "IEC_Timer_0_DB_22".TON(IN := ("MODE SELECTION DB"."MODE BUFF" <> 0) AND ("TRANSFER DB".BUFF."MFG TO STORAGE-3 WITH INLINE FILTER PRES" = 1),
                           PT := T#1S);
   IF "IEC_Timer_0_DB_22".Q THEN "TRANSFER DB".BUFF."MFG TO STORAGE-3 WITH INLINE FILTER PRES" := 2; END_IF;
END_REGION

REGION Network 77 (SCL): OPENVALVE
   IF ("MODE SELECTION DB"."MODE BUFF" <> 0 AND "TRANSFER DB".BUFF."MFG TO STORAGE-3 WITH INLINE FILTER PRES" = 2
       AND NOT "TRANSFER DB".PAUSE."MFG TO STORAGE-3 WITH INLINE FILTER PRES"
       AND "CONTINUE DB"."SYRUP MFG PROCESS ERROR" = 0 AND "LEVEL BUFF"."SYRUP MFG_LOAD CELL" = 0)
       OR ("MODE SELECTION DB"."MODE BUFF"=1 AND "MFG PROCESS_DB"."AUTO BUFF"=0
       AND "MFG TRANSFER CYCLE DB".TRANSFER."TRANSFER BUFF"."MFG TO STORAGE-3 WITH INLINE FILTER PRES"=10 AND "CONTINUE DB"."SYRUP MFG PROCESS ERROR" <>1
       AND "MFG TRANSFER CYCLE DB".TRANSFER.SELECT."SELECT BUFF"=6)
   THEN
       "TRANSFER DB".BIT."MFG TO STORAGE-3 WITH INLINE FILTER PRES"."PFBV-59 TANK OUTLET VALVE" := TRUE;
       "TRANSFER DB".BIT."MFG TO STORAGE-3 WITH INLINE FILTER PRES"."PBV-114 TANK OUTLET TO INLINE HOMOGENIZER LINE" := TRUE;
       "TRANSFER DB".BIT."MFG TO STORAGE-3 WITH INLINE FILTER PRES"."PBV-108 INLINE HOMOGENIZER TO FILTER PRESS INLET LINE" := TRUE;
       "TRANSFER DB".BIT."MFG TO STORAGE-3 WITH INLINE FILTER PRES"."FILTER PRESS MOTOR 1 RUN" := TRUE;
       "TRANSFER DB".BIT."MFG TO STORAGE-3 WITH INLINE FILTER PRES"."PBV-118 FILTER PRESS INLET" := TRUE;
       "TRANSFER DB".BIT."MFG TO STORAGE-3 WITH INLINE FILTER PRES"."PBV-111 FILTER PRESS OUTLER VALVE" := TRUE;
       "TRANSFER DB".BIT."MFG TO STORAGE-3 WITH INLINE FILTER PRES"."PBV-112 FILTER PRESS TO TRANSFER LINE" := TRUE;
       "TRANSFER DB".BIT."MFG TO STORAGE-3 WITH INLINE FILTER PRES"."PBV-117 MFG TO STORAGE – 3 TRANSFER LINE" := TRUE;
   ELSE
       "TRANSFER DB".BIT."MFG TO STORAGE-3 WITH INLINE FILTER PRES"."PFBV-59 TANK OUTLET VALVE" := FALSE;
       "TRANSFER DB".BIT."MFG TO STORAGE-3 WITH INLINE FILTER PRES"."PBV-114 TANK OUTLET TO INLINE HOMOGENIZER LINE" := FALSE;
       "TRANSFER DB".BIT."MFG TO STORAGE-3 WITH INLINE FILTER PRES"."PBV-108 INLINE HOMOGENIZER TO FILTER PRESS INLET LINE" := FALSE;
       "TRANSFER DB".BIT."MFG TO STORAGE-3 WITH INLINE FILTER PRES"."FILTER PRESS MOTOR 1 RUN" := FALSE;
       "TRANSFER DB".BIT."MFG TO STORAGE-3 WITH INLINE FILTER PRES"."PBV-118 FILTER PRESS INLET" := FALSE;
       "TRANSFER DB".BIT."MFG TO STORAGE-3 WITH INLINE FILTER PRES"."PBV-111 FILTER PRESS OUTLER VALVE" := FALSE;
       "TRANSFER DB".BIT."MFG TO STORAGE-3 WITH INLINE FILTER PRES"."PBV-112 FILTER PRESS TO TRANSFER LINE" := FALSE;
       "TRANSFER DB".BIT."MFG TO STORAGE-3 WITH INLINE FILTER PRES"."PBV-117 MFG TO STORAGE – 3 TRANSFER LINE" := FALSE;
       ;
   END_IF;
END_REGION

REGION Network 78: LOAD CELL_CUTOFF
   RUNG wire#powerrail
      { S7_Templates := "SrcType := Int" } NE_Contact(in1 := "MODE SELECTION DB"."MODE BUFF", in2 := 0)
      { S7_Templates := "SrcType := Int" } EQ_Contact(in1 := "TRANSFER DB".BUFF."MFG TO STORAGE-3 WITH INLINE FILTER PRES", in2 := 2)
      I_Contact( "TRANSFER DB".PAUSE."MFG TO STORAGE-3 WITH INLINE FILTER PRES" )
      { S7_Templates := "SrcType := Int" } NE_Contact(in1 := "CONTINUE DB"."SYRUP MFG PROCESS ERROR", in2 := 1)
      { S7_Templates := "SrcType := Int" } EQ_Contact(in1 := "LEVEL BUFF"."SYRUP MFG_LOAD CELL", in2 := 1)
      Move(in := 3, out1 => "TRANSFER DB".BUFF."MFG TO STORAGE-3 WITH INLINE FILTER PRES")
   END_RUNG
   // the same network as SCL:
   IF ("MODE SELECTION DB"."MODE BUFF" <> 0) AND ("TRANSFER DB".BUFF."MFG TO STORAGE-3 WITH INLINE FILTER PRES" = 2) AND NOT "TRANSFER DB".PAUSE."MFG TO STORAGE-3 WITH INLINE FILTER PRES" AND ("CONTINUE DB"."SYRUP MFG PROCESS ERROR" <> 1) AND ("LEVEL BUFF"."SYRUP MFG_LOAD CELL" = 1) THEN
       "TRANSFER DB".BUFF."MFG TO STORAGE-3 WITH INLINE FILTER PRES" := 3;
   END_IF;
END_REGION

REGION Network 79: PROCESS OVER & STOP
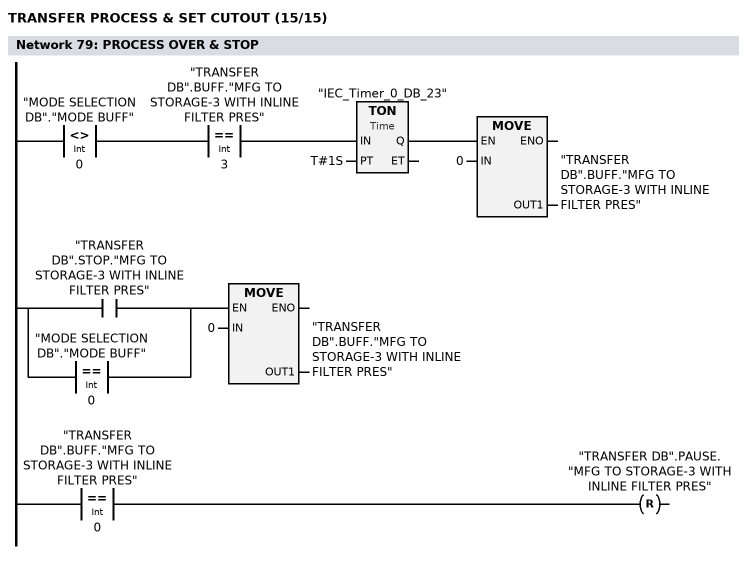
   RUNG wire#powerrail
      { S7_Templates := "SrcType := Int" } NE_Contact(in1 := "MODE SELECTION DB"."MODE BUFF", in2 := 0)
      { S7_Templates := "SrcType := Int" } EQ_Contact(in1 := "TRANSFER DB".BUFF."MFG TO STORAGE-3 WITH INLINE FILTER PRES", in2 := 3)
      { S7_Templates := "time_type := Time" } "IEC_Timer_0_DB_23".TON(pt := T#1S, et =>)
      Move(in := 0, out1 => "TRANSFER DB".BUFF."MFG TO STORAGE-3 WITH INLINE FILTER PRES")
   END_RUNG
   RUNG wire#powerrail
      Contact( "TRANSFER DB".STOP."MFG TO STORAGE-3 WITH INLINE FILTER PRES" )
      wire#w1
      Move(in := 0, out1 => "TRANSFER DB".BUFF."MFG TO STORAGE-3 WITH INLINE FILTER PRES")
   END_RUNG
   RUNG wire#powerrail
      { S7_Templates := "SrcType := Int" } EQ_Contact(in1 := "MODE SELECTION DB"."MODE BUFF", in2 := 0)
   END_RUNG wire#w1
   RUNG wire#powerrail
      { S7_Templates := "SrcType := Int" } EQ_Contact(in1 := "TRANSFER DB".BUFF."MFG TO STORAGE-3 WITH INLINE FILTER PRES", in2 := 0)
      R_Coil( "TRANSFER DB".PAUSE."MFG TO STORAGE-3 WITH INLINE FILTER PRES" )
   END_RUNG
   // the same network as SCL:
   "IEC_Timer_0_DB_23".TON(IN := ("MODE SELECTION DB"."MODE BUFF" <> 0) AND ("TRANSFER DB".BUFF."MFG TO STORAGE-3 WITH INLINE FILTER PRES" = 3),
                           PT := T#1S);
   IF "IEC_Timer_0_DB_23".Q THEN "TRANSFER DB".BUFF."MFG TO STORAGE-3 WITH INLINE FILTER PRES" := 0; END_IF;
   IF "TRANSFER DB".STOP."MFG TO STORAGE-3 WITH INLINE FILTER PRES" OR ("MODE SELECTION DB"."MODE BUFF" = 0) THEN
       "TRANSFER DB".BUFF."MFG TO STORAGE-3 WITH INLINE FILTER PRES" := 0;
   END_IF;
   IF "TRANSFER DB".BUFF."MFG TO STORAGE-3 WITH INLINE FILTER PRES" = 0 THEN
       "TRANSFER DB".PAUSE."MFG TO STORAGE-3 WITH INLINE FILTER PRES" := FALSE;
   END_IF;
END_REGION
END_FUNCTION

FUNCTION "TRANSFER SUBOUTPUT" : Void   // FC13, LAD
{ S7_Optimized_Access := 'TRUE' }
// stored: SetENOAutomatically false
BEGIN

REGION Network 1: SYRUP MFG VESSEL BOTTOM STERROR RUN
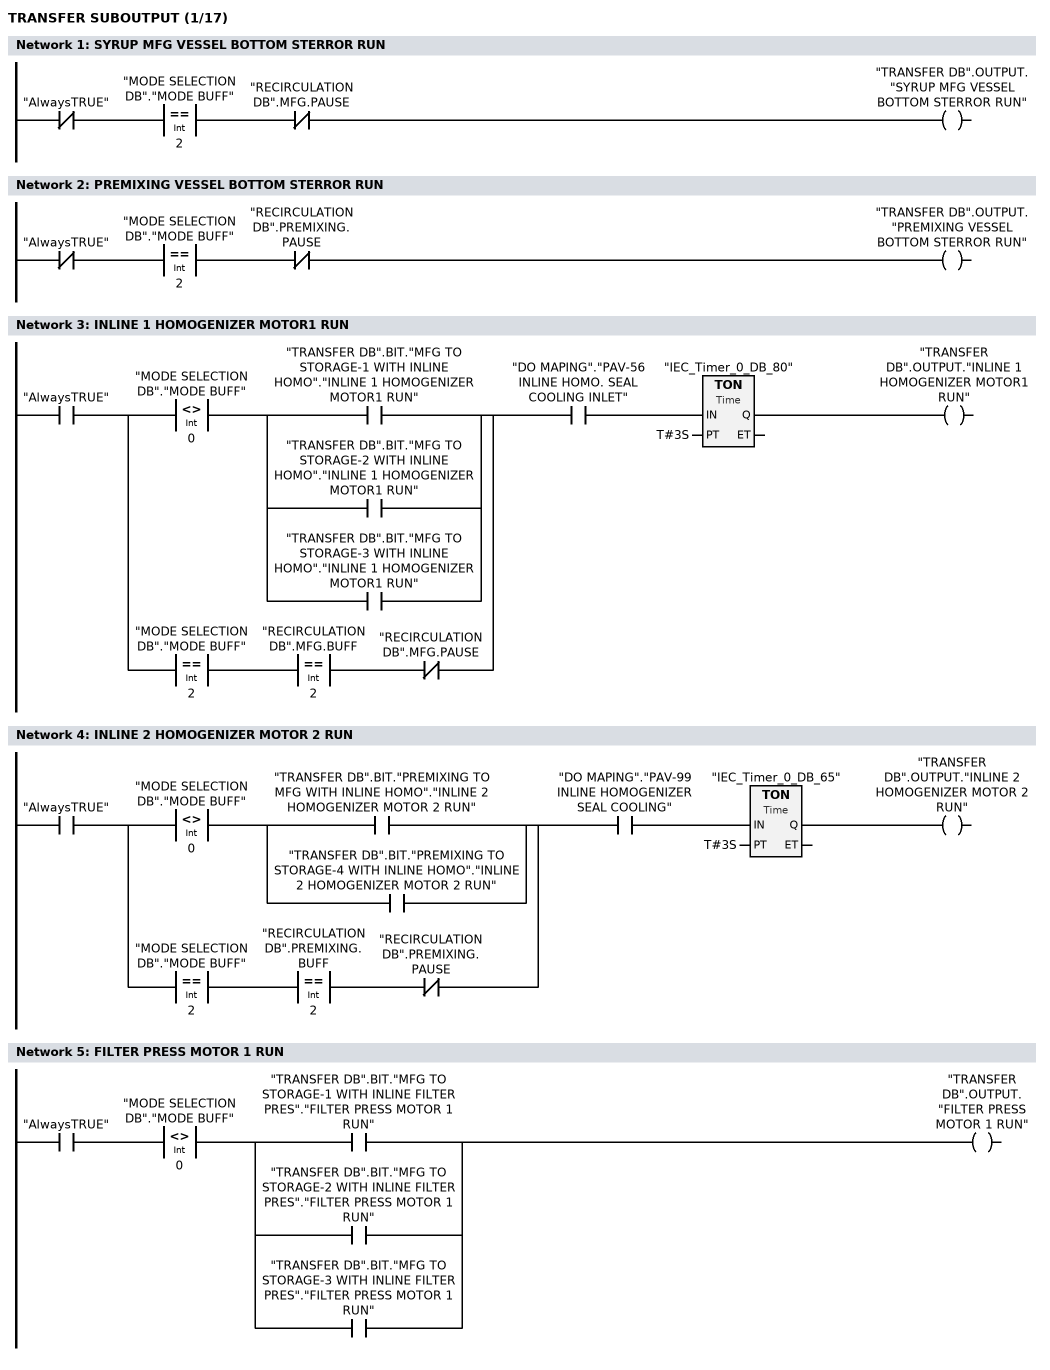
   RUNG wire#powerrail
      I_Contact( "AlwaysTRUE" )
      { S7_Templates := "SrcType := Int" } EQ_Contact(in1 := "MODE SELECTION DB"."MODE BUFF", in2 := 2)
      I_Contact( "RECIRCULATION DB".MFG.PAUSE )
      Coil( "TRANSFER DB".OUTPUT."SYRUP MFG VESSEL BOTTOM STERROR RUN" )
   END_RUNG
   // the same network as SCL:
   "TRANSFER DB".OUTPUT."SYRUP MFG VESSEL BOTTOM STERROR RUN" := NOT "AlwaysTRUE" AND ("MODE SELECTION DB"."MODE BUFF" = 2) AND NOT "RECIRCULATION DB".MFG.PAUSE;
END_REGION

